{Region "Angulo de rotação das válvulas"}
	//Linha 1
	CA1_L1_V1_POSIC AT %I*	:DUT_PosicValvula;
	CA1_L1_V2_POSIC AT %I*	:DUT_PosicValvula;
	CA1_L1_V3_POSIC AT %I*	:DUT_PosicValvula;
	CA1_L1_V4_POSIC AT %I*	:DUT_PosicValvula;
	//Linha 2
	CA1_L2_V1_POSIC AT %I*	:DUT_PosicValvula;
	CA1_L2_V2_POSIC AT %I*	:DUT_PosicValvula;
	CA1_L2_V3_POSIC AT %I*	:DUT_PosicValvula;
	CA1_L2_V4_POSIC AT %I*	:DUT_PosicValvula;
	//Linha 3
	CA1_L3_V1_POSIC AT %I*	:DUT_PosicValvula;
	CA1_L3_V2_POSIC AT %I*	:DUT_PosicValvula;
	CA1_L3_V3_POSIC AT %I*	:DUT_PosicValvula;
	CA1_L3_V4_POSIC AT %I*	:DUT_PosicValvula;
	//Linha 4
	CA1_L4_V1_POSIC AT %I*	:DUT_PosicValvula;
	CA1_L4_V2_POSIC AT %I*	:DUT_PosicValvula;
	CA1_L4_V3_POSIC AT %I*	:DUT_PosicValvula;
	CA1_L4_V4_POSIC AT %I*	:DUT_PosicValvula;
	
	//Linha 5
	CA2_L5_V1_POSIC AT %I*	:DUT_PosicValvula;
	CA2_L5_V2_POSIC AT %I*	:DUT_PosicValvula;
	CA2_L5_V3_POSIC AT %I*	:DUT_PosicValvula;
	CA2_L5_V4_POSIC AT %I*	:DUT_PosicValvula;
	//Linha 6
	CA2_L6_V1_POSIC AT %I*	:DUT_PosicValvula;
	CA2_L6_V2_POSIC AT %I*	:DUT_PosicValvula;
	CA2_L6_V3_POSIC AT %I*	:DUT_PosicValvula;
	CA2_L6_V4_POSIC AT %I*	:DUT_PosicValvula;
	//Linha 7
	CA2_L7_V1_POSIC AT %I*	:DUT_PosicValvula;
	CA2_L7_V2_POSIC AT %I*	:DUT_PosicValvula;
	CA2_L7_V3_POSIC AT %I*	:DUT_PosicValvula;
	CA2_L7_V4_POSIC AT %I*	:DUT_PosicValvula;
	//Linha 8
	CA2_L8_V1_POSIC AT %I*	:DUT_PosicValvula;
	CA2_L8_V2_POSIC AT %I*	:DUT_PosicValvula;
	CA2_L8_V3_POSIC AT %I*	:DUT_PosicValvula;
	CA2_L8_V4_POSIC AT %I*	:DUT_PosicValvula;
	
	//Linha 9
	CA3_L9_V1_POSIC AT %I*	:DUT_PosicValvula;
	CA3_L9_V2_POSIC AT %I*	:DUT_PosicValvula;
	CA3_L9_V3_POSIC AT %I*	:DUT_PosicValvula;
	CA3_L9_V4_POSIC AT %I*	:DUT_PosicValvula;
	//Linha 10
	CA3_L10_V1_POSIC AT %I*	:DUT_PosicValvula;
	CA3_L10_V2_POSIC AT %I*	:DUT_PosicValvula;
	CA3_L10_V3_POSIC AT %I*	:DUT_PosicValvula;
	CA3_L10_V4_POSIC AT %I*	:DUT_PosicValvula;
	//Linha 11
	CA3_L11_V1_POSIC AT %I*	:DUT_PosicValvula;
	CA3_L11_V2_POSIC AT %I*	:DUT_PosicValvula;
	CA3_L11_V3_POSIC AT %I*	:DUT_PosicValvula;
	CA3_L11_V4_POSIC AT %I*	:DUT_PosicValvula;
	//Linha 12
	CA3_L12_V1_POSIC AT %I*	:DUT_PosicValvula;
	CA3_L12_V2_POSIC AT %I*	:DUT_PosicValvula;
	CA3_L12_V3_POSIC AT %I*	:DUT_PosicValvula;
	CA3_L12_V4_POSIC AT %I*	:DUT_PosicValvula;
{endregion}
	
	
	
	
END_VAR

// ---- GVLs/HMI.TcGVL
{attribute 'qualified_only'}
VAR_GLOBAL
	//Hora de ajuste
	HoraParaAjuste:DT;
	
	//Lavagem das linhas
	IniciaLavagem :BOOL;	//Inicia lavagem na linha selecionada
	PararLavagem:BOOL;		//Interrompe a lavagem
	AbreValvResid:BOOL;		//Abre a válvula de água resisdual
	AbreValvLimpa:BOOL;		//Abre a válvula de água limpa
	
	// General
	bModo_Auto:BOOL;
	bModo_Ciclico:BOOL;
	bModo_UnCiclo:BOOL;
	bMarcha		:BOOL;
	bParada		:BOOL;
	bReset_Alarma:BOOL;
	bPB_vaciarTolva:BOOL;
	bRun			:BOOL;
	bPesoFueraTolerancia :BOOL;
	bDemoraCargaBalanza	:BOOL;
	bDescargarBalanza	:BOOL;
	iCircuito_a_calibrar:INT;
	bPararTolvaSupVacia:BOOL;
	tTiempoBatch:DINT;

	//Agitadores
	PP1_L1_AG_Cmd_Man:BOOL;
	PP1_L1_AG_Alr:BOOL;
	PP1_L1_AG_Alr_discr:BOOL;
	PP1_L1_AG_Estado:INT;
	bPP1_L1_AG_HsParc:DINT;
	bPP1_L1_AG_HsTot:DINT;	
	bPP1_L1_AG_RstHs:BOOL;
	bPP1_L1_AG_RstALr:BOOL;
	//
	PP1_L2_AG_Cmd_Man:BOOL;
	PP1_L2_AG_Alr:BOOL;
	PP1_L2_AG_Alr_discr:BOOL;
	PP1_L2_AG_Estado:INT;
	bPP1_L2_AG_HsParc:DINT;
	bPP1_L2_AG_HsTot:DINT;	
	bPP1_L2_AG_RstHs:BOOL;
	bPP1_L2_AG_RstALr:BOOL;
	//
	PP1_L3_AG_Cmd_Man:BOOL;
	PP1_L3_AG_Alr:BOOL;
	PP1_L3_AG_Alr_discr:BOOL;
	PP1_L3_AG_Estado:INT;
	bPP1_L3_AG_HsParc:DINT;
	bPP1_L3_AG_HsTot:DINT;	
	bPP1_L3_AG_RstHs:BOOL;
	bPP1_L3_AG_RstALr:BOOL;
	//
	PP1_L4_AG_Cmd_Man:BOOL;
	PP1_L4_AG_Alr:BOOL;
	PP1_L4_AG_Alr_discr:BOOL;
	PP1_L4_AG_Estado:INT;
	bPP1_L4_AG_HsParc:DINT;
	bPP1_L4_AG_HsTot:DINT;	
	bPP1_L4_AG_RstHs:BOOL;
	bPP1_L4_AG_RstALr:BOOL;
	
	PP2_L5_AG_Cmd_Man:BOOL;
	PP2_L5_AG_Alr:BOOL;
	PP2_L5_AG_Alr_discr:BOOL;
	PP2_L5_AG_Estado:INT;
	bPP2_L5_AG_HsParc:DINT;
	bPP2_L5_AG_HsTot:DINT;	
	bPP2_L5_AG_RstHs:BOOL;
	bPP2_L5_AG_RstALr:BOOL;
	//
	PP2_L6_AG_Cmd_Man:BOOL;
	PP2_L6_AG_Alr:BOOL;
	PP2_L6_AG_Alr_discr:BOOL;
	PP2_L6_AG_Estado:INT;
	bPP2_L6_AG_HsParc:DINT;
	bPP2_L6_AG_HsTot:DINT;	
	bPP2_L6_AG_RstHs:BOOL;
	bPP2_L6_AG_RstALr:BOOL;
	//
	PP2_L7_AG_Cmd_Man:BOOL;
	PP2_L7_AG_Alr:BOOL;
	PP2_L7_AG_Alr_discr:BOOL;
	PP2_L7_AG_Estado:INT;
	bPP2_L7_AG_HsParc:DINT;
	bPP2_L7_AG_HsTot:DINT;	
	bPP2_L7_AG_RstHs:BOOL;
	bPP2_L7_AG_RstALr:BOOL;
		//
	PP2_L8_AG_Cmd_Man:BOOL;
	PP2_L8_AG_Alr:BOOL;
	PP2_L8_AG_Alr_discr:BOOL;
	PP2_L8_AG_Estado:INT;
	bPP2_L8_AG_HsParc:DINT;
	bPP2_L8_AG_HsTot:DINT;	
	bPP2_L8_AG_RstHs:BOOL;
	bPP2_L8_AG_RstALr:BOOL;
	//
	PP3_L9_AG_Cmd_Man:BOOL;
	PP3_L9_AG_Alr:BOOL;
	PP3_L9_AG_Alr_discr:BOOL;
	PP3_L9_AG_Estado:INT;
	bPP3_L9_AG_HsParc:DINT;
	bPP3_L9_AG_HsTot:DINT;	
	bPP3_L9_AG_RstHs:BOOL;
	bPP3_L9_AG_RstALr:BOOL;
	//
	PP3_L10_AG_Cmd_Man:BOOL;
	PP3_L10_AG_Alr:BOOL;
	PP3_L10_AG_Alr_discr:BOOL;
	PP3_L10_AG_Estado:INT;
	bPP3_L10_AG_HsParc:DINT;
	bPP3_L10_AG_HsTot:DINT;	
	bPP3_L10_AG_RstHs:BOOL;
	bPP3_L10_AG_RstALr:BOOL;
	//
	PP3_L11_AG_Cmd_Man:BOOL;
	PP3_L11_AG_Alr:BOOL;
	PP3_L11_AG_Alr_discr:BOOL;
	PP3_L11_AG_Estado:INT;
	bPP3_L11_AG_HsParc:DINT;
	bPP3_L11_AG_HsTot:DINT;	
	bPP3_L11_AG_RstHs:BOOL;
	bPP3_L11_AG_RstALr:BOOL;
	//
	PP3_L12_AG_Cmd_Man:BOOL;
	PP3_L12_AG_Alr:BOOL;
	PP3_L12_AG_Alr_discr:BOOL;
	PP3_L12_AG_Estado:INT;
	bPP3_L12_AG_HsParc:DINT;
	bPP3_L12_AG_HsTot:DINT;	
	bPP3_L12_AG_RstHs:BOOL;
	bPP3_L12_AG_RstALr:BOOL;
	
	
	//Soplador tratadora
	TR_S_VE1_Cmd_Man:BOOL;
	TR_S_VE1_Alr:BOOL;
	TR_S_VE1_Alr_discr:BOOL;
	TR_S_VE1_Estado:INT;
	TR_S_VE1_HsParc:DINT;
	TR_S_VE1_HsTot:DINT;	
	TR_S_VE1_RstHs:BOOL;
	TR_S_VE1_RstAlr:BOOL;
	
	//Lavado Gral
	bBypassNivelAguaResidual:BOOL;
	
	//Lavado Circuito 1
	bInicioLavado_Cir1:BOOL;//Inicio de Lavado
	bModoECO_Cir1:BOOL;//Seleccion modo ECO
	bCancelarLavado_Cir1:BOOL;//Cancelacion de lavado (finaliza con circuito vacio)
	wEstadoLavado_Cir1:WORD; //1=vaciado 2=prelavado 3=lavado
	iCantCiclosLavado_Cir1:INT;//Cantidad de ciclos a realizar de Lavado
	iCantCiclosECO_Cir1:INT;//Cantidad de ciclos a realizar de Eco
	rPorcECO_Cir1:REAL;//Porcentaje de ciclos ECO en relacion al total pedido (ECO+Lavado)
	rPorcLavado_Cir1:REAL;//Porcentaje de ciclos Lavado en relacion al total pedido (ECO+Lavado)
	rPorcAvance_Cir1:REAL;//Porcentaje de avance en relacion al total pedido (ECO+Lavado)
	tSetTmrVaciado_Cir1:TIME;//Tiempo luego de detectar caudalimetro inferior en cero
	tSetTmrLlenado_Cir1:TIME;//Tiempo luego de detectar caudalimetro superior mayor a cero
	rVelBbaVaciado_Cir1:REAL;//Velocidad de bomba durante vaciado (unidad?)
	rVelBbaLlenado_Cir1:REAL;//Velocidad de bomba durante llenado (unidad?)
	
	//valvula descarga semilla de tambor
	TR_S_V1_Cmd_Man		:BOOL;
	TR_S_V1_Alr			:BOOL;
	TR_S_V1_Alr_discr	:BOOL;
	TR_S_V1_Estado		:INT;  // 1= cerrado 2=abierto 3=alarma 4=emergencia
	TR_S_V1_EventoParc	:DINT;//cant de actuaciones parciales
	TR_S_V1_EventoTot	:DINT;//cant de actuaciones totales
	
	//valvula carga grueso semilla a balanza
	TR_S_V2_Cmd_Man		:BOOL;
	TR_S_V2_Alr			:BOOL;
	TR_S_V2_Alr_discr	:BOOL;
	TR_S_V2_Estado		:INT;
	
	//valvula carga fino semilla a balanza
	TR_S_V3_Cmd_Man		:BOOL;
	TR_S_V3_Alr			:BOOL;
	TR_S_V3_Alr_discr	:BOOL;
	TR_S_V3_Estado		:INT;
	
	//valvula descarga semilla de balanza
	TR_S_V4_Cmd_Man		:BOOL;
	TR_S_V4_Alr			:BOOL;
	TR_S_V4_Alr_discr	:BOOL;
	TR_S_V4_Estado		:INT;
	
	
	//Homogenizador
	CmdM_TR_S_VF1		:BOOL; //marcha en manual
	CmdR_TR_S_VF1		:BOOL; //seleccion reversa en manual
	StMarcha_TR_S_VF1	:BOOL; //confirmacion en marcha
	StAlarma_TR_S_VF1	:BOOL;
	StVeloc_TR_S_VF1	:INT;	
	
	//Aspersor
	CmdM_TR_S_VF2		:BOOL; //marcha en manual
	CmdR_TR_S_VF2		:BOOL; //seleccion reversa en manual
	StMarcha_TR_S_VF2	:BOOL; //confirmacion en marcha
	StAlarma_TR_S_VF2	:BOOL;
	StVeloc_TR_S_VF2	:INT;	
	
	//Valv Calibracion L1
	CA1_L1_V1_estado	:INT;
	CA1_L1_V1_Cmd_Man	:BOOL;
	CA1_L1_V1_RsAlr		:BOOL;
	//Valv Calibracion L2
	CA1_L2_V1_estado	:INT;
	CA1_L2_V1_Cmd_Man	:BOOL;
	CA1_L2_V1_RsAlr		:BOOL;	
	//Valv Calibracion L3
	CA1_L3_V1_estado	:INT;
	CA1_L3_V1_Cmd_Man	:BOOL;
	CA1_L3_V1_RsAlr		:BOOL;
	//Valv Calibracion L4
	CA1_L4_V1_estado	:INT;
	CA1_L4_V1_Cmd_Man	:BOOL;
	CA1_L4_V1_RsAlr		:BOOL;
	//Valv Calibracion L5
	CA2_L5_V1_estado	:INT;
	CA2_L5_V1_Cmd_Man	:BOOL;
	CA2_L5_V1_RsAlr		:BOOL;
	//Valv Calibracion L6
	CA2_L6_V1_estado	:INT;
	CA2_L6_V1_Cmd_Man	:BOOL;
	CA2_L6_V1_RsAlr		:BOOL;
	//Valv Calibracion L7
	CA2_L7_V1_estado	:INT;
	CA2_L7_V1_Cmd_Man	:BOOL;
	CA2_L7_V1_RsAlr		:BOOL;
	//Valv Calibracion L8
	CA2_L8_V1_estado	:INT;
	CA2_L8_V1_Cmd_Man	:BOOL;
	CA2_L8_V1_RsAlr		:BOOL;				
	//Valv Calibracion L9
	CA3_L9_V1_estado	:INT;
	CA3_L9_V1_Cmd_Man	:BOOL;	
	CA3_L9_V1_RsAlr		:BOOL;
	//Valv Calibracion L10
	CA3_L10_V1_estado	:INT;
	CA3_L10_V1_Cmd_Man	:BOOL;
	CA3_L10_V1_RsAlr		:BOOL;
	//Valv Calibracion L11
	CA3_L11_V1_estado	:INT;
	CA3_L11_V1_Cmd_Man	:BOOL;
	CA3_L11_V1_RsAlr		:BOOL;	
	//Valv Calibracion L12
	CA3_L12_V1_estado	:INT;
	CA3_L12_V1_Cmd_Man	:BOOL;
	CA3_L12_V1_RsAlr		:BOOL;		
	
	//Valv Calibracion L1
	CA1_L1_V2_estado	:INT;
	CA1_L1_V2_Cmd_Man	:BOOL;
	CA1_L1_V2_RsAlr		:BOOL;
	//Valv Lavado L1
	CA1_L1_V3_estado	:INT;
	CA1_L1_V3_Cmd_Man	:BOOL;
	CA1_L1_V3_RsAlr		:BOOL;
	//Valv IBC L1
	CA1_L1_V4_estado	:INT;
	CA1_L1_V4_Cmd_Man	:BOOL;
	CA1_L1_V4_RsAlr		:BOOL;
	//Valv Calibracion L2
	CA1_L2_V2_estado	:INT;
	CA1_L2_V2_Cmd_Man	:BOOL;
	CA1_L2_V2_RsAlr		:BOOL;
	//Valv Lavado L2
	CA1_L2_V3_estado	:INT;
	CA1_L2_V3_Cmd_Man	:BOOL;
	CA1_L2_V3_RsAlr		:BOOL;
	//Valv IBC L2
	CA1_L2_V4_estado	:INT;
	CA1_L2_V4_Cmd_Man	:BOOL;
	CA1_L2_V4_RsAlr		:BOOL;
	//Valv Calibracion L3
	CA1_L3_V2_estado	:INT;
	CA1_L3_V2_Cmd_Man	:BOOL;
	CA1_L3_V2_RsAlr		:BOOL;
	//Valv Lavado L3
	CA1_L3_V3_estado	:INT;
	CA1_L3_V3_Cmd_Man	:BOOL;
	CA1_L3_V3_RsAlr		:BOOL;
	//Valv IBC L3
	CA1_L3_V4_estado	:INT;
	CA1_L3_V4_Cmd_Man	:BOOL;
	CA1_L3_V4_RsAlr		:BOOL;
	//Valv Calibracion L4
	CA1_L4_V2_estado	:INT;
	CA1_L4_V2_Cmd_Man	:BOOL;
	CA1_L4_V2_RsAlr		:BOOL;
	//Valv Lavado L4
	CA1_L4_V3_estado	:INT;
	CA1_L4_V3_Cmd_Man	:BOOL;
	CA1_L4_V3_RsAlr		:BOOL;
	//Valv IBC L4
	CA1_L4_V4_estado	:INT;
	CA1_L4_V4_Cmd_Man	:BOOL;
	CA1_L4_V4_RsAlr		:BOOL;
	//Valv Calibracion L5
	CA2_L5_V2_estado	:INT;
	CA2_L5_V2_Cmd_Man	:BOOL;
	CA2_L5_V2_RsAlr		:BOOL;
	//Valv Lavado L5
	CA2_L5_V3_estado	:INT;
	CA2_L5_V3_Cmd_Man	:BOOL;
	CA2_L5_V3_RsAlr		:BOOL;
	//Valv IBC L5
	CA2_L5_V4_estado	:INT;
	CA2_L5_V4_Cmd_Man	:BOOL;
	CA2_L5_V4_RsAlr		:BOOL;
	//Valv Calibracion L6
	CA2_L6_V2_estado	:INT;
	CA2_L6_V2_Cmd_Man	:BOOL;
	CA2_L6_V2_RsAlr		:BOOL;
	//Valv Lavado L6
	CA2_L6_V3_estado	:INT;
	CA2_L6_V3_Cmd_Man	:BOOL;
	CA2_L6_V3_RsAlr		:BOOL;
	//Valv IBC L6
	CA2_L6_V4_estado	:INT;
	CA2_L6_V4_Cmd_Man	:BOOL;
	CA2_L6_V4_RsAlr		:BOOL;
	//Valv Calibracion L7
	CA2_L7_V2_estado	:INT;
	CA2_L7_V2_Cmd_Man	:BOOL;
	CA2_L7_V2_RsAlr		:BOOL;
	//Valv Lavado L7
	CA2_L7_V3_estado	:INT;
	CA2_L7_V3_Cmd_Man	:BOOL;
	CA2_L7_V3_RsAlr		:BOOL;
	//Valv IBC L7
	CA2_L7_V4_estado	:INT;
	CA2_L7_V4_Cmd_Man	:BOOL;
	CA2_L7_V4_RsAlr		:BOOL;
	//Valv Calibracion L8
	CA2_L8_V2_estado	:INT;
	CA2_L8_V2_Cmd_Man	:BOOL;
	CA2_L8_V2_RsAlr		:BOOL;
	//Valv Lavado L8
	CA2_L8_V3_estado	:INT;
	CA2_L8_V3_Cmd_Man	:BOOL;
	CA2_L8_V3_RsAlr		:BOOL;
	//Valv IBC L8
	CA2_L8_V4_estado	:INT;
	CA2_L8_V4_Cmd_Man	:BOOL;
	CA2_L8_V4_RsAlr		:BOOL;
	//Valv Calibracion L9
	CA3_L9_V2_estado	:INT;
	CA3_L9_V2_Cmd_Man	:BOOL;
	CA3_L9_V2_RsAlr		:BOOL;
	//Valv Lavado L9
	CA3_L9_V3_estado	:INT;
	CA3_L9_V3_Cmd_Man	:BOOL;
	CA3_L9_V3_RsAlr		:BOOL;
	//Valv IBC L9
	CA3_L9_V4_estado	:INT;
	CA3_L9_V4_Cmd_Man	:BOOL;
	CA3_L9_V4_RsAlr		:BOOL;
	//Valv Calibracion L10
	CA3_L10_V2_estado	:INT;
	CA3_L10_V2_Cmd_Man	:BOOL;
	CA3_L10_V2_RsAlr	:BOOL;
	//Valv Lavado L10
	CA3_L10_V3_estado	:INT;
	CA3_L10_V3_Cmd_Man	:BOOL;
	CA3_L10_V3_RsAlr	:BOOL;
	//Valv IBC L10
	CA3_L10_V4_estado	:INT;
	CA3_L10_V4_Cmd_Man	:BOOL;
	CA3_L10_V4_RsAlr	:BOOL;
	//Valv Calibracion L11
	CA3_L11_V2_estado	:INT;
	CA3_L11_V2_Cmd_Man	:BOOL;
	CA3_L11_V2_RsAlr	:BOOL;
	//Valv Lavado L11
	CA3_L11_V3_estado	:INT;
	CA3_L11_V3_Cmd_Man	:BOOL;
	CA3_L11_V3_RsAlr	:BOOL;
	//Valv IBC L11
	CA3_L11_V4_estado	:INT;
	CA3_L11_V4_Cmd_Man	:BOOL;
	CA3_L11_V4_RsAlr	:BOOL;
	//Valv Calibracion L12
	CA3_L12_V2_estado	:INT;
	CA3_L12_V2_Cmd_Man	:BOOL;
	CA3_L12_V2_RsAlr	:BOOL;
	//Valv Lavado L12
	CA3_L12_V3_estado	:INT;
	CA3_L12_V3_Cmd_Man	:BOOL;
	CA3_L12_V3_RsAlr	:BOOL;
	//Valv IBC L12
	CA3_L12_V4_estado	:INT;
	CA3_L12_V4_Cmd_Man	:BOOL;
	CA3_L12_V4_RsAlr	:BOOL;
	//Valv Agua limpia
	PU_Lav_V5_estado	:INT;
	PU_Lav_V5_Cmd_Man	:BOOL;
	PU_Lav_V5_RsAlr		:BOOL;
	//Valv Agua residual
	PU_Lav_V6_estado	:INT;
	PU_Lav_V6_Cmd_Man	:BOOL;
	PU_Lav_V6_RsAlr		:BOOL;	
	
	//Bomba circuito L1
	CmdM_PC1_L1_BD	:BOOL; //marcha en manual
	CmdR_PC1_L1_BD	:BOOL; //seleccion reversa en manual
	StMarcha_PC1_L1_BD :BOOL; //confirmacion bomba en marcha
	StAlarma_PC1_L1_BD :BOOL;
	StVeloc_PC1_L1_BD :INT;
	//Bomba circuito L2
	CmdM_PC1_L2_BD	:BOOL; //marcha en manual
	CmdR_PC1_L2_BD	:BOOL; //seleccion reversa en manual
	StMarcha_PC1_L2_BD :BOOL; //confirmacion bomba en marcha
	StAlarma_PC1_L2_BD :BOOL;
	StVeloc_PC1_L2_BD :INT;	
	//Bomba circuito L3
	CmdM_PC1_L3_BD	:BOOL; //marcha en manual
	CmdR_PC1_L3_BD	:BOOL; //seleccion reversa en manual
	StMarcha_PC1_L3_BD :BOOL; //confirmacion bomba en marcha
	StAlarma_PC1_L3_BD :BOOL;
	StVeloc_PC1_L3_BD :INT;	
	//Bomba circuito L4
	CmdM_PC1_L4_BD	:BOOL; //marcha en manual
	CmdR_PC1_L4_BD	:BOOL; //seleccion reversa en manual
	StMarcha_PC1_L4_BD :BOOL; //confirmacion bomba en marcha
	StAlarma_PC1_L4_BD :BOOL;
	StVeloc_PC1_L4_BD :INT;		
	//Bomba circuito L5
	CmdM_PC2_L5_BD	:BOOL; //marcha en manual
	CmdR_PC2_L5_BD	:BOOL; //seleccion reversa en manual
	StMarcha_PC2_L5_BD :BOOL; //confirmacion bomba en marcha
	StAlarma_PC2_L5_BD :BOOL;
	StVeloc_PC2_L5_BD :INT;	
	//Bomba circuito L6
	CmdM_PC2_L6_BD	:BOOL; //marcha en manual
	CmdR_PC2_L6_BD	:BOOL; //seleccion reversa en manual
	StMarcha_PC2_L6_BD :BOOL; //confirmacion bomba en marcha
	StAlarma_PC2_L6_BD :BOOL;
	StVeloc_PC2_L6_BD :INT;	
	//Bomba circuito L7
	CmdM_PC2_L7_BD	:BOOL; //marcha en manual
	CmdR_PC2_L7_BD	:BOOL; //seleccion reversa en manual
	StMarcha_PC2_L7_BD :BOOL; //confirmacion bomba en marcha
	StAlarma_PC2_L7_BD :BOOL;
	StVeloc_PC2_L7_BD :INT;	
	//Bomba circuito L8
	CmdM_PC2_L8_BD	:BOOL; //marcha en manual
	CmdR_PC2_L8_BD	:BOOL; //seleccion reversa en manual
	StMarcha_PC2_L8_BD :BOOL; //confirmacion bomba en marcha
	StAlarma_PC2_L8_BD :BOOL;
	StVeloc_PC2_L8_BD :INT;					
	//Bomba circuito L9
	CmdM_PC3_L9_BD	:BOOL; //marcha en manual
	CmdR_PC3_L9_BD	:BOOL; //seleccion reversa en manual
	StMarcha_PC3_L9_BD :BOOL; //confirmacion bomba en marcha
	StAlarma_PC3_L9_BD :BOOL;
	StVeloc_PC3_L9_BD :INT;	
	//Bomba circuito L10
	CmdM_PC3_L10_BD	:BOOL; //marcha en manual
	CmdR_PC3_L10_BD	:BOOL; //seleccion reversa en manual
	StMarcha_PC3_L10_BD :BOOL; //confirmacion bomba en marcha
	StAlarma_PC3_L10_BD :BOOL;
	StVeloc_PC3_L10_BD :INT;
	//Bomba circuito L11
	CmdM_PC3_L11_BD	:BOOL; //marcha en manual
	CmdR_PC3_L11_BD	:BOOL; //seleccion reversa en manual
	StMarcha_PC3_L11_BD :BOOL; //confirmacion bomba en marcha
	StAlarma_PC3_L11_BD :BOOL;
	StVeloc_PC3_L11_BD :INT;
	//Bomba circuito L12
	CmdM_PC3_L12_BD	:BOOL; //marcha en manual
	CmdR_PC3_L12_BD	:BOOL; //seleccion reversa en manual
	StMarcha_PC3_L12_BD :BOOL; //confirmacion bomba en marcha
	StAlarma_PC3_L12_BD :BOOL;
	StVeloc_PC3_L12_BD :INT;		
	
	//Caudalimetros Calibracion
	CA1_L1_FT1_caudal :REAL;
	CA1_L1_FT1_temp :REAL;
	CA1_L2_FT1_caudal :REAL;
	CA1_L2_FT1_temp :REAL;	
	CA1_L3_FT1_caudal :REAL;
	CA1_L3_FT1_tot	:REAL;
	CA1_L3_FT1_temp :REAL;
	CA1_L4_FT1_caudal :REAL;
	CA1_L4_FT1_temp :REAL;
	CA2_L5_FT1_caudal :REAL;
	CA2_L5_FT1_temp :REAL;
	CA2_L6_FT1_caudal :REAL;
	CA2_L6_FT1_temp :REAL;	
	CA2_L7_FT1_caudal :REAL;
	CA2_L7_FT1_temp :REAL;
	CA2_L8_FT1_caudal :REAL;
	CA2_L8_FT1_temp :REAL;
	CA3_L9_FT1_caudal :REAL;
	CA3_L9_FT1_temp :REAL;
	CA3_L10_FT1_caudal :REAL;
	CA3_L10_FT1_temp :REAL;
	CA3_L11_FT1_caudal :REAL;
	CA3_L11_FT1_temp :REAL;
	CA3_L12_FT1_caudal :REAL;
	CA3_L12_FT1_temp :REAL;
	//Caudalimetros Tratadora
	TR_L1_FT2_caudal :REAL;
	TR_L1_FT2_temp :REAL;
	TR_L2_FT2_caudal :REAL;
	TR_L2_FT2_temp :REAL;	
	TR_L3_FT2_caudal :REAL;
	TR_L3_FT2_temp :REAL;
	TR_L4_FT2_caudal :REAL;
	TR_L4_FT2_temp :REAL;
	TR_L5_FT2_caudal :REAL;
	TR_L5_FT2_temp :REAL;
	TR_L6_FT2_caudal :REAL;
	TR_L6_FT2_temp :REAL;	
	TR_L7_FT2_caudal :REAL;
	TR_L7_FT2_temp :REAL;
	TR_L8_FT2_caudal :REAL;
	TR_L8_FT2_temp :REAL;
	TR_L9_FT2_caudal :REAL;
	TR_L9_FT2_temp :REAL;
	TR_L10_FT2_caudal :REAL;
	TR_L10_FT2_temp :REAL;
	TR_L11_FT2_caudal :REAL;
	TR_L11_FT2_temp :REAL;
	TR_L12_FT2_caudal :REAL;
	TR_L12_FT2_temp :REAL;
	//Balanza probeta CA1
	bCmd_Zero_WT_CA1 :BOOL;
	bCmd_Full_WT_CA1 :BOOL;
	bCmd_LoadReference_WT_CA1:BOOL;
	rPesoPatron_WT_CA1 :REAL;
	bCalibrado_WT_CA1:BOOL;
	//Balanza probeta CA2
	bCmd_Zero_WT_CA2 :BOOL;
	bCmd_Full_WT_CA2 :BOOL;
	bCmd_LoadReference_WT_CA2:BOOL;
	rPesoPatron_WT_CA2 :REAL;
	bCalibrado_WT_CA2:BOOL;	
	//Balanza probeta CA3
	bCmd_Zero_WT_CA3 :BOOL;
	bCmd_Full_WT_CA3 :BOOL;
	bCmd_LoadReference_WT_CA3:BOOL;
	rPesoPatron_WT_CA3 :REAL;
	bCalibrado_WT_CA3:BOOL;
	//Balanza IBC L1
	bCmd_Zero_WT1_PU1 :BOOL;
	bCmd_Full_WT1_PU1 :BOOL;
	bCmd_LoadReference_WT1_PU1:BOOL;
	rPesoPatron_WT1_PU1 :REAL;
	bCalibrado_WT1_PU1:BOOL;
	//Balanza IBC L2
	bCmd_Zero_WT2_PU1 :BOOL;
	bCmd_Full_WT2_PU1 :BOOL;
	bCmd_LoadReference_WT2_PU1:BOOL;
	rPesoPatron_WT2_PU1 :REAL;
	bCalibrado_WT2_PU1:BOOL;
	//Balanza IBC L3
	bCmd_Zero_WT3_PU1 :BOOL;
	bCmd_Full_WT3_PU1 :BOOL;
	bCmd_LoadReference_WT3_PU1:BOOL;
	rPesoPatron_WT3_PU1 :REAL;
	bCalibrado_WT3_PU1:BOOL;
	//Balanza IBC L4
	bCmd_Zero_WT4_PU1 :BOOL;
	bCmd_Full_WT4_PU1 :BOOL;
	bCmd_LoadReference_WT4_PU1:BOOL;
	rPesoPatron_WT4_PU1 :REAL;
	bCalibrado_WT4_PU1:BOOL;
	//Balanza IBC L5
	bCmd_Zero_WT5_PU2 :BOOL;
	bCmd_Full_WT5_PU2 :BOOL;
	bCmd_LoadReference_WT5_PU2:BOOL;
	rPesoPatron_WT5_PU2 :REAL;
	bCalibrado_WT5_PU2:BOOL;
	//Balanza IBC L6
	bCmd_Zero_WT6_PU2 :BOOL;
	bCmd_Full_WT6_PU2 :BOOL;
	bCmd_LoadReference_WT6_PU2:BOOL;
	rPesoPatron_WT6_PU2 :REAL;
	bCalibrado_WT6_PU2:BOOL;
	//Balanza IBC L7
	bCmd_Zero_WT7_PU2 :BOOL;
	bCmd_Full_WT7_PU2 :BOOL;
	bCmd_LoadReference_WT7_PU2:BOOL;
	rPesoPatron_WT7_PU2 :REAL;
	bCalibrado_WT7_PU2:BOOL;
	//Balanza IBC L8
	bCmd_Zero_WT8_PU2 :BOOL;
	bCmd_Full_WT8_PU2 :BOOL;
	bCmd_LoadReference_WT8_PU2:BOOL;
	rPesoPatron_WT8_PU2 :REAL;
	bCalibrado_WT8_PU2:BOOL;
	//Balanza IBC L9
	bCmd_Zero_WT9_PU3 :BOOL;
	bCmd_Full_WT9_PU3 :BOOL;
	bCmd_LoadReference_WT9_PU3:BOOL;
	rPesoPatron_WT9_PU3 :REAL;
	bCalibrado_WT9_PU3:BOOL;
	//Balanza IBC L10
	bCmd_Zero_WT10_PU3 :BOOL;
	bCmd_Full_WT10_PU3 :BOOL;
	bCmd_LoadReference_WT10_PU3:BOOL;
	rPesoPatron_WT10_PU3 :REAL;
	bCalibrado_WT10_PU3:BOOL;
	//Balanza IBC L11
	bCmd_Zero_WT11_PU3 :BOOL;
	bCmd_Full_WT11_PU3 :BOOL;
	bCmd_LoadReference_WT11_PU3:BOOL;
	rPesoPatron_WT11_PU3 :REAL;
	bCalibrado_WT11_PU3:BOOL;
	//Balanza IBC L12
	bCmd_Zero_WT12_PU3 :BOOL;
	bCmd_Full_WT12_PU3 :BOOL;
	bCmd_LoadReference_WT12_PU3:BOOL;
	rPesoPatron_WT12_PU3 :REAL;
	bCalibrado_WT12_PU3:BOOL;	
	//Balanza Semilla
	bCmd_Zero_TR_S_WT1 :BOOL;
	bCmd_Full_TR_S_WT1 :BOOL;
	bCmd_LoadReference_TR_S_WT1:BOOL;
	bInicio_Cal_TR_S_WT1 :BOOL;
	bCalibrando:BOOL;
	bCalibrado:BOOL;
	
	//Dosificador Polvo 1
	CmdM_TR_P1_VF	:BOOL; //marcha en manual
	CmdR_TR_P1_VF	:BOOL; //seleccion reversa en manual
	StMarcha_TR_P1_VF :BOOL; //confirmacion motor en marcha
	StAlarma_TR_P1_VF :BOOL;
	StVeloc_TR_P1_VF :INT;
	//Dosificador Polvo 2
	CmdM_TR_P2_VF	:BOOL; //marcha en manual
	CmdR_TR_P2_VF	:BOOL; //seleccion reversa en manual
	StMarcha_TR_P2_VF :BOOL; //confirmacion motor en marcha
	StAlarma_TR_P2_VF :BOOL;
	StVeloc_TR_P2_VF :INT;
	//Balanza Polvo 1
	bCmd_Zero_TR_P1_WT1 :BOOL;
	bCmd_Full_TR_P1_WT1 :BOOL;
	bCmd_LoadReference_TR_P1_WT1:BOOL;
	rPesoPatron_TR_P1_WT1 :REAL;
	bCalibrado_TR_P1_WT1:BOOL;	
	//Balanza Polvo 2
	bCmd_Zero_TR_P2_WT1 :BOOL;
	bCmd_Full_TR_P2_WT1 :BOOL;
	bCmd_LoadReference_TR_P2_WT1:BOOL;
	rPesoPatron_TR_P2_WT1 :REAL;
	bCalibrado_TR_P2_WT1:BOOL;	
	//Vibrador Polvo 1
	CmdM_TR_P1_VI	:BOOL; //marcha en manual
	CmdR_TR_P1_VI	:BOOL; //seleccion reversa en manual
	CmdV_TR_P1_VI	:REAL; // velocidad manual en % 
	StMarcha_TR_P1_VI :BOOL; //confirmacion motor en marcha
	StAlarma_TR_P1_VI :BOOL;
	StVeloc_TR_P1_VI :INT;
	//Vibrador Polvo 2
	CmdM_TR_P2_VI	:BOOL; //marcha en manual
	CmdR_TR_P2_VI	:BOOL; //seleccion reversa en manual
	CmdV_TR_P2_VI	:REAL; // velocidad manual en % 
	StMarcha_TR_P2_VI :BOOL; //confirmacion motor en marcha
	StAlarma_TR_P2_VI :BOOL;
	StVeloc_TR_P2_VI :INT;
	
	TR_P1_Alr_ZS :BOOL;//alarma zero speed dosificador Polvo 1
	TR_P1_Alr_ZS_RstAlr :BOOL;
	TR_P2_Alr_ZS :BOOL;//alarma zero speed dosificador Polvo 2
	TR_P2_Alr_ZS_RstAlr :BOOL;	
	
	//Perifericos Elevador 1
	CmdM_PE_B_VF1	:BOOL; //marcha en manual
	CmdR_PE_B_VF1	:BOOL; //seleccion reversa en manual
	StMarcha_PE_B_VF1 :BOOL; //confirmacion motor en marcha
	StAlarma_PE_B_VF1 :BOOL;
	StVeloc_PE_B_VF1 :INT;
	//Perifericos Elevador 2
	CmdM_PE_H_VF1	:BOOL; //marcha en manual
	CmdR_PE_H_VF1	:BOOL; //seleccion reversa en manual
	StMarcha_PE_H_VF1 :BOOL; //confirmacion motor en marcha
	StAlarma_PE_H_VF1 :BOOL;
	StVeloc_PE_H_VF1 :INT;	
	//Perifericos Elevador 3
	CmdM_PE_H_VF2	:BOOL; //marcha en manual
	CmdR_PE_H_VF2	:BOOL; //seleccion reversa en manual
	StMarcha_PE_H_VF2 :BOOL; //confirmacion motor en marcha
	StAlarma_PE_H_VF2 :BOOL;
	StVeloc_PE_H_VF2 :INT;	
	
	//valvula intermedia 1 embolse
	PE_B1_V1_Cmd_Man_Pos1:BOOL;// descargando
	PE_B1_V1_Cmd_Man_Pos2:BOOL;// no descarga
	PE_B1_V1_Alr:BOOL;
	PE_B1_V1_Alr_discr:BOOL;
	PE_B1_V1_Estado:INT;
	PE_B1_V1_RsAlr:BOOL;
	//valvula intermedia 12 embolse
	PE_B2_V1_Cmd_Man_Pos1:BOOL;// descargando
	PE_B2_V1_Cmd_Man_Pos2:BOOL;// no descarga
	PE_B2_V1_Alr:BOOL;
	PE_B2_V1_Alr_discr:BOOL;
	PE_B2_V1_Estado:INT;
	PE_B2_V1_RsAlr:BOOL;
	//valvula intermedia 3 embolse
	PE_B3_V1_Cmd_Man_Pos1:BOOL;// descargando
	PE_B3_V1_Cmd_Man_Pos2:BOOL;// no descarga
	PE_B3_V1_Alr:BOOL;
	PE_B3_V1_Alr_discr:BOOL;
	PE_B3_V1_Estado:INT;
	PE_B3_V1_RsAlr:BOOL;
	
	PE_B1_V2_Cmd_Man:BOOL;//valvula descarga tolva embolse CE1
	PE_B2_V2_Cmd_Man:BOOL;//valvula descarga tolva embolse CE2
	PE_B3_V2_Cmd_Man:BOOL;//valvula descarga tolva embolse CE3
	PE_B3_V3_Cmd_Man:BOOL;//valvula tolva CE3b	
	TR_S_V6_Cmd_Man	:BOOL;//registro CP 1,8t
	TR_S_V7_Cmd_Man	:BOOL;//registro CP 30t
	TR_S_V8_Cmd_Man	:BOOL;//registro tolva recepción
	
	
	StMarcha_PC1_L5_BD: BOOL;
	Restart: BOOL;
END_VAR
VAR_GLOBAL PERSISTENT
	
	UltimasCalibracoes	:ARRAY[0..12] OF UDINT;	//Array com as ultima calibrações das linhas
	UltimoAlrCalibr		:ARRAY[0..12] OF LINT;	//Esse array é usado para subir o alarme na tela
	//
	SetTmr_Alr_Mot:TIME;
	SetTmr_Alr_Valv:TIME:=T#5S;
	rPesoPatron_TR_S_WT1 :REAL := 198.2;
	bModo_Pausa:BOOL;
	PE_B_SelectorBigBag	:BOOL;
	PE_B_SelectorBolsas	:BOOL;
	bDeshabilitaRecepcion:BOOL;
	bDeshabilita30t		:BOOL;	
	
	SelecionaBigBag1:BOOL;	//Permite descarga no bigbag1
	SelecionaBigBag2:BOOL;	//DESCARGA NO BIGBAG2
	
	CmdV_TR_S_VF1	:REAL; // Homogenizador velocidad manual en % 
	CmdV_TR_S_VF2	:REAL; // Aspersor velocidad manual en % 
	CmdV_PC1_L1_BD	:REAL; //Bomba circuito L1 velocidad manual en % 
	CmdV_PC1_L2_BD	:REAL; // Bomba circuito L2 velocidad manual en % 
	CmdV_PC1_L3_BD	:REAL; //Bomba circuito L3 velocidad manual en % 
	CmdV_PC1_L4_BD	:REAL; //Bomba circuito L4 velocidad manual en % 
	CmdV_PC2_L5_BD	:REAL; //Bomba circuito L5 velocidad manual en % 
	CmdV_PC2_L6_BD	:REAL; //Bomba circuito L6 velocidad manual en % 
	CmdV_PC2_L7_BD	:REAL; //Bomba circuito L7 velocidad manual en % 
	CmdV_PC2_L8_BD	:REAL; //Bomba circuito L8 velocidad manual en % 
	CmdV_PC3_L9_BD	:REAL; //Bomba circuito L9 velocidad manual en % 	
	CmdV_PC3_L10_BD	:REAL; //Bomba circuito L10 velocidad manual en % 
	CmdV_PC3_L11_BD	:REAL; //Bomba circuito L11 velocidad manual en % 
	CmdV_PC3_L12_BD	:REAL; //Bomba circuito L12 velocidad manual en % 
	CmdV_PE_B_VF1	:REAL; //Perifericos Elevador 1 velocidad manual en % 
	CmdV_PE_H_VF1	:REAL; //Perifericos Elevador 2 velocidad manual en % 
	CmdV_PE_H_VF2	:REAL; //Perifericos velocidad manual en % 
	CmdV_TR_P1_VF	:REAL; //Dosificador Polvo 1 velocidad manual en % 
	CmdV_TR_P2_VF	:REAL; //Dosificador Polvo 2 velocidad manual en % 	
	
	CaudalNom_PC1_L1_BD :REAL := 347.22; //Caudal nominal Bomba circuito L1 en ml/s
	CaudalNom_PC1_L2_BD :REAL := 142.28; //Caudal nominal Bomba circuito L2 en ml/s	
	CaudalNom_PC1_L3_BD :REAL := 142.28; //Caudal nominal Bomba circuito L3 en ml/s
	CaudalNom_PC1_L4_BD :REAL := 142.28; //Caudal nominal Bomba circuito L4 en ml/s
	CaudalNom_PC2_L5_BD :REAL := 142.28; //Caudal nominal Bomba circuito L5 en ml/s
	CaudalNom_PC2_L6_BD :REAL := 142.28; //Caudal nominal Bomba circuito L6 en ml/s
	CaudalNom_PC2_L7_BD :REAL := 142.28; //Caudal nominal Bomba circuito L7 en ml/s
	CaudalNom_PC2_L8_BD :REAL := 80.6; //Caudal nominal Bomba circuito L8 en ml/s
	CaudalNom_PC3_L9_BD :REAL := 80.6; //Caudal nominal Bomba circuito L9 en ml/s
	CaudalNom_PC3_L10_BD :REAL := 80.6; //Caudal nominal Bomba circuito L10 en ml/s
	CaudalNom_PC3_L11_BD :REAL := 36.7; //Caudal nominal Bomba circuito L11 en ml/s
	CaudalNom_PC3_L12_BD :REAL := 36.7; //Caudal nominal Bomba circuito L12 en ml/s
	
	//variables carga semilla
	bSet_pesoSemilla:REAL;
	rSet_corteGrueso_semilla:REAL;
	rSet_corteFino_semilla:REAL;
	rTolerancia_pesoSemilla:REAL;
	rBalanzaVacia_TR_S_WT1:REAL;
	tSetTmrMax_carga_TR_S_WT1:TIME;
	tSetTmrMax_descarga_TR_S_WT1:TIME;
	Pesadas :ARRAY [1..10]  OF REAL;
	
	//Demoras parada elevadores
	tDemoraParadaPE_H_VF1 :DINT;
	tDemoraParadaPE_H_VF2 :DINT;	
	tDemoraParadaPE_B_VF1 :DINT;

	PID_L1_Kp:REAL;
	PID_L2_Kp:REAL;
	PID_L3_Kp:REAL;
	PID_L4_Kp:REAL;	
	PID_L5_Kp:REAL;
	PID_L6_Kp:REAL;
	PID_L7_Kp:REAL;
	PID_L8_Kp:REAL;	
	PID_L9_Kp:REAL;
	PID_L10_Kp:REAL;
	PID_L11_Kp:REAL;
	PID_L12_Kp:REAL;	
	PID_L1_Ti:REAL;
	PID_L2_Ti:REAL;	
	PID_L3_Ti:REAL;
	PID_L4_Ti:REAL;
	PID_L5_Ti:REAL;
	PID_L6_Ti:REAL;	
	PID_L7_Ti:REAL;
	PID_L8_Ti:REAL;
	PID_L9_Ti:REAL;
	PID_L10_Ti:REAL;	
	PID_L11_Ti:REAL;
	PID_L12_Ti:REAL;	
	PID_L1_bMuerta:REAL;
	PID_L2_bMuerta:REAL;	
	PID_L3_bMuerta:REAL;
	PID_L4_bMuerta:REAL;	
	PID_L5_bMuerta:REAL;
	PID_L6_bMuerta:REAL;	
	PID_L7_bMuerta:REAL;
	PID_L8_bMuerta:REAL;	
	PID_L9_bMuerta:REAL;
	PID_L10_bMuerta:REAL;	
	PID_L11_bMuerta:REAL;
	PID_L12_bMuerta:REAL;
END_VAR

// ---- GVLs/HMICA1.TcGVL
{attribute 'qualified_only'}
VAR_GLOBAL
	Inicio_calibracion			:BOOL;
	Pausa_calibracion			:BOOL;
	VaciarProbeta_calibracion	:BOOL;//probeta llena	
	Fin_calibracion				:BOOL;
	Error_promedio				:REAL;
	Continuar_calibracion		:BOOL;
	Volumen_calibracion			:ARRAY[1..3]OF REAL;
	Tiempo_calibracion			:ARRAY[1..3]OF DINT;
	Peso_calibracion			:REAL;
	Dosis_calibracion			:REAL;
	VolumenPedido_calibracion	:REAL;
	Tolerancia_calibracion		:REAL;
	TInyeccion_calibracion		:DINT;
	VolMaxProbeta_calibracion	:REAL;
	Vol_enProbeta				:REAL;
	TiempoInyectado				:DINT;
END_VAR

// ---- GVLs/HMICA2.TcGVL
{attribute 'qualified_only'}
VAR_GLOBAL	
	Inicio_calibracion			:BOOL;
	Pausa_calibracion			:BOOL;
	VaciarProbeta_calibracion	:BOOL;//probeta llena	
	Fin_calibracion				:BOOL;
	Error_promedio				:REAL;
	Continuar_calibracion		:BOOL;
	Volumen_calibracion			:ARRAY[1..3]OF REAL;
	Tiempo_calibracion			:ARRAY[1..3]OF DINT;
	Peso_calibracion			:REAL;
	Dosis_calibracion			:REAL;
	VolumenPedido_calibracion	:REAL;
	Tolerancia_calibracion		:REAL;
	TInyeccion_calibracion		:DINT;
	VolMaxProbeta_calibracion	:REAL;
	Vol_enProbeta				:REAL;
	TiempoInyectado				:DINT;
END_VAR

// ---- GVLs/HMICA3.TcGVL
{attribute 'qualified_only'}
VAR_GLOBAL
	Inicio_calibracion			:BOOL;
	Pausa_calibracion			:BOOL;
	VaciarProbeta_calibracion	:BOOL;//probeta llena	
	Fin_calibracion				:BOOL;
	Error_promedio				:REAL;
	Continuar_calibracion		:BOOL;
	Volumen_calibracion			:ARRAY[1..3]OF REAL;
	Tiempo_calibracion			:ARRAY[1..3]OF DINT;
	Peso_calibracion			:REAL;
	Dosis_calibracion			:REAL;
	VolumenPedido_calibracion	:REAL;
	Tolerancia_calibracion		:REAL;
	TInyeccion_calibracion		:DINT;
	VolMaxProbeta_calibracion	:REAL;
	Vol_enProbeta				:REAL;
	TiempoInyectado				:DINT;
END_VAR

// ---- GVLs/HMIcalP1.TcGVL
{attribute 'qualified_only'}
VAR_GLOBAL
	Inicio:BOOL;
	PesoMaxConte:REAL;
	Dosis:REAL;
	Tinyeccion:DINT;
	PesoBatch:REAL;
	Tolerancia:REAL;
	Pausa:BOOL;		
	Error:REAL;
	ContLleno:BOOL;	
	CantPesadas:INT;
	PesoCalibracion:REAL;
	Muestra1_Ok:BOOL;
	Finalizado:BOOL;
	PesoPromedio6:REAL;
	
END_VAR

// ---- GVLs/HMIcalP2.TcGVL
{attribute 'qualified_only'}
VAR_GLOBAL
	Inicio:BOOL;
	PesoMaxConte:REAL;
	Dosis:REAL;
	Tinyeccion:DINT;
	PesoBatch:REAL;
	Tolerancia:REAL;
	Pausa:BOOL;		
	Error:REAL;
	ContLleno:BOOL;	
	CantPesadas:INT;
	PesoCalibracion:REAL;
	Muestra1_Ok:BOOL;
	Finalizado:BOOL;
	PesoPromedio6:REAL;
	
END_VAR

// ---- GVLs/ioLink.TcGVL
{attribute 'qualified_only'}
VAR_GLOBAL
		
	//Valvulas ioLink PC1
	//St1  	posicion angular (-1800 To 1799) * 0.1 grados
	//St2	bit0=open..bit1=close..bit2=seat..bit3=n/a..bit4..7(Byte)= 0=Ok 1=Mant  2=fuera especificacion  3=funcion chequeo  4=falla
	b0St1_CA1_L1_V1 AT%I*	:BYTE;			//
	b1St1_CA1_L1_V1 AT%I*	:BYTE;			//
	b2St1_CA1_L1_V1 AT%I*	:BYTE;			//
	b3St1_CA1_L1_V1 AT%I*	:BYTE;			//
	b0Cmd_CA1_L1_V1 AT%Q*	:BYTE;
	b0St1_CA1_L2_V1 AT%I*	:BYTE;			//
	b1St1_CA1_L2_V1 AT%I*	:BYTE;			//
	b2St1_CA1_L2_V1 AT%I*	:BYTE;			//
	b3St1_CA1_L2_V1 AT%I*	:BYTE;			//
	b0Cmd_CA1_L2_V1 AT%Q*	:BYTE;
	b0St1_CA1_L3_V1 AT%I*	:BYTE;			//
	b1St1_CA1_L3_V1 AT%I*	:BYTE;			//
	b2St1_CA1_L3_V1 AT%I*	:BYTE;			//
	b3St1_CA1_L3_V1 AT%I*	:BYTE;			//
	b0Cmd_CA1_L3_V1 AT%Q*	:BYTE;
	b0St1_CA1_L4_V1 AT%I*	:BYTE;			//
	b1St1_CA1_L4_V1 AT%I*	:BYTE;			//
	b2St1_CA1_L4_V1 AT%I*	:BYTE;			//
	b3St1_CA1_L4_V1 AT%I*	:BYTE;			//
	b0Cmd_CA1_L4_V1 AT%Q*	:BYTE;
	b0St1_CA2_L5_V1 AT%I*	:BYTE;			//
	b1St1_CA2_L5_V1 AT%I*	:BYTE;			//
	b2St1_CA2_L5_V1 AT%I*	:BYTE;			//
	b3St1_CA2_L5_V1 AT%I*	:BYTE;			//
	b0Cmd_CA2_L5_V1 AT%Q*	:BYTE;
	b0St1_CA2_L6_V1 AT%I*	:BYTE;			//
	b1St1_CA2_L6_V1 AT%I*	:BYTE;			//
	b2St1_CA2_L6_V1 AT%I*	:BYTE;			//
	b3St1_CA2_L6_V1 AT%I*	:BYTE;			//
	b0Cmd_CA2_L6_V1 AT%Q*	:BYTE;
	b0St1_CA2_L7_V1 AT%I*	:BYTE;			//
	b1St1_CA2_L7_V1 AT%I*	:BYTE;			//
	b2St1_CA2_L7_V1 AT%I*	:BYTE;			//
	b3St1_CA2_L7_V1 AT%I*	:BYTE;			//
	b0Cmd_CA2_L7_V1 AT%Q*	:BYTE;
	b0St1_CA2_L8_V1 AT%I*	:BYTE;			//
	b1St1_CA2_L8_V1 AT%I*	:BYTE;			//
	b2St1_CA2_L8_V1 AT%I*	:BYTE;			//
	b3St1_CA2_L8_V1 AT%I*	:BYTE;			//
	b0Cmd_CA2_L8_V1 AT%Q*	:BYTE;
	b0St1_CA3_L9_V1 AT%I*	:BYTE;			//
	b1St1_CA3_L9_V1 AT%I*	:BYTE;			//
	b2St1_CA3_L9_V1 AT%I*	:BYTE;			//
	b3St1_CA3_L9_V1 AT%I*	:BYTE;			//
	b0Cmd_CA3_L9_V1 AT%Q*	:BYTE;
	b0St1_CA3_L10_V1 AT%I*	:BYTE;			//
	b1St1_CA3_L10_V1 AT%I*	:BYTE;			//
	b2St1_CA3_L10_V1 AT%I*	:BYTE;			//
	b3St1_CA3_L10_V1 AT%I*	:BYTE;			//
	b0Cmd_CA3_L10_V1 AT%Q*	:BYTE;
	b0St1_CA3_L11_V1 AT%I*	:BYTE;			//
	b1St1_CA3_L11_V1 AT%I*	:BYTE;			//
	b2St1_CA3_L11_V1 AT%I*	:BYTE;			//
	b3St1_CA3_L11_V1 AT%I*	:BYTE;			//
	b0Cmd_CA3_L11_V1 AT%Q*	:BYTE;
	b0St1_CA3_L12_V1 AT%I*	:BYTE;			//
	b1St1_CA3_L12_V1 AT%I*	:BYTE;			//
	b2St1_CA3_L12_V1 AT%I*	:BYTE;			//
	b3St1_CA3_L12_V1 AT%I*	:BYTE;			//
	b0Cmd_CA3_L12_V1 AT%Q*	:BYTE;		
	
	b0St1_CA1_L1_V2 AT%I*	:BYTE;			//
	b1St1_CA1_L1_V2 AT%I*	:BYTE;			//
	b2St1_CA1_L1_V2 AT%I*	:BYTE;			//
	b3St1_CA1_L1_V2 AT%I*	:BYTE;			//
	b0Cmd_CA1_L1_V2 AT%Q*	:BYTE;
	b0St1_CA1_L1_V3 AT%I*	:BYTE;			//
	b1St1_CA1_L1_V3 AT%I*	:BYTE;			//
	b2St1_CA1_L1_V3 AT%I*	:BYTE;			//
	b3St1_CA1_L1_V3 AT%I*	:BYTE;			//
	b0Cmd_CA1_L1_V3 AT%Q*	:BYTE;
	b0St1_CA1_L1_V4 AT%I*	:BYTE;			//
	b1St1_CA1_L1_V4 AT%I*	:BYTE;			//
	b2St1_CA1_L1_V4 AT%I*	:BYTE;			//
	b3St1_CA1_L1_V4 AT%I*	:BYTE;			//
	b0Cmd_CA1_L1_V4 AT%Q*	:BYTE;
	b0St1_CA1_L2_V2 AT%I*	:BYTE;			//
	b1St1_CA1_L2_V2 AT%I*	:BYTE;			//
	b2St1_CA1_L2_V2 AT%I*	:BYTE;			//
	b3St1_CA1_L2_V2 AT%I*	:BYTE;			//
	b0Cmd_CA1_L2_V2 AT%Q*	:BYTE;
	b0St1_CA1_L2_V3 AT%I*	:BYTE;			//
	b1St1_CA1_L2_V3 AT%I*	:BYTE;			//
	b2St1_CA1_L2_V3 AT%I*	:BYTE;			//
	b3St1_CA1_L2_V3 AT%I*	:BYTE;			//
	b0Cmd_CA1_L2_V3 AT%Q*	:BYTE;
	b0St1_CA1_L2_V4 AT%I*	:BYTE;			//
	b1St1_CA1_L2_V4 AT%I*	:BYTE;			//
	b2St1_CA1_L2_V4 AT%I*	:BYTE;			//
	b3St1_CA1_L2_V4 AT%I*	:BYTE;			//
	b0Cmd_CA1_L2_V4 AT%Q*	:BYTE;
	b0St1_CA1_L3_V2 AT%I*	:BYTE;			//
	b1St1_CA1_L3_V2 AT%I*	:BYTE;			//
	b2St1_CA1_L3_V2 AT%I*	:BYTE;			//
	b3St1_CA1_L3_V2 AT%I*	:BYTE;			//
	b0Cmd_CA1_L3_V2 AT%Q*	:BYTE;
	b0St1_CA1_L3_V3 AT%I*	:BYTE;			//
	b1St1_CA1_L3_V3 AT%I*	:BYTE;			//
	b2St1_CA1_L3_V3 AT%I*	:BYTE;			//
	b3St1_CA1_L3_V3 AT%I*	:BYTE;			//
	b0Cmd_CA1_L3_V3 AT%Q*	:BYTE;
	b0St1_CA1_L3_V4 AT%I*	:BYTE;			//
	b1St1_CA1_L3_V4 AT%I*	:BYTE;			//
	b2St1_CA1_L3_V4 AT%I*	:BYTE;			//
	b3St1_CA1_L3_V4 AT%I*	:BYTE;			//
	b0Cmd_CA1_L3_V4 AT%Q*	:BYTE;
	b0St1_CA1_L4_V2 AT%I*	:BYTE;			//
	b1St1_CA1_L4_V2 AT%I*	:BYTE;			//
	b2St1_CA1_L4_V2 AT%I*	:BYTE;			//
	b3St1_CA1_L4_V2 AT%I*	:BYTE;			//
	b0Cmd_CA1_L4_V2 AT%Q*	:BYTE;
	b0St1_CA1_L4_V3 AT%I*	:BYTE;			//
	b1St1_CA1_L4_V3 AT%I*	:BYTE;			//
	b2St1_CA1_L4_V3 AT%I*	:BYTE;			//
	b3St1_CA1_L4_V3 AT%I*	:BYTE;			//
	b0Cmd_CA1_L4_V3 AT%Q*	:BYTE;
	b0St1_CA1_L4_V4 AT%I*	:BYTE;			//
	b1St1_CA1_L4_V4 AT%I*	:BYTE;			//
	b2St1_CA1_L4_V4 AT%I*	:BYTE;			//
	b3St1_CA1_L4_V4 AT%I*	:BYTE;			//
	b0Cmd_CA1_L4_V4 AT%Q*	:BYTE;
	b1St1_CA2_L5_V2 AT%I*	:BYTE;			//
	b2St1_CA2_L5_V2 AT%I*	:BYTE;			//
	b3St1_CA2_L5_V2 AT%I*	:BYTE;			//
	b0Cmd_CA2_L5_V2 AT%Q*	:BYTE;
	b0St1_CA2_L5_V3 AT%I*	:BYTE;			//
	b1St1_CA2_L5_V3 AT%I*	:BYTE;			//
	b2St1_CA2_L5_V3 AT%I*	:BYTE;			//
	b3St1_CA2_L5_V3 AT%I*	:BYTE;			//
	b0Cmd_CA2_L5_V3 AT%Q*	:BYTE;
	b0St1_CA2_L5_V4 AT%I*	:BYTE;			//
	b1St1_CA2_L5_V4 AT%I*	:BYTE;			//
	b2St1_CA2_L5_V4 AT%I*	:BYTE;			//
	b3St1_CA2_L5_V4 AT%I*	:BYTE;			//
	b0Cmd_CA2_L5_V4 AT%Q*	:BYTE;
	b1St1_CA2_L6_V2 AT%I*	:BYTE;			//
	b2St1_CA2_L6_V2 AT%I*	:BYTE;			//
	b3St1_CA2_L6_V2 AT%I*	:BYTE;			//
	b0Cmd_CA2_L6_V2 AT%Q*	:BYTE;
	b0St1_CA2_L6_V3 AT%I*	:BYTE;			//
	b1St1_CA2_L6_V3 AT%I*	:BYTE;			//
	b2St1_CA2_L6_V3 AT%I*	:BYTE;			//
	b3St1_CA2_L6_V3 AT%I*	:BYTE;			//
	b0Cmd_CA2_L6_V3 AT%Q*	:BYTE;
	b0St1_CA2_L6_V4 AT%I*	:BYTE;			//
	b1St1_CA2_L6_V4 AT%I*	:BYTE;			//
	b2St1_CA2_L6_V4 AT%I*	:BYTE;			//
	b3St1_CA2_L6_V4 AT%I*	:BYTE;			//
	b0Cmd_CA2_L6_V4 AT%Q*	:BYTE;
	b1St1_CA2_L7_V2 AT%I*	:BYTE;			//
	b2St1_CA2_L7_V2 AT%I*	:BYTE;			//
	b3St1_CA2_L7_V2 AT%I*	:BYTE;			//
	b0Cmd_CA2_L7_V2 AT%Q*	:BYTE;
	b0St1_CA2_L7_V3 AT%I*	:BYTE;			//
	b1St1_CA2_L7_V3 AT%I*	:BYTE;			//
	b2St1_CA2_L7_V3 AT%I*	:BYTE;			//
	b3St1_CA2_L7_V3 AT%I*	:BYTE;			//
	b0Cmd_CA2_L7_V3 AT%Q*	:BYTE;
	b0St1_CA2_L7_V4 AT%I*	:BYTE;			//
	b1St1_CA2_L7_V4 AT%I*	:BYTE;			//
	b2St1_CA2_L7_V4 AT%I*	:BYTE;			//
	b3St1_CA2_L7_V4 AT%I*	:BYTE;			//
	b0Cmd_CA2_L7_V4 AT%Q*	:BYTE;
	b1St1_CA2_L8_V2 AT%I*	:BYTE;			//
	b2St1_CA2_L8_V2 AT%I*	:BYTE;			//
	b3St1_CA2_L8_V2 AT%I*	:BYTE;			//
	b0Cmd_CA2_L8_V2 AT%Q*	:BYTE;
	b0St1_CA2_L8_V3 AT%I*	:BYTE;			//
	b1St1_CA2_L8_V3 AT%I*	:BYTE;			//
	b2St1_CA2_L8_V3 AT%I*	:BYTE;			//
	b3St1_CA2_L8_V3 AT%I*	:BYTE;			//
	b0Cmd_CA2_L8_V3 AT%Q*	:BYTE;
	b0St1_CA2_L8_V4 AT%I*	:BYTE;			//
	b1St1_CA2_L8_V4 AT%I*	:BYTE;			//
	b2St1_CA2_L8_V4 AT%I*	:BYTE;			//
	b3St1_CA2_L8_V4 AT%I*	:BYTE;			//
	b0Cmd_CA2_L8_V4 AT%Q*	:BYTE;
	b1St1_CA3_L9_V2 AT%I*	:BYTE;			//
	b2St1_CA3_L9_V2 AT%I*	:BYTE;			//
	b3St1_CA3_L9_V2 AT%I*	:BYTE;			//
	b0Cmd_CA3_L9_V2 AT%Q*	:BYTE;
	b0St1_CA3_L9_V3 AT%I*	:BYTE;			//
	b1St1_CA3_L9_V3 AT%I*	:BYTE;			//
	b2St1_CA3_L9_V3 AT%I*	:BYTE;			//
	b3St1_CA3_L9_V3 AT%I*	:BYTE;			//
	b0Cmd_CA3_L9_V3 AT%Q*	:BYTE;
	b0St1_CA3_L9_V4 AT%I*	:BYTE;			//
	b1St1_CA3_L9_V4 AT%I*	:BYTE;			//
	b2St1_CA3_L9_V4 AT%I*	:BYTE;			//
	b3St1_CA3_L9_V4 AT%I*	:BYTE;			//
	b0Cmd_CA3_L9_V4 AT%Q*	:BYTE;
	b1St1_CA3_L10_V2 AT%I*	:BYTE;			//
	b2St1_CA3_L10_V2 AT%I*	:BYTE;			//
	b3St1_CA3_L10_V2 AT%I*	:BYTE;			//
	b0Cmd_CA3_L10_V2 AT%Q*	:BYTE;
	b0St1_CA3_L10_V3 AT%I*	:BYTE;			//
	b1St1_CA3_L10_V3 AT%I*	:BYTE;			//
	b2St1_CA3_L10_V3 AT%I*	:BYTE;			//
	b3St1_CA3_L10_V3 AT%I*	:BYTE;			//
	b0Cmd_CA3_L10_V3 AT%Q*	:BYTE;
	b0St1_CA3_L10_V4 AT%I*	:BYTE;			//
	b1St1_CA3_L10_V4 AT%I*	:BYTE;			//
	b2St1_CA3_L10_V4 AT%I*	:BYTE;			//
	b3St1_CA3_L10_V4 AT%I*	:BYTE;			//
	b0Cmd_CA3_L10_V4 AT%Q*	:BYTE;
	b1St1_CA3_L11_V2 AT%I*	:BYTE;			//
	b2St1_CA3_L11_V2 AT%I*	:BYTE;			//
	b3St1_CA3_L11_V2 AT%I*	:BYTE;			//
	b0Cmd_CA3_L11_V2 AT%Q*	:BYTE;
	b0St1_CA3_L11_V3 AT%I*	:BYTE;			//
	b1St1_CA3_L11_V3 AT%I*	:BYTE;			//
	b2St1_CA3_L11_V3 AT%I*	:BYTE;			//
	b3St1_CA3_L11_V3 AT%I*	:BYTE;			//
	b0Cmd_CA3_L11_V3 AT%Q*	:BYTE;
	b0St1_CA3_L11_V4 AT%I*	:BYTE;			//
	b1St1_CA3_L11_V4 AT%I*	:BYTE;			//
	b2St1_CA3_L11_V4 AT%I*	:BYTE;			//
	b3St1_CA3_L11_V4 AT%I*	:BYTE;			//
	b0Cmd_CA3_L11_V4 AT%Q*	:BYTE;
	b1St1_CA3_L12_V2 AT%I*	:BYTE;			//
	b2St1_CA3_L12_V2 AT%I*	:BYTE;			//
	b3St1_CA3_L12_V2 AT%I*	:BYTE;			//
	b0Cmd_CA3_L12_V2 AT%Q*	:BYTE;
	b0St1_CA3_L12_V3 AT%I*	:BYTE;			//
	b1St1_CA3_L12_V3 AT%I*	:BYTE;			//
	b2St1_CA3_L12_V3 AT%I*	:BYTE;			//
	b3St1_CA3_L12_V3 AT%I*	:BYTE;			//
	b0Cmd_CA3_L12_V3 AT%Q*	:BYTE;
	b0St1_CA3_L12_V4 AT%I*	:BYTE;			//
	b1St1_CA3_L12_V4 AT%I*	:BYTE;			//
	b2St1_CA3_L12_V4 AT%I*	:BYTE;			//
	b3St1_CA3_L12_V4 AT%I*	:BYTE;			//
	b0Cmd_CA3_L12_V4 AT%Q*	:BYTE;		
	//Valvula agua limpia
	b0St1_PU_Lav_V6  AT%I*	:BYTE;
	b1St1_PU_Lav_V6  AT%I*	:BYTE;	
	b2St1_PU_Lav_V6  AT%I*	:BYTE;
	b3St1_PU_Lav_V6  AT%I*	:BYTE;
	b0Cmd_PU_Lav_V6  AT%Q*	:BYTE;
	//Valvula agua residual
	b0St1_PU_Lav_V5  AT%I*	:BYTE;
	b1St1_PU_Lav_V5  AT%I*	:BYTE;	
	b2St1_PU_Lav_V5  AT%I*	:BYTE;
	b3St1_PU_Lav_V5  AT%I*	:BYTE;
	b0Cmd_PU_Lav_V5  AT%Q*	:BYTE;	
	
	
	wSt1_PC1_V10:WORD;			//
	wSt2_PC1_V10:WORD;			
	wSt1_PC1_V20:WORD;			//
	wSt2_PC1_V20:WORD;	


		
END_VAR

// ---- GVLs/Liquidos.TcGVL
{attribute 'qualified_only'}
VAR_GLOBAL
END_VAR

VAR_GLOBAL PERSISTENT
	TablaLiquidos				:ARRAY[1..64]OF stListado_Liquidos;
	Circuito_Liquido			:ARRAY[1..12]OF INT;	//Array que salva o indice do produto que está associado ao liquido
	Circuito_Offset				:ARRAY[1..12]OF REAL;
	InyectarLiq					:ARRAY[1..12]OF BOOL;
	LiqNaReceita				:ARRAY[1..12]OF BOOL; 	//Liquidos que estão sendo usados na receita
	UltimoAlrLavagem			:ARRAY[1..12] OF LINT;	//Hora do ultimo alarme por falta de lavagem
	
END_VAR

// ---- GVLs/Polvos.TcGVL
{attribute 'qualified_only'}
VAR_GLOBAL PERSISTENT
	ProdutoAsociado			:ARRAY[1..4] OF INT;
	TablaPolvos				:ARRAY[1..10]OF stListado_Polvos;
	InyectarPolvo			:ARRAY[1..4]OF BOOL;
END_VAR

// ---- GVLs/RecetasGestion.TcGVL
{attribute 'qualified_only'}
VAR_GLOBAL PERSISTENT
	aComboboxRecipes : ARRAY [1..100] OF stComboBoxRecipes;
	RecetaEditar:RecetaEdicion;
	EdicionRecetaNro:INT;
	GrabarRecetaEdicion:BOOL;
	LeerRecetaEditar:BOOL;
	BibliotecaRecetas:ARRAY [1..100] OF RecetaEdicion;
END_VAR

// ---- GVLs/Receta_Activa.TcGVL
{attribute 'qualified_only'}
VAR_GLOBAL
END_VAR
VAR_GLOBAL PERSISTENT
	//Receita enviada para a máquina
	SetNombreRecetaActiva	:STRING;
	SetTmrHomogenizado		:DINT;
	SetTmrDescarga			:DINT;
	SetVelocHomogenizado	:REAL;// %
	SetVelocDescarga		:REAL;// %
	SetCircuitosLiq			:ARRAY [1..12] OF stReceta_Circuito;
	SetCircuitosPo			:ARRAY [1..4] OF stReceta_Polvo;
	SetTiempoTotal			:REAL;
	SetAspiracao			:BOOL;

	//Interface da receita. Esses variáveis são interligadas com a tela de edição
	//Quando o operador aperta para carregar a receita, as variáveis de interface
	//são enviadas para a máquina
	interfaceSetNombreRecetaActiva	:STRING;	//Nome da receita na interface
	interfaceSetTmrHomogenizado		:DINT;
	interfaceSetTmrDescarga			:DINT;
	interfaceSetVelocHomogenizado	:REAL;// %
	interfaceSetVelocDescarga		:REAL;// %
	interfaceSetCircuitosLiq		:ARRAY [1..12] OF stReceta_Circuito;
	interfaceSetCircuitosPo			:ARRAY [1..4] OF stReceta_Polvo;
	interfaceSetTiempoTotal			:REAL;
	interfaceSetAspiracao			:BOOL;
END_VAR

// ---- GVLs/SafetyInputs.TcGVL
{attribute 'qualified_only'}
VAR_GLOBAL
	//Essa GVL é para os sensores de porta da tratadora
	
	//Entradas da régua TR_2
	TR2_E1_CH01 AT %I*	:BOOL;	//Tampa esquerda da balança
	TR2_E1_CH02 AT %I*	:BOOL;
	TR2_E2_CH01 AT %I*	:BOOL;	//Tampa traseira inferior da balança
	TR2_E2_CH02 AT %I*	:BOOL;
	TR2_E3_CH01 AT %I*	:BOOL;	//Tampa frontal da balança
	TR2_E3_CH02 AT %I*	:BOOL;
	TR2_E4_CH01 AT %I*	:BOOL;	//Tampa frontal inferior da balança
	TR2_E4_CH02 AT %I*	:BOOL;
	
		//Entradas da régua TR_2
	TR3_E1_CH01 AT %I*	:BOOL;	//Tampa direita da balança
	TR3_E1_CH02 AT %I*	:BOOL;
	TR3_E2_CH01 AT %I*	:BOOL;	//Tampa traseira da balança
	TR3_E2_CH02 AT %I*	:BOOL;
	TR3_E3_CH01 AT %I*	:BOOL;	//Tampas do homogeneizador
	TR3_E3_CH02 AT %I*	:BOOL;
	TR3_E4_CH01 AT %I*	:BOOL;	//Tampa da porta de inspeção da descarga
	TR3_E4_CH02 AT %I*	:BOOL;
END_VAR

// ---- GVLs/Salidas.TcGVL
{attribute 'qualified_only'}
VAR_GLOBAL
	
	//Alarmas
	TR_AL1_L AT %Q*:BYTE;
	TR_AL2_L AT %Q*:BYTE;
	TR_AL2_Ac AT %Q*:BYTE;//acustica
	
	//Agitadores
	bPP1_L1_AG_M   AT %Q* :BOOL;
	bPP1_L2_AG_M   AT %Q* :BOOL;
	bPP1_L3_AG_M   AT %Q* :BOOL;
	bPP1_L4_AG_M   AT %Q* :BOOL;
	bPP2_L5_AG_M   AT %Q* :BOOL;
	bPP2_L6_AG_M   AT %Q* :BOOL;
	bPP2_L7_AG_M   AT %Q* :BOOL;
	bPP2_L8_AG_M   AT %Q* :BOOL;	
	bPP3_L9_AG_M   AT %Q* :BOOL;
	bPP3_L10_AG_M   AT %Q* :BOOL;
	bPP3_L11_AG_M   AT %Q* :BOOL;
	bPP3_L12_AG_M   AT %Q* :BOOL;
	
	//Soplador 
	bTR_S_VE1 AT %Q*	:BOOL;
	
	//valvulas tratadora
	TR_S_V1 AT %Q* :BOOL;
	TR_S_V2 AT %Q*:BOOL;
	TR_S_V3 AT %Q*:BOOL;
	TR_S_V4 AT %Q*:BOOL;
	TR_S_V5 AT %Q*:BOOL;	//Pesos de calibração da balança
	
	//TR_S_WT1 semilla
	TR_S_WT1_wControl AT %Q*:WORD;
	
	//Balanza probeta CA1
	CA1_WT1_wControl AT%Q* :WORD;
	//Balanza probeta CA2
	CA2_WT1_wControl AT%Q* :WORD;
	//Balanza probeta CA3
	CA3_WT1_wControl AT%Q* :WORD;
	
	//Balanza IBC L1
	PU1_WT1_wControl AT%Q* :WORD;
	//Balanza IBC L2
	PU1_WT2_wControl AT%Q* :WORD;
	//Balanza IBC L31
	PU1_WT3_wControl AT%Q* :WORD;
	//Balanza IBC L4
	PU1_WT4_wControl AT%Q* :WORD;
	//Balanza IBC L5
	PU2_WT5_wControl AT%Q* :WORD;
	//Balanza IBC L6
	PU2_WT6_wControl AT%Q* :WORD;
	//Balanza IBC L7
	PU2_WT7_wControl AT%Q* :WORD;
	//Balanza IBC L8
	PU2_WT8_wControl AT%Q* :WORD;
	//Balanza IBC L9
	PU3_WT9_wControl AT%Q* :WORD;
	//Balanza IBC L10
	PU3_WT10_wControl AT%Q* :WORD;	
	//Balanza IBC L11
	PU3_WT11_wControl AT%Q* :WORD;
	//Balanza IBC L12
	PU3_WT12_wControl AT%Q* :WORD;
	
	//Bomba Circuito 1
	wPP1_L1_BD_Cmd AT%Q* :WORD;
	wPP1_L1_BD_Set AT%Q* :WORD;
	//Bomba Circuito 2
	wPP1_L2_BD_Cmd AT%Q* :WORD;
	wPP1_L2_BD_Set AT%Q* :WORD;
	//Bomba Circuito 3
	wPP1_L3_BD_Cmd AT%Q* :WORD;
	wPP1_L3_BD_Set AT%Q* :WORD;
	//Bomba Circuito 4
	wPP1_L4_BD_Cmd AT%Q* :WORD;
	wPP1_L4_BD_Set AT%Q* :WORD;
	//Bomba Circuito 5
	wPP2_L5_BD_Cmd AT%Q* :WORD;
	wPP2_L5_BD_Set AT%Q* :WORD;
	//Bomba Circuito 6
	wPP2_L6_BD_Cmd AT%Q* :WORD;
	wPP2_L6_BD_Set AT%Q* :WORD;
	//Bomba Circuito 7
	wPP2_L7_BD_Cmd AT%Q* :WORD;
	wPP2_L7_BD_Set AT%Q* :WORD;
	//Bomba Circuito 8
	wPP2_L8_BD_Cmd AT%Q* :WORD;
	wPP2_L8_BD_Set AT%Q* :WORD;
	//Bomba Circuito 9
	wPP3_L9_BD_Cmd AT%Q* :WORD;
	wPP3_L9_BD_Set AT%Q* :WORD;
	//Bomba Circuito 10
	wPP3_L10_BD_Cmd AT%Q* :WORD;
	wPP3_L10_BD_Set AT%Q* :WORD;
	//Bomba Circuito 11
	wPP3_L11_BD_Cmd AT%Q* :WORD;
	wPP3_L11_BD_Set AT%Q* :WORD;
	//Bomba Circuito 12
	wPP3_L12_BD_Cmd AT%Q* :WORD;
	wPP3_L12_BD_Set AT%Q* :WORD;

	//Balanza Polvo P1
	TR_P1_WT1_wControl AT%Q* :WORD;	
	//Balanza Polvo P2
	TR_P2_WT1_wControl AT%Q* :WORD;		
	//Dosificador Polvo 1
	TR_P1_VF_Cmd AT%Q* :WORD;
	TR_P1_VF_Set AT%Q* :WORD;
	// habilita carga de polvo 1
	PE_P1_HC AT %Q* :BOOL;
	//Dosificador Polvo 2
	TR_P2_VF_Cmd AT%Q* :WORD;
	TR_P2_VF_Set AT%Q* :WORD;
	// habilita carga de polvo 2
	PE_P2_HC AT %Q* :BOOL;	
	//Vibrador Polvo 1 
	TR_P1_VI_Cmd AT%Q* :WORD;
	TR_P1_VI_Set AT%Q* :WORD;	
	//Vibrador Polvo 2 
	TR_P2_VI_Cmd AT%Q* :WORD;
	TR_P2_VI_Set AT%Q* :WORD;	
	
	wTR_S_VF1_Cmd AT%Q* :WORD;//homogenizador
	wTR_S_VF1_Set AT%Q* :WORD;//homogenizador

	wTR_S_VF2_Cmd AT%Q* :WORD;//aspersor
	wTR_S_VF2_Set AT%Q* :WORD;//aspersor
	
	//Perifericos Elevador 1
	wPE_B_VF1_Cmd AT%Q* :WORD;	
	wPE_B_VF1_Set AT%Q* :WORD;
	//Perifericos Elevador 2
	wPE_H_VF1_Cmd AT%Q* :WORD;	
	wPE_H_VF1_Set AT%Q* :WORD;
	//Perifericos Elevador 3
	wPE_H_VF2_Cmd AT%Q* :WORD;	
	wPE_H_VF2_Set AT%Q* :WORD;

	PE_B1_V1_Pos1	AT%Q* 	:BOOL;//descargando intermedia 1
	PE_B1_V1_Pos2	AT%Q*	:BOOL;//no descarga intermedia 1
	PE_B2_V1_Pos1	AT%Q* 	:BOOL;//descargando intermedia 2
	PE_B2_V1_Pos2	AT%Q* 	:BOOL;//no descarga intermedia 2
	PE_B3_V1_Pos1	AT%Q*	:BOOL;//descargando intermedia 3
	PE_B3_V1_Pos2	AT%Q*	:BOOL;//no descarga intermedia 3
	PE_B1_V2		AT%Q*	:BOOL;//descarga tolva CE1
	PE_B2_V2		AT%Q* 	:BOOL;//descarga tolva CE2
	PE_B3_V2		AT%Q* 	:BOOL;//descarga tolva CE3a
	PE_B3_V3		AT%Q* 	:BOOL;//descarga tolva CE3b
	
	TR_S_V6			AT%Q* 	:BOOL;//registro CP 1,8t
	TR_S_V7			AT%Q*	:BOOL;//registro CP 30t
	TR_S_V8			AT%Q*	:BOOL;//registro tolva recepción	
	
	TravaHomog		AT%Q*	:BOOL;	//Trava magnética da tampa do homogeneizador
		
END_VAR

// ---- GVLs/Seguridad.TcGVL
{attribute 'qualified_only'}
VAR_GLOBAL
	Run				AT%Q* :BOOL;
	ErrorAck		AT%Q* :BOOL;
	Restart			AT%Q* :BOOL;
	ResetPorta		AT%Q* :BOOL;
	PB_Emergencia	AT%I* :BOOL;	//Fica em TRUE quando a emergência está ok
	ParadaDePorta	AT%I* :BOOL;	//Fica em TRUE quando as portas estão fechadas e foi feito o reset
END_VAR

// ---- POUs/Testes Thiago/Testes.TcGVL
{attribute 'qualified_only'}
VAR_GLOBAL
	EmTeste:BOOL;
	LinhaSelecionada:INT;
	TesteHora:DATE;
	Teste2:DT;
END_VAR

// ---- POUs/MAIN.TcPOU
PROGRAM MAIN
VAR
	HS AT %I*:BOOL;
	DataHoraIHM:DATE_AND_TIME;
	testeString:STRING;
	NomeUsuario:STRING;		//Nome do usuário vindo da IHM
	SerialDaMaquina:STRING;		//Serial da máquina com 16 digitos
	
	//Reloj
	fbTime: FB_LocalSystemTime;
	DataHora	:STRING;
	wHora		:INT;
	wMin		: INT;
	wSec		: INT;


	indice: INT;
	SetLocalTime: NT_SetLocalTime;	//Instância para ajustar a hora
	
	Teste:UDINT;
	Teste2:time;
	Teste3:DT;
	fbSystemTime : GETSYSTEMTIME;
    timeAsFileTime : T_FILETIME;
	
	
	HoraAtual	:DT;	//Hora atual
	udHoraAtual	:UDINT;	//Hora atual em UDINT
	// variavel para testes
	i: INT;
END_VAR

//Serial da máquina
SerialDaMaquina := '9BLSB3002RPR0004';



//Ajusta a data e hora do CLP pela IHM
SetLocalTime(
	NETID:= '127.0.0.1.1.1', 
	TIMESTR:= , 
	START:= , 
	TMOUT:= , 
	BUSY=> , 
	ERR=> , 
	ERRID=> );
IF SetLocalTime.START THEN
	SetLocalTime.START := FALSE;
END_IF

//Essa parte do código é utilizada para auxiliar na verificação da útima vez da calibração/lavagem 
fbSystemTime(
    timeLoDW=>timeAsFileTime.dwLowDateTime,
    timeHiDW=>timeAsFileTime.dwHighDateTime 
);

HoraAtual 	:= FILETIME_TO_DT(timeAsFileTime); 
udHoraAtual	:= DT_TO_UDINT(HoraAtual);

Teste := TIME_TO_UDINT(t#1D);



//'DT#1970-01-01-00:00:00'
SetLocalTime.TIMESTR.wDay		:= STRING_TO_WORD(MID(DT_TO_STRING(DataHoraIHM), 2, 12));
SetLocalTime.TIMESTR.wMonth		:= STRING_TO_WORD(MID(DT_TO_STRING(DataHoraIHM), 2, 9));
SetLocalTime.TIMESTR.wYear		:= STRING_TO_WORD(MID(DT_TO_STRING(DataHoraIHM), 4, 4));
SetLocalTime.TIMESTR.wHour		:= STRING_TO_WORD(MID(DT_TO_STRING(DataHoraIHM - T#3H), 2, 15));
SetLocalTime.TIMESTR.wMinute	:= STRING_TO_WORD(MID(DT_TO_STRING(DataHoraIHM), 2, 18));
SetLocalTime.TIMESTR.wSecond	:= STRING_TO_WORD(MID(DT_TO_STRING(DataHoraIHM), 2, 21));

//Faz a leitura da data e hora
fbTime(
	sNetID:= '' , 
	bEnable:= TRUE, 
	dwCycle:=1 , 
	dwOpt:= , 
	tTimeout:= , 
	bValid=> , 
	systemTime=> , 
	tzID=> );
wHora:=WORD_TO_INT(fbTime.systemTime.wHour);
wMin:=WORD_TO_INT(fbTime.systemTime.wMinute);
wSec:=WORD_TO_INT(fbTime.systemTime.wSecond);


//Data e hora formatada para a IHM
//dd/MM/AAAA, HH:mm
DataHora := CONCAT(
    CONCAT(
        CONCAT(
            CONCAT(
                CONCAT(
                    WORD_TO_STRING(fbTime.systemTime.wDay), '/'
                ),
                WORD_TO_STRING(fbTime.systemTime.wMonth)
            ),
            '/'
        ),
        WORD_TO_STRING(fbTime.systemTime.wYear)
    ),
    CONCAT(
        CONCAT(', ', INT_TO_STRING(wHora)),
        CONCAT(':', INT_TO_STRING(wMin))
    )
);

//Inicializacion de variables
IF HMI.iCircuito_a_calibrar=0 THEN
	HMI.iCircuito_a_calibrar:=1;
END_IF
FOR indice:= 1 TO 12 BY 1 DO
	IF Liquidos.Circuito_Liquido[indice]=0 THEN
		Liquidos.Circuito_Liquido[indice]:=1;
	END_IF
END_FOR

//Verifica se tem alguma linha de pó sem produto definido
FOR indice := 1 TO 4 DO
	IF Polvos.ProdutoAsociado[indice] = 0 THEN
		Polvos.ProdutoAsociado[indice] := 1;
	END_IF
END_FOR


VarPersistentes();
Datos_Variadores();
Datos_Caudalimetros();
Agitadores();
_Seguridad();
Alarmas();
Inicio();
Tratadora();
Balanza_Semilla();
Puesto_CA1();
Circuito_L1();
Circuito_L2();
Circuito_L3();
Circuito_L4();
Puesto_CA2();
Circuito_L5();
Circuito_L6();
Circuito_L7();
Circuito_L8();
Puesto_CA3();
Circuito_L9();
Circuito_L10();
Circuito_L11();
Circuito_L12();
Valvulas_Lavado();
Dosificador_Polvo_1();
Dosificador_Polvo_2();
Carga_Semilla();
Descarga_Semilla();

//Testes
Receitas();
PRG_DE_TESTES();
//BancoDeDados();
AlarmesDaMaquina();
IntervaloLavCalibr();
CalculoConsumo();
ConsumoIBCs();
AquecimentoValvulas();
ConfigBombas();
iPC_Diagnostic();

END_PROGRAM

// ---- POUs/VarPersistentes.TcPOU

 PROGRAM VarPersistentes
VAR
		Datos_persistentes :WritePersistentData;
		StartON:TON;
		IntervalON:TON;
END_VAR
VAR // added by the converter: edge detectors and wires of the graphical bodies
    _rt1 : R_TRIG;
END_VAR

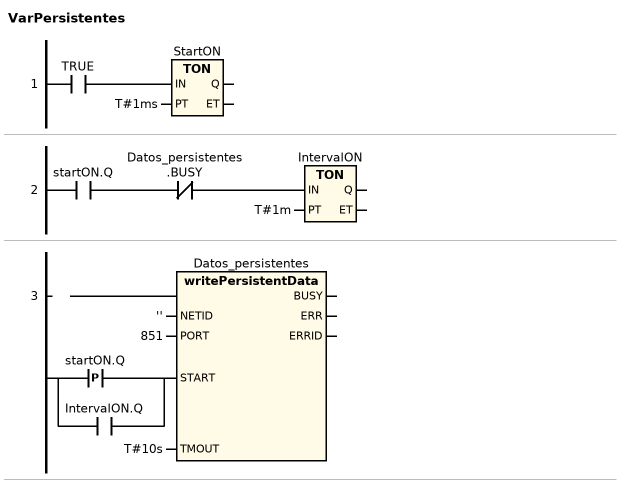
// NETWORK 1
StartON(IN := TRUE, PT := T#1ms); // TON

// NETWORK 2
IntervalON(IN := startON.Q AND NOT Datos_persistentes.BUSY, PT := T#1m); // TON

// NETWORK 3
_rt1(CLK := startON.Q);
Datos_persistentes(NETID := '', PORT := 851, START := _rt1.Q OR IntervalON.Q, TMOUT := T#10s); // writePersistentData

END_PROGRAM

// ---- POUs/Datos_Variadores.TcPOU
PROGRAM Datos_Variadores
VAR
	Variador_6 :SDO_READ;
	ReadStart :BOOL;
	ReadError :DWORD;
	ReadData :ARRAY[0..255] OF BYTE;
	AuxRPM:u_RPM;
	RPM_6 :INT;
END_VAR



Variador_6(

    StartReading := ReadStart,
    CO_Index := 16#2042,
    CO_SubIndex := 16#5,
    DataLength := 2,
    PortNr := 16#1005,
    ADSNetID:='169.254.25.50.3.1'
    );

IF Variador_6.ReadDataAvailable THEN
    ReadStart := FALSE;
    ReadError := Variador_6.Error;
    ReadData := Variador_6.ReadData;
END_IF
AuxRPM.rpm[0]:=ReadData[0];
AuxRPM.rpm[1]:=ReadData[1];
RPM_6 :=AuxRPM.iRpm;

END_PROGRAM

// ---- POUs/CanOpen/SDO_READ.TcPOU
FUNCTION_BLOCK SDO_READ
VAR_INPUT
    ADSNetID:STRING(23); // The AMSNetID addresses the EL6751. Can be empty if only one local single channel card is present

    PortNr:WORD;         //  This Port No. addresses the CANopen Node (see System Manager) 

    CO_Index:DWORD;      //  This is the Index of the CANopen Object Dictionary Entry

    CO_SubIndex:DWORD;   // This is the Sub-Index of the CANopen Object Dictionary Entry

    DataLength:DWORD;    //  This is the Length of the CANopen Object Dictionary Entry

    StartReading:BOOL;   //  only reset to FALSE after ReadDataAvailable=TRUE

END_VAR

VAR_OUTPUT
    ReadData:ARRAY[0..255] OF BYTE;
    ReadDataAvailable:BOOL;
    Error:DWORD;
END_VAR

VAR
    state:BYTE := 0;
    ADSREAD:ADSREAD;
END_VAR

CASE
state OF
    0:
        IF StartReading THEN
           ReadDataAvailable := FALSE;
           Error := 0;
           ADSRead(
               NETID:= ADSNetID,
               PORT:= PortNr,
               IDXGRP:= CO_Index,
               IDXOFFS:= CO_SubIndex,
               LEN:= DataLength,
               DESTADDR:= ADR(ReadData),
               READ:= TRUE,
               TMOUT := T#1s
               );
           IF ADSRead.err THEN
               state := 2;
               ReadDataAvailable := TRUE;
               Error := ADSRead.ErrId;
           ELSE
               state := 1;
           END_IF
        ELSE
           ADSRead(
               NETID:= ADSNetID,
               PORT:= PortNr,
               IDXGRP:= CO_Index,
               IDXOFFS:= CO_SubIndex,
               LEN:= DataLength,
               DESTADDR:= ADR(ReadData),
               READ:= FALSE,
               TMOUT := T#1s
           );
        END_IF
    1:
        ADSRead(READ:= FALSE);
        IF ADSRead.err THEN
           state := 2;
           ReadDataAvailable := TRUE;
           Error := ADSRead.ErrId;
        ELSE
           IF NOT ADSRead.busy THEN
               state := 2;
               ReadDataAvailable := TRUE;
           END_IF
        END_IF
    2:
        ADSRead(READ:= FALSE);
        state := 0;
END_CASE

END_FUNCTION_BLOCK

// ---- POUs/Datos_Caudalimetros.TcPOU
PROGRAM Datos_Caudalimetros
VAR
END_VAR

(*
HMI.CA1_L1_FT1_caudal	:= SEL(TO_REAL(Entradas.CA1_L1_FT1_caudal.icaudal)*16.6667/1000 > 0, 0, TO_REAL(Entradas.CA1_L1_FT1_caudal.icaudal)*16.6667/1000);		// Em L/min 
HMI.CA1_L1_FT1_temp 	:= TO_REAL(Entradas.CA1_L1_FT1_temp.itemp)*0.01; // en grados centigrados
HMI.CA1_L2_FT1_caudal	:= SEL(TO_REAL(Entradas.CA1_L2_FT1_caudal.icaudal)*16.6667/1000 > 0, 0, TO_REAL(Entradas.CA1_L2_FT1_caudal.icaudal)*16.6667/1000);		// Em L/min 
HMI.CA1_L2_FT1_temp		:= TO_REAL(Entradas.CA1_L2_FT1_temp.itemp)*0.01; // en grados centigrados
HMI.CA1_L3_FT1_caudal 	:= SEL(TO_REAL(Entradas.CA1_L3_FT1_caudal.icaudal)*16.6667/1000 > 0, 0, TO_REAL(Entradas.CA1_L3_FT1_caudal.icaudal)*16.6667/1000);		// Em L/min
HMI.CA1_L3_FT1_temp 	:= TO_REAL(Entradas.CA1_L3_FT1_temp.itemp)*0.01; // en grados centigrados
HMI.CA1_L4_FT1_caudal 	:= SEL(TO_REAL(Entradas.CA1_L4_FT1_caudal.icaudal)*16.6667/1000 > 0, 0, TO_REAL(Entradas.CA1_L4_FT1_caudal.icaudal)*16.6667/1000);		// Em L/min
HMI.CA1_L4_FT1_temp 	:= TO_REAL(Entradas.CA1_L4_FT1_temp.itemp)*0.01; // en grados centigrados
HMI.CA2_L5_FT1_caudal 	:= SEL(TO_REAL(Entradas.CA2_L5_FT1_caudal.icaudal)*16.6667/1000 > 0, 0, TO_REAL(Entradas.CA2_L5_FT1_caudal.icaudal)*16.6667/1000);		// Em L/min
HMI.CA2_L5_FT1_temp 	:= TO_REAL(Entradas.CA2_L5_FT1_temp.itemp)*0.01; // en grados centigrados
HMI.CA2_L6_FT1_caudal 	:= SEL(TO_REAL(Entradas.CA2_L6_FT1_caudal.icaudal)*16.6667/1000 > 0, 0, TO_REAL(Entradas.CA2_L6_FT1_caudal.icaudal)*16.6667/1000);		// Em L/min
HMI.CA2_L6_FT1_temp 	:= TO_REAL(Entradas.CA2_L6_FT1_temp.itemp)*0.01; // en grados centigrados
HMI.CA2_L7_FT1_caudal 	:= SEL(TO_REAL(Entradas.CA2_L7_FT1_caudal.icaudal)*16.6667/1000 > 0, 0, TO_REAL(Entradas.CA2_L7_FT1_caudal.icaudal)*16.6667/1000);		// Em L/min
HMI.CA2_L7_FT1_temp 	:= TO_REAL(Entradas.CA2_L7_FT1_temp.itemp)*0.01; // en grados centigrados
HMI.CA2_L8_FT1_caudal 	:= SEL(TO_REAL(Entradas.CA2_L8_FT1_caudal.icaudal)*16.6667/1000 > 0, 0, TO_REAL(Entradas.CA2_L8_FT1_caudal.icaudal)*16.6667/1000);		// Em L/min
HMI.CA2_L8_FT1_temp 	:= TO_REAL(Entradas.CA2_L8_FT1_temp.itemp)*0.01; // en grados centigrados
HMI.CA3_L9_FT1_caudal 	:= SEL(TO_REAL(Entradas.CA3_L9_FT1_caudal.icaudal)*16.6667/1000 > 0, 0, TO_REAL(Entradas.CA3_L9_FT1_caudal.icaudal)*16.6667/1000);		// Em L/min
HMI.CA3_L9_FT1_temp 	:= TO_REAL(Entradas.CA3_L9_FT1_temp.itemp)*0.01; // en grados centigrados
HMI.CA3_L10_FT1_caudal 	:= SEL(TO_REAL(Entradas.CA3_L10_FT1_caudal.icaudal)*16.6667/1000 > 0, 0, TO_REAL(Entradas.CA3_L10_FT1_caudal.icaudal)*16.6667/1000);		// Em L/min
HMI.CA3_L10_FT1_temp 	:= TO_REAL(Entradas.CA3_L10_FT1_temp.itemp)*0.01; // en grados centigrados
HMI.CA3_L11_FT1_caudal 	:= SEL(TO_REAL(Entradas.CA3_L11_FT1_caudal.icaudal)*16.6667/1000 > 0, 0, TO_REAL(Entradas.CA3_L11_FT1_caudal.icaudal)*16.6667/1000);		// Em L/min
HMI.CA3_L11_FT1_temp 	:= TO_REAL(Entradas.CA3_L11_FT1_temp.itemp)*0.01; // en grados centigrados 
HMI.CA3_L12_FT1_caudal 	:= SEL(TO_REAL(Entradas.CA3_L12_FT1_caudal.icaudal)*16.6667/1000 > 0, 0, TO_REAL(Entradas.CA3_L12_FT1_caudal.icaudal)*16.6667/1000);		// Em L/min
HMI.CA3_L12_FT1_temp 	:= TO_REAL(Entradas.CA3_L12_FT1_temp.itemp)*0.01; // en grados centigrados
//
HMI.TR_L1_FT2_caudal	:= SEL(TO_REAL(Entradas.TR_L1_FT2_caudal.icaudal)*16.6667/1000 > 0, 0, TO_REAL(Entradas.TR_L1_FT2_caudal.icaudal)*16.6667/1000); // en ml/s
HMI.TR_L1_FT2_temp 		:= TO_REAL(Entradas.TR_L1_FT2_temp.itemp)*0.01; // en grados centigrados
HMI.TR_L2_FT2_caudal 	:= SEL(TO_REAL(Entradas.TR_L2_FT2_caudal.icaudal)*16.6667/1000 > 0, 0, TO_REAL(Entradas.TR_L2_FT2_caudal.icaudal)*16.6667/1000); // en ml/s
HMI.TR_L2_FT2_temp 		:= TO_REAL(Entradas.TR_L2_FT2_temp.itemp)*0.01; // en grados centigrados
HMI.TR_L3_FT2_caudal 	:= SEL(TO_REAL(Entradas.TR_L3_FT2_caudal.icaudal)*16.6667/1000 > 0, 0, TO_REAL(Entradas.TR_L3_FT2_caudal.icaudal)*16.6667/1000); // en ml/s
HMI.TR_L3_FT2_temp 		:= TO_REAL(Entradas.TR_L3_FT2_temp.itemp)*0.01; // en grados centigrados
HMI.TR_L4_FT2_caudal 	:= SEL(TO_REAL(Entradas.TR_L4_FT2_caudal.icaudal)*16.6667/1000 > 0, 0, TO_REAL(Entradas.TR_L4_FT2_caudal.icaudal)*16.6667/1000); // en ml/s
HMI.TR_L4_FT2_temp 		:= TO_REAL(Entradas.TR_L4_FT2_temp.itemp)*0.01; // en grados centigrados
HMI.TR_L5_FT2_caudal 	:= SEL(TO_REAL(Entradas.TR_L5_FT2_caudal.icaudal)*16.6667/1000 > 0, 0, TO_REAL(Entradas.TR_L5_FT2_caudal.icaudal)*16.6667/1000); // en ml/s
HMI.TR_L5_FT2_temp 		:= TO_REAL(Entradas.TR_L5_FT2_temp.itemp)*0.01; // en grados centigrados
HMI.TR_L6_FT2_caudal 	:= SEL(TO_REAL(Entradas.TR_L6_FT2_caudal.icaudal)*16.6667/1000 > 0, 0, TO_REAL(Entradas.TR_L6_FT2_caudal.icaudal)*16.6667/1000); // en ml/s
HMI.TR_L6_FT2_temp 		:= TO_REAL(Entradas.TR_L6_FT2_temp.itemp)*0.01; // en grados centigrados
HMI.TR_L7_FT2_caudal 	:= SEL(TO_REAL(Entradas.TR_L7_FT2_caudal.icaudal)*16.6667/1000 > 0, 0, TO_REAL(Entradas.TR_L7_FT2_caudal.icaudal)*16.6667/1000); // en ml/s
HMI.TR_L7_FT2_temp 		:= TO_REAL(Entradas.TR_L7_FT2_temp.itemp)*0.01; // en grados centigrados
HMI.TR_L8_FT2_caudal 	:= SEL(TO_REAL(Entradas.TR_L8_FT2_caudal.icaudal)*16.6667/1000 > 0, 0, TO_REAL(Entradas.TR_L8_FT2_caudal.icaudal)*16.6667/1000); // en ml/s
HMI.TR_L8_FT2_temp 		:= TO_REAL(Entradas.TR_L8_FT2_temp.itemp)*0.01; // en grados centigrados
HMI.TR_L9_FT2_caudal 	:= SEL(TO_REAL(Entradas.TR_L9_FT2_caudal.icaudal)*16.6667/1000 > 0, 0, TO_REAL(Entradas.TR_L9_FT2_caudal.icaudal)*16.6667/1000); // en ml/s
HMI.TR_L9_FT2_temp 		:= TO_REAL(Entradas.TR_L9_FT2_temp.itemp)*0.01; // en grados centigrados
HMI.TR_L10_FT2_caudal 	:= SEL(TO_REAL(Entradas.TR_L10_FT2_caudal.icaudal)*16.6667/1000 > 0, 0, TO_REAL(Entradas.TR_L10_FT2_caudal.icaudal)*16.6667/1000); // en ml/s
HMI.TR_L10_FT2_temp 	:= TO_REAL(Entradas.TR_L10_FT2_temp.itemp)*0.01; // en grados centigrados
HMI.TR_L11_FT2_caudal 	:= SEL(TO_REAL(Entradas.TR_L11_FT2_caudal.icaudal)*16.6667/1000 > 0, 0, TO_REAL(Entradas.TR_L11_FT2_caudal.icaudal)*16.6667/1000); // en ml/s
HMI.TR_L11_FT2_temp 	:= TO_REAL(Entradas.TR_L11_FT2_temp.itemp)*0.01; // en grados centigrados
HMI.TR_L12_FT2_caudal 	:= SEL(TO_REAL(Entradas.TR_L12_FT2_caudal.icaudal)*16.6667/1000 > 0, 0, TO_REAL(Entradas.TR_L12_FT2_caudal.icaudal)*16.6667/1000); // en ml/s
HMI.TR_L12_FT2_temp 	:= TO_REAL(Entradas.TR_L12_FT2_temp.itemp)*0.01; // en grados centigrados

*)

{Region "Sensores dos totens"}

//Sensores de vazão doos totens
	HMI.CA1_L1_FT1_caudal	:=TO_REAL(Entradas.CA1_L1_FT1_caudal.icaudal)*0.0166667*16.6667; // en ml/s
	HMI.CA1_L2_FT1_caudal	:=TO_REAL(Entradas.CA1_L2_FT1_caudal.icaudal)*0.0166667*16.6667; // en ml/s
	HMI.CA1_L3_FT1_caudal	:=TO_REAL(Entradas.CA1_L3_FT1_caudal.icaudal)*0.0166667*16.6667; // en ml/s
	HMI.CA1_L4_FT1_caudal 	:=TO_REAL(Entradas.CA1_L4_FT1_caudal.icaudal)*0.0166667*16.6667; // en ml/s
	HMI.CA2_L5_FT1_caudal 	:=TO_REAL(Entradas.CA2_L5_FT1_caudal.icaudal)*0.0166667*16.6667; // en ml/s
	HMI.CA2_L6_FT1_caudal 	:=TO_REAL(Entradas.CA2_L6_FT1_caudal.icaudal)*0.0166667*16.6667; // en ml/s
	HMI.CA2_L7_FT1_caudal 	:=TO_REAL(Entradas.CA2_L7_FT1_caudal.icaudal)*0.0166667*16.6667; // en ml/s
	HMI.CA2_L8_FT1_caudal 	:=TO_REAL(Entradas.CA2_L8_FT1_caudal.icaudal)*0.0166667*16.6667; // en ml/s
	HMI.CA3_L9_FT1_caudal 	:=TO_REAL(Entradas.CA3_L9_FT1_caudal.icaudal)*0.0166667*16.6667; // en ml/s
	HMI.CA3_L10_FT1_caudal 	:=TO_REAL(Entradas.CA3_L10_FT1_caudal.icaudal)*0.0166667*16.6667; // en ml/s
	HMI.CA3_L11_FT1_caudal 	:=TO_REAL(Entradas.CA3_L11_FT1_caudal.icaudal)*0.00166667*16.6667; // en ml/s
	HMI.CA3_L12_FT1_caudal 	:=TO_REAL(Entradas.CA3_L12_FT1_caudal.icaudal)*0.00166667*16.6667; // en ml/s
	
	//Sensores de temperatura dos totens
	HMI.CA1_L1_FT1_temp		:=TO_REAL(Entradas.CA1_L1_FT1_temp.itemp)*0.01; // en grados centigrados
	HMI.CA1_L2_FT1_temp		:=TO_REAL(Entradas.CA1_L2_FT1_temp.itemp)*0.01; // en grados centigrados
	HMI.CA1_L3_FT1_temp 	:=TO_REAL(Entradas.CA1_L3_FT1_temp.itemp)*0.01; // en grados centigrados
	HMI.CA1_L4_FT1_temp 	:=TO_REAL(Entradas.CA1_L4_FT1_temp.itemp)*0.01; // en grados centigrados
	HMI.CA2_L5_FT1_temp 	:=TO_REAL(Entradas.CA2_L5_FT1_temp.itemp)*0.01; // en grados centigrados
	HMI.CA2_L6_FT1_temp 	:=TO_REAL(Entradas.CA2_L6_FT1_temp.itemp)*0.01; // en grados centigrados
	HMI.CA2_L7_FT1_temp 	:=TO_REAL(Entradas.CA2_L7_FT1_temp.itemp)*0.01; // en grados centigrados
	HMI.CA2_L8_FT1_temp 	:=TO_REAL(Entradas.CA2_L8_FT1_temp.itemp)*0.01; // en grados centigrados
	HMI.CA3_L9_FT1_temp 	:=TO_REAL(Entradas.CA3_L9_FT1_temp.itemp)*0.01; // en grados centigrados
	HMI.CA3_L10_FT1_temp 	:=TO_REAL(Entradas.CA3_L10_FT1_temp.itemp)*0.01; // en grados centigrados
	HMI.CA3_L11_FT1_temp 	:=TO_REAL(Entradas.CA3_L11_FT1_temp.itemp)*0.01; // en grados centigrados
	HMI.CA3_L12_FT1_temp 	:=TO_REAL(Entradas.CA3_L12_FT1_temp.itemp)*0.01; // en grados centigrados
{endregion}


{Region "Sensores da tratadora"}

	//Sensores de vazão da tratadora
	HMI.TR_L1_FT2_caudal :=TO_REAL(Entradas.TR_L1_FT2_caudal.icaudal)*0.0166667*16.6667; // en ml/s
	HMI.TR_L2_FT2_caudal :=TO_REAL(Entradas.TR_L2_FT2_caudal.icaudal)*0.0166667*16.6667; // en ml/s
	HMI.TR_L3_FT2_caudal :=TO_REAL(Entradas.TR_L3_FT2_caudal.icaudal)*0.0166667*16.6667; // en ml/s
	HMI.TR_L4_FT2_caudal :=TO_REAL(Entradas.TR_L4_FT2_caudal.icaudal)*0.0166667*16.6667; // en ml/s
	HMI.TR_L5_FT2_caudal :=TO_REAL(Entradas.TR_L5_FT2_caudal.icaudal)*0.0166667*16.6667; // en ml/s
	HMI.TR_L6_FT2_caudal :=TO_REAL(Entradas.TR_L6_FT2_caudal.icaudal)*0.0166667*16.6667; // en ml/s
	HMI.TR_L7_FT2_caudal :=TO_REAL(Entradas.TR_L7_FT2_caudal.icaudal)*0.0166667*16.6667; // en ml/s
	HMI.TR_L8_FT2_caudal :=TO_REAL(Entradas.TR_L8_FT2_caudal.icaudal)*0.0166667*16.6667; // en ml/s
	HMI.TR_L9_FT2_caudal :=TO_REAL(Entradas.TR_L9_FT2_caudal.icaudal)*0.0166667*16.6667; // en ml/s
	HMI.TR_L10_FT2_caudal :=TO_REAL(Entradas.TR_L10_FT2_caudal.icaudal)*0.0166667*16.6667; // en ml/s
	HMI.TR_L11_FT2_caudal :=TO_REAL(Entradas.TR_L11_FT2_caudal.icaudal)*0.00166667*16.6667; // en ml/s
	HMI.TR_L12_FT2_caudal :=TO_REAL(Entradas.TR_L12_FT2_caudal.icaudal)*0.00166667*16.6667; // en ml/s
	
	//Sensores de temperatura da tratadora
	HMI.TR_L1_FT2_temp :=TO_REAL(Entradas.TR_L1_FT2_temp.itemp)*0.01; // en grados centigrados
	HMI.TR_L2_FT2_temp :=TO_REAL(Entradas.TR_L2_FT2_temp.itemp)*0.01; // en grados centigrados
	HMI.TR_L3_FT2_temp :=TO_REAL(Entradas.TR_L3_FT2_temp.itemp)*0.01; // en grados centigrados
	HMI.TR_L4_FT2_temp :=TO_REAL(Entradas.TR_L4_FT2_temp.itemp)*0.01; // en grados centigrados
	HMI.TR_L5_FT2_temp :=TO_REAL(Entradas.TR_L5_FT2_temp.itemp)*0.01; // en grados centigrados
	HMI.TR_L6_FT2_temp :=TO_REAL(Entradas.TR_L6_FT2_temp.itemp)*0.01; // en grados centigrados
	HMI.TR_L7_FT2_temp :=TO_REAL(Entradas.TR_L7_FT2_temp.itemp)*0.01; // en grados centigrados
	HMI.TR_L8_FT2_temp :=TO_REAL(Entradas.TR_L8_FT2_temp.itemp)*0.01; // en grados centigrados
	HMI.TR_L9_FT2_temp :=TO_REAL(Entradas.TR_L9_FT2_temp.itemp)*0.01; // en grados centigrados
	HMI.TR_L10_FT2_temp :=TO_REAL(Entradas.TR_L10_FT2_temp.itemp)*0.01; // en grados centigrados
	HMI.TR_L11_FT2_temp :=TO_REAL(Entradas.TR_L11_FT2_temp.itemp)*0.01; // en grados centigrados
	HMI.TR_L12_FT2_temp :=TO_REAL(Entradas.TR_L12_FT2_temp.itemp)*0.01;  // en grados centigrados

{endregion}

END_PROGRAM

// ---- POUs/Tratadora.TcPOU
PROGRAM Tratadora
VAR
	//Ventilador en tratadora
	TR_S_VE1: Equipo_Motor_No_Rev;
	//
	Eq_TR_sinFalla:BOOL;

	// puerta descarga semilla procesada
	TR_S_V1: Equipo_Valvula_5_2;	//Porta de descarga
	TR_S_V1_CmdAuto:BOOL;	//Comando automático da porta de descarga
	Tmr_PuertaDescarga	:TOF;
	
	fbHomogenizador :Equipo_Motor_ATV320;//Homogenizador
	fbAspersor :Equipo_Motor_ATV320;//Aspersor
	//provisorio
	bHSTR	:BOOL;
	Fin_Dosificado :BOOL;
	
	bHSVE	:BOOL;
	
	Aux_VE:BOOL;
	AbrirDescarga :BOOL;
	
	Tmr_Homogenizado: TON;
	Tiempo_seg_to_TIME_THomog: Tiempo_seg_to_TIME;
	AuxSetTmrPuertaDescarga :TIME;
	AuxSetTmrHomogenizado	:TIME;
	DetenerHomogenizador: BOOL;
	MarchaAutoAspersor: BOOL;
	Dosificar: BOOL;
	PasoDosif: INT;
	VeloAspersorAuto_TR: VeloAspersorAuto;
	TmrDuracionBatch: TON;
	Tiempo_TIME_to_seg_Duracion: Tiempo_TIME_to_seg;
	TBatch:BOOL;
	AuxET_segBatch:DINT;
	CalcPercentual: Percentual;
	TOF_Aspersor: TOF;			//Após a dosagem de produtos, o aspersor fica ligado por 5s 
	TotalizBateladas	:REAL;	//Totalizador dos tempos individuais das bateladas
	TempoBatelada		:REAL; 	//Tempo decorrido da batelada atual
END_VAR
VAR // added by the converter: edge detectors and wires of the graphical bodies
    _w1, _w2, _w3 : BOOL;
    _rt1, _rt2, _rt3 : R_TRIG;
    _ft1 : F_TRIG;
END_VAR

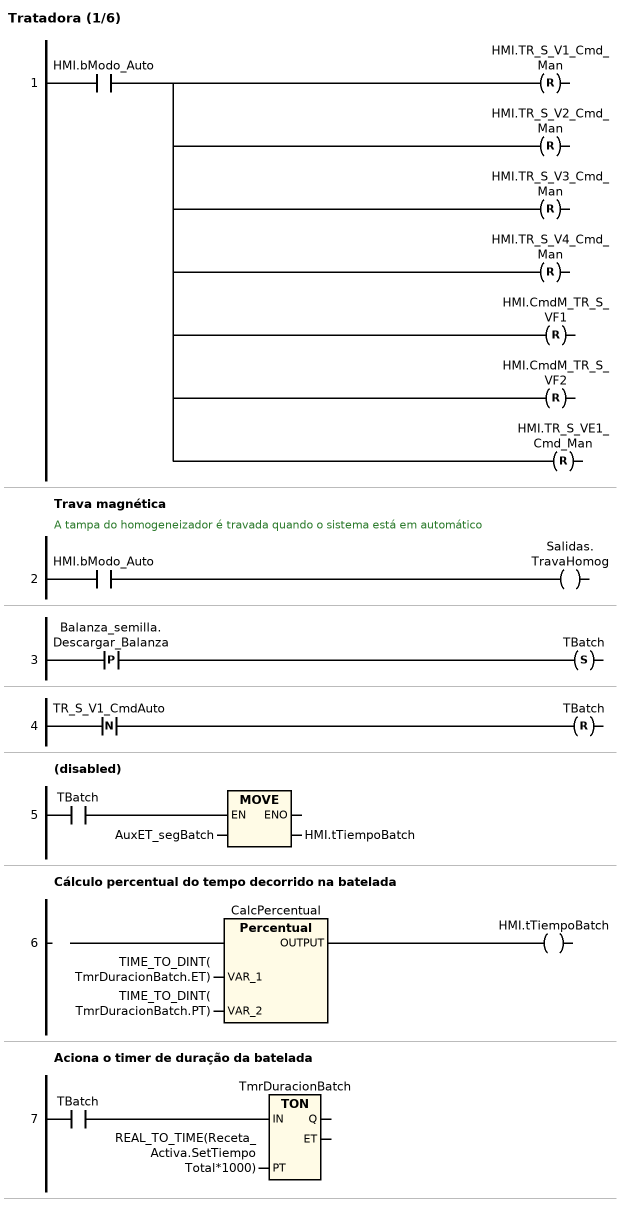
// NETWORK 1
_w1 := HMI.bModo_Auto;
HMI.TR_S_V1_Cmd_Man R= _w1;
HMI.TR_S_V2_Cmd_Man R= _w1;
HMI.TR_S_V3_Cmd_Man R= _w1;
HMI.TR_S_V4_Cmd_Man R= _w1;
HMI.CmdM_TR_S_VF1 R= _w1;
HMI.CmdM_TR_S_VF2 R= _w1;
HMI.TR_S_VE1_Cmd_Man R= _w1;

// NETWORK 2: Trava magnética
// A tampa do homogeneizador é travada quando o sistema está em automático
Salidas.TravaHomog := HMI.bModo_Auto;

// NETWORK 3
_rt1(CLK := Balanza_semilla.Descargar_Balanza);
TBatch S= _rt1.Q;

// NETWORK 4
_ft1(CLK := TR_S_V1_CmdAuto);
TBatch R= _ft1.Q;

// NETWORK 5 (disabled)
// IF TBatch THEN HMI.tTiempoBatch := AuxET_segBatch; END_IF

// NETWORK 6: Cálculo percentual do tempo decorrido na batelada
CalcPercentual(VAR_1 := TIME_TO_DINT(TmrDuracionBatch.ET), VAR_2 := TIME_TO_DINT(TmrDuracionBatch.PT)); // Percentual
HMI.tTiempoBatch := CalcPercentual.OUTPUT;

// NETWORK 7: Aciona o timer de duração da batelada
TmrDuracionBatch(IN := TBatch, PT := REAL_TO_TIME(Receta_Activa.SetTiempoTotal*1000)); // TON

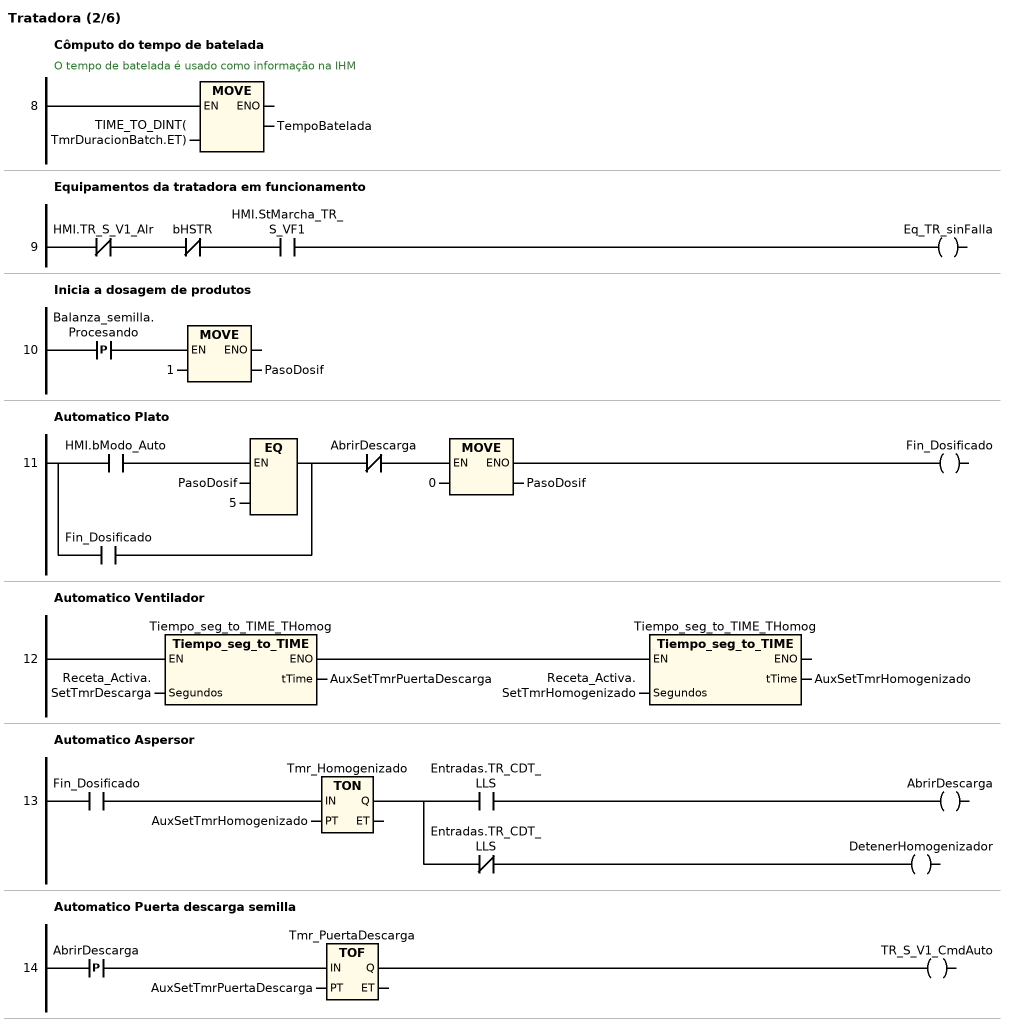
// NETWORK 8: Cômputo do tempo de batelada
// O tempo de batelada é usado como informação na IHM
TempoBatelada := TIME_TO_DINT(TmrDuracionBatch.ET);

// NETWORK 9: Equipamentos da tratadora em funcionamento
Eq_TR_sinFalla := NOT HMI.TR_S_V1_Alr AND NOT bHSTR AND HMI.StMarcha_TR_S_VF1;

// NETWORK 10: Inicia a dosagem de produtos
_rt2(CLK := Balanza_semilla.Procesando);
IF _rt2.Q THEN PasoDosif := 1; END_IF

// NETWORK 11: Automatico Plato
_w2 := (HMI.bModo_Auto AND PasoDosif = 5 OR Fin_Dosificado) AND NOT AbrirDescarga;
IF _w2 THEN PasoDosif := 0; END_IF
Fin_Dosificado := _w2;

// NETWORK 12: Automatico Ventilador
Tiempo_seg_to_TIME_THomog(Segundos := Receta_Activa.SetTmrDescarga, tTime => AuxSetTmrPuertaDescarga); // Tiempo_seg_to_TIME
Tiempo_seg_to_TIME_THomog(Segundos := Receta_Activa.SetTmrHomogenizado, tTime => AuxSetTmrHomogenizado); // Tiempo_seg_to_TIME

// NETWORK 13: Automatico Aspersor
Tmr_Homogenizado(IN := Fin_Dosificado, PT := AuxSetTmrHomogenizado); // TON
AbrirDescarga := Tmr_Homogenizado.Q AND Entradas.TR_CDT_LLS;
DetenerHomogenizador := Tmr_Homogenizado.Q AND NOT Entradas.TR_CDT_LLS;

// NETWORK 14: Automatico Puerta descarga semilla
_rt3(CLK := AbrirDescarga);
Tmr_PuertaDescarga(IN := _rt3.Q, PT := AuxSetTmrPuertaDescarga); // TOF
TR_S_V1_CmdAuto := Tmr_PuertaDescarga.Q;

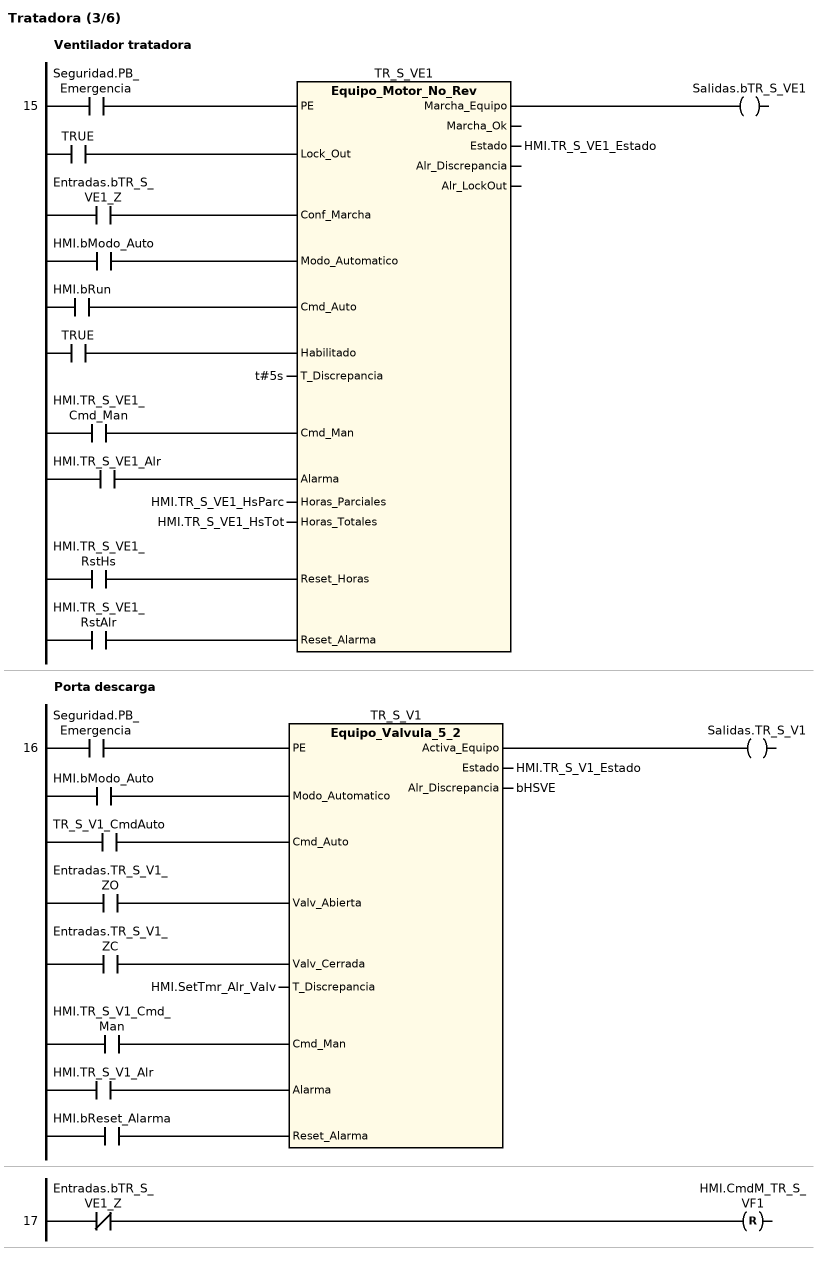
// NETWORK 15: Ventilador tratadora
TR_S_VE1(
    PE := Seguridad.PB_Emergencia,
    Lock_Out := TRUE,
    Conf_Marcha := Entradas.bTR_S_VE1_Z,
    Modo_Automatico := HMI.bModo_Auto,
    Cmd_Auto := HMI.bRun,
    Habilitado := TRUE,
    T_Discrepancia := t#5s,
    Cmd_Man := HMI.TR_S_VE1_Cmd_Man,
    Alarma := HMI.TR_S_VE1_Alr,
    Horas_Parciales := HMI.TR_S_VE1_HsParc,
    Horas_Totales := HMI.TR_S_VE1_HsTot,
    Reset_Horas := HMI.TR_S_VE1_RstHs,
    Reset_Alarma := HMI.TR_S_VE1_RstAlr,
    Estado => HMI.TR_S_VE1_Estado); // Equipo_Motor_No_Rev
Salidas.bTR_S_VE1 := TR_S_VE1.Marcha_Equipo;

// NETWORK 16: Porta descarga
TR_S_V1(
    PE := Seguridad.PB_Emergencia,
    Modo_Automatico := HMI.bModo_Auto,
    Cmd_Auto := TR_S_V1_CmdAuto,
    Valv_Abierta := Entradas.TR_S_V1_ZO,
    Valv_Cerrada := Entradas.TR_S_V1_ZC,
    T_Discrepancia := HMI.SetTmr_Alr_Valv,
    Cmd_Man := HMI.TR_S_V1_Cmd_Man,
    Alarma := HMI.TR_S_V1_Alr,
    Reset_Alarma := HMI.bReset_Alarma,
    Estado => HMI.TR_S_V1_Estado,
    Alr_Discrepancia => bHSVE); // Equipo_Valvula_5_2
Salidas.TR_S_V1 := TR_S_V1.Activa_Equipo;

// NETWORK 17
HMI.CmdM_TR_S_VF1 R= NOT Entradas.bTR_S_VE1_Z;

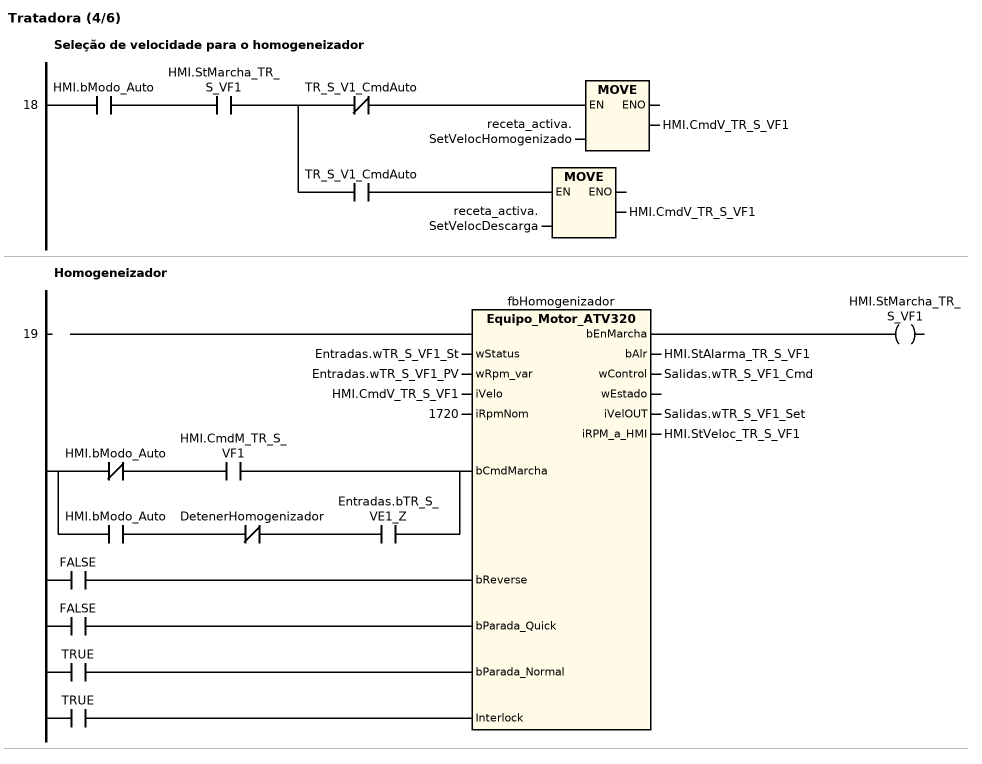
// NETWORK 18: Seleção de velocidade para o homogeneizador
_w3 := HMI.bModo_Auto AND HMI.StMarcha_TR_S_VF1;
IF _w3 AND NOT TR_S_V1_CmdAuto THEN HMI.CmdV_TR_S_VF1 := receta_activa.SetVelocHomogenizado; END_IF
IF _w3 AND TR_S_V1_CmdAuto THEN HMI.CmdV_TR_S_VF1 := receta_activa.SetVelocDescarga; END_IF

// NETWORK 19: Homogeneizador
fbHomogenizador(
    wStatus := Entradas.wTR_S_VF1_St,
    wRpm_var := Entradas.wTR_S_VF1_PV,
    iVelo := HMI.CmdV_TR_S_VF1,
    iRpmNom := 1720,
    bCmdMarcha := NOT HMI.bModo_Auto AND HMI.CmdM_TR_S_VF1 OR HMI.bModo_Auto AND NOT DetenerHomogenizador AND Entradas.bTR_S_VE1_Z,
    bReverse := FALSE,
    bParada_Quick := FALSE,
    bParada_Normal := TRUE,
    Interlock := TRUE,
    bAlr => HMI.StAlarma_TR_S_VF1,
    wControl => Salidas.wTR_S_VF1_Cmd,
    iVelOUT => Salidas.wTR_S_VF1_Set,
    iRPM_a_HMI => HMI.StVeloc_TR_S_VF1); // Equipo_Motor_ATV320
HMI.StMarcha_TR_S_VF1 := fbHomogenizador.bEnMarcha;

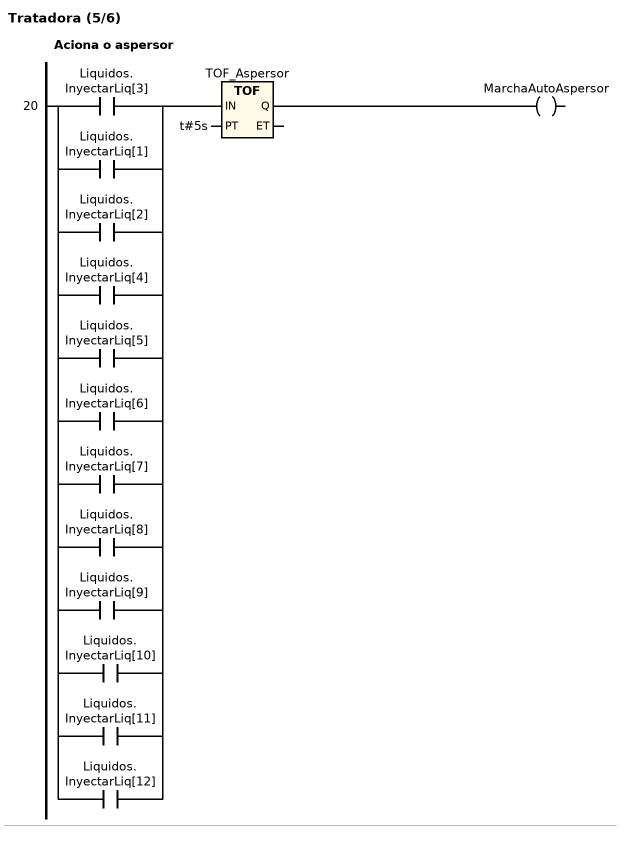
// NETWORK 20: Aciona o aspersor
TOF_Aspersor(IN := Liquidos.InyectarLiq[3] OR Liquidos.InyectarLiq[1] OR Liquidos.InyectarLiq[2] OR Liquidos.InyectarLiq[4] OR Liquidos.InyectarLiq[5] OR Liquidos.InyectarLiq[6] OR Liquidos.InyectarLiq[7] OR Liquidos.InyectarLiq[8] OR Liquidos.InyectarLiq[9] OR Liquidos.InyectarLiq[10] OR Liquidos.InyectarLiq[11] OR Liquidos.InyectarLiq[12], PT := t#5s); // TOF
MarchaAutoAspersor := TOF_Aspersor.Q;

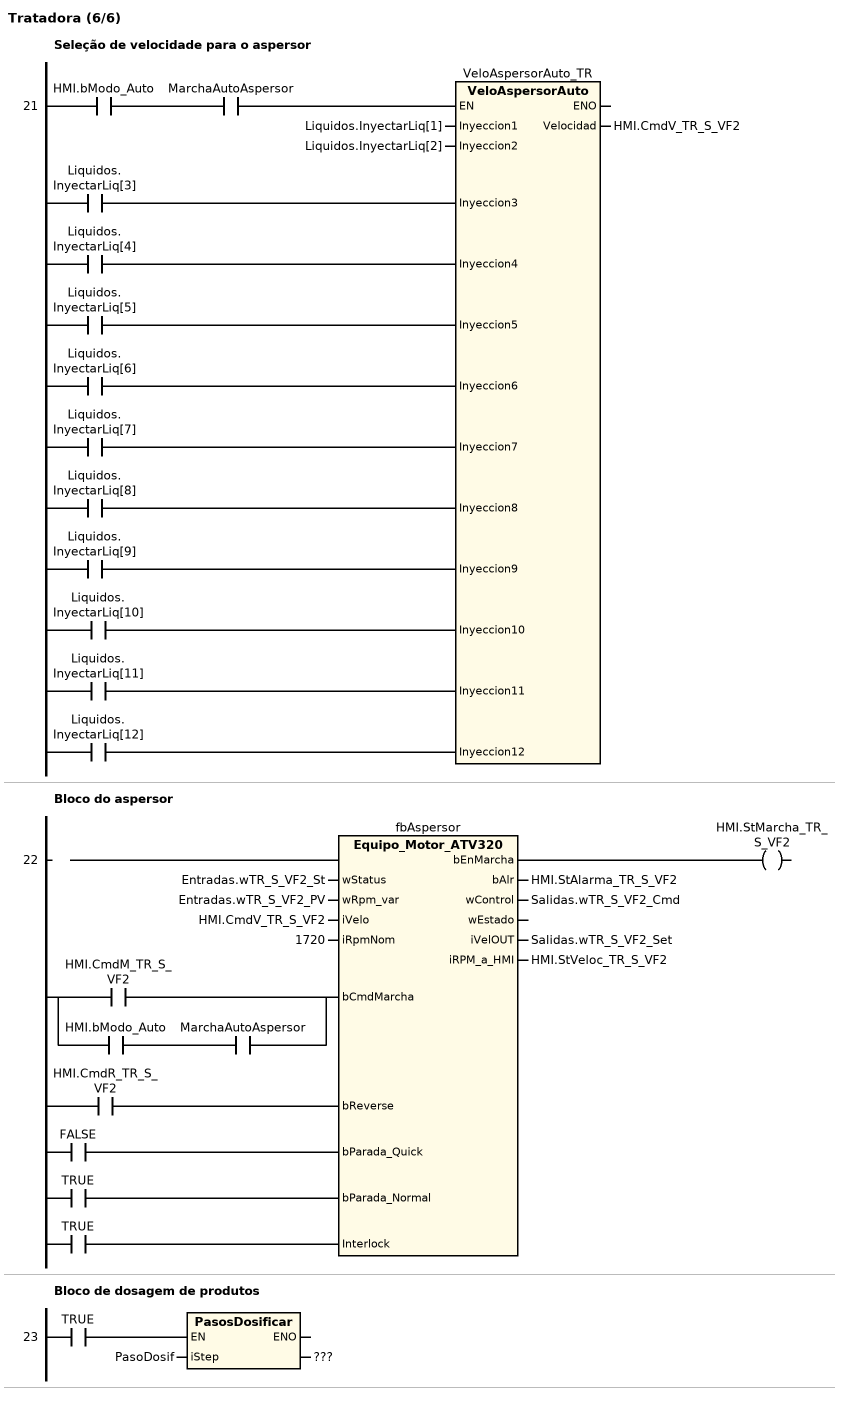
// NETWORK 21: Seleção de velocidade para o aspersor
IF HMI.bModo_Auto AND MarchaAutoAspersor THEN
    VeloAspersorAuto_TR(
        Inyeccion1 := Liquidos.InyectarLiq[1],
        Inyeccion2 := Liquidos.InyectarLiq[2],
        Inyeccion3 := Liquidos.InyectarLiq[3],
        Inyeccion4 := Liquidos.InyectarLiq[4],
        Inyeccion5 := Liquidos.InyectarLiq[5],
        Inyeccion6 := Liquidos.InyectarLiq[6],
        Inyeccion7 := Liquidos.InyectarLiq[7],
        Inyeccion8 := Liquidos.InyectarLiq[8],
        Inyeccion9 := Liquidos.InyectarLiq[9],
        Inyeccion10 := Liquidos.InyectarLiq[10],
        Inyeccion11 := Liquidos.InyectarLiq[11],
        Inyeccion12 := Liquidos.InyectarLiq[12],
        Velocidad => HMI.CmdV_TR_S_VF2); // VeloAspersorAuto
END_IF

// NETWORK 22: Bloco do aspersor
fbAspersor(
    wStatus := Entradas.wTR_S_VF2_St,
    wRpm_var := Entradas.wTR_S_VF2_PV,
    iVelo := HMI.CmdV_TR_S_VF2,
    iRpmNom := 1720,
    bCmdMarcha := HMI.CmdM_TR_S_VF2 OR HMI.bModo_Auto AND MarchaAutoAspersor,
    bReverse := HMI.CmdR_TR_S_VF2,
    bParada_Quick := FALSE,
    bParada_Normal := TRUE,
    Interlock := TRUE,
    bAlr => HMI.StAlarma_TR_S_VF2,
    wControl => Salidas.wTR_S_VF2_Cmd,
    iVelOUT => Salidas.wTR_S_VF2_Set,
    iRPM_a_HMI => HMI.StVeloc_TR_S_VF2); // Equipo_Motor_ATV320
HMI.StMarcha_TR_S_VF2 := fbAspersor.bEnMarcha;

// NETWORK 23: Bloco de dosagem de produtos
PasosDosificar(iStep := PasoDosif);

END_PROGRAM

// ---- POUs/Control Equipos/Equipo_Motor_No_Rev.TcPOU
FUNCTION_BLOCK Equipo_Motor_No_Rev

VAR_INPUT
PE 	  					  : BOOL; (*Parada deemergencia*)
Lock_Out 				  : BOOL;
Conf_Marcha 			  : BOOL; (*Confirmacion de Marcha *)
Modo_Automatico           : BOOL;
Cmd_Auto         		  : BOOL;
Habilitado  			  : BOOL;
T_Discrepancia            : TIME;
END_VAR

VAR_OUTPUT
	Marcha_Equipo	 	  : BOOL;
	Marcha_Ok  				  : BOOL;
	Estado					  : INT;
	Alr_Discrepancia		  : BOOL;	
	Alr_LockOut        		  : BOOL;
END_VAR

VAR_IN_OUT
	Cmd_Man 				  : BOOL;
	Alarma				      : BOOL;
	Horas_Parciales			  : DINT;
	Horas_Totales		 	  : DINT;
	Reset_Horas         	  : BOOL;
	Reset_Alarma		      : BOOL;
END_VAR

VAR_TEMP
	Reset_Cmd_Auto 		      : BOOL;
	Aux_Limpieza		      : TIME;
END_VAR

VAR_STAT
	Cmd_Auto_Directa		  : BOOL;
	FP_Reset				  : R_TRIG;
	FN_Parada_Auto			  : F_TRIG;
	Parcial_Horas			  : INT;
END_VAR

VAR
	Timer_Discrepancia		  : TON;
	Timer_Segundos		      : TON;
END_VAR
VAR PERSISTENT
	Acionamentos	:UDINT;	//Quantidade de vezes que o motor foi acionado
	TempoFuncionando:UDINT;	//Tempo de funcionamento do motor
		
END_VAR
VAR // added by the converter: edge detectors and wires of the graphical bodies
    _w1, _w2, _w3, _w4, _w5, _w6, _w7, _w8, _w9, _w10 : BOOL;
    _rt1 : R_TRIG;
END_VAR

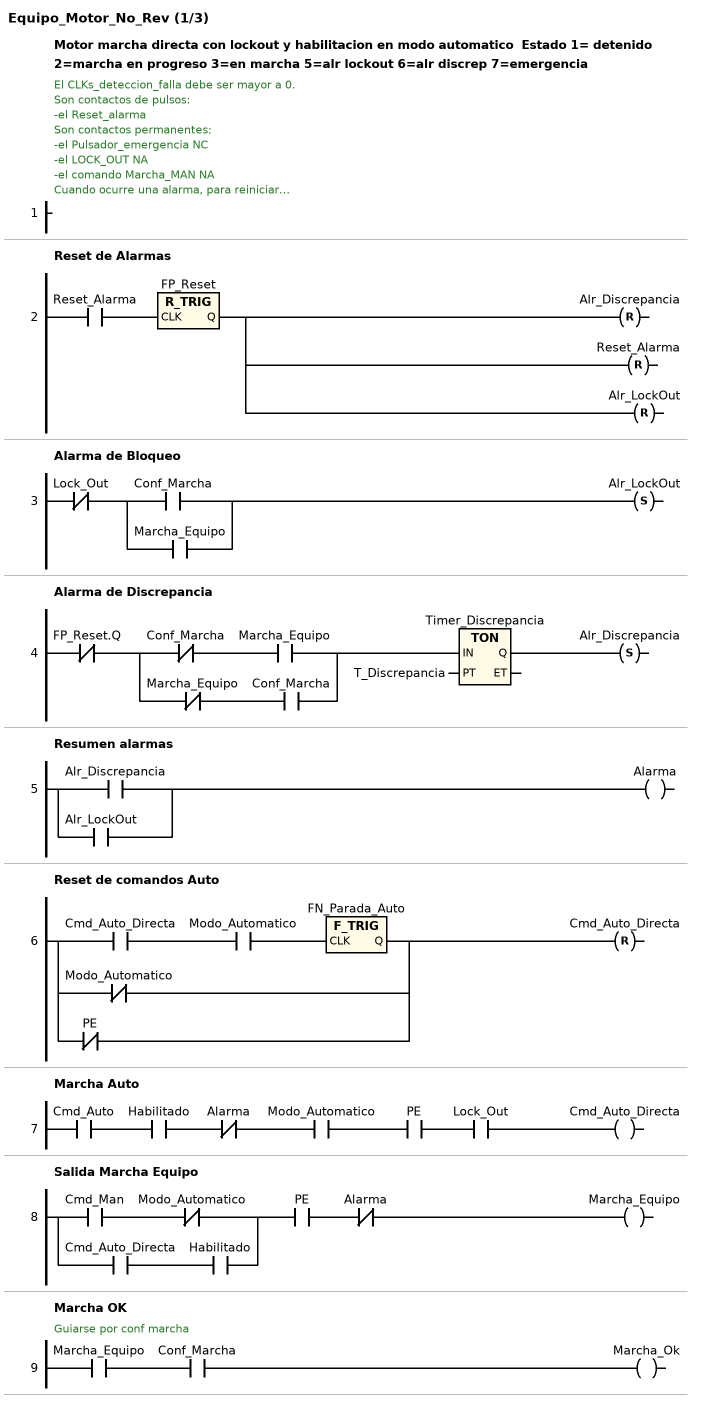
// NETWORK 1: Motor marcha directa con lockout y habilitacion en modo automatico Estado 1= detenido 2=marcha en progreso 3=en marcha 5=alr lockout 6=alr discrep 7=emergencia
// El CLKs_deteccion_falla debe ser mayor a 0.
//
// Son contactos de pulsos:
// -el Reset_alarma
//
// Son contactos permanentes:
// -el Pulsador_emergencia NC
// -el LOCK_OUT NA
// -el comando Marcha_MAN NA
//
// Cuando ocurre una alarma, para reiniciar:
// -en manual reponer la causa de la alarma, pulsar Reset_alarma y pulsar
// Marcha_MAN.
// -en automático reponer la causa de la alarma, pulsar Reset_alarma y si el
// equipo aguas abajo y la Marcha_auto continuan activas, el equipo arrancará.
//
// Siempre que se conmute de automático a manual y viceversa, el equipo se
// detendrá.
//
// Si el equipo es el primero aguas abajo se debe setear siempre en
// 1 Equipos_aguas_abajoOk.
//
// Si el equipo no tiene equipos aguas arribas se debe poner el mismo comando de
// Marcha_MAN en Marcha_aguas_arribaOk

// NETWORK 2: Reset de Alarmas
FP_Reset(CLK := Reset_Alarma); // R_TRIG
Alr_Discrepancia R= FP_Reset.Q;
Reset_Alarma R= FP_Reset.Q;
Alr_LockOut R= FP_Reset.Q;

// NETWORK 3: Alarma de Bloqueo
Alr_LockOut S= NOT Lock_Out AND (Conf_Marcha OR Marcha_Equipo);

// NETWORK 4: Alarma de Discrepancia
Timer_Discrepancia(IN := NOT FP_Reset.Q AND (NOT Conf_Marcha AND Marcha_Equipo OR NOT Marcha_Equipo AND Conf_Marcha), PT := T_Discrepancia); // TON
Alr_Discrepancia S= Timer_Discrepancia.Q;

// NETWORK 5: Resumen alarmas
Alarma := Alr_Discrepancia OR Alr_LockOut;

// NETWORK 6: Reset de comandos Auto
FN_Parada_Auto(CLK := Cmd_Auto_Directa AND Modo_Automatico); // F_TRIG
Cmd_Auto_Directa R= FN_Parada_Auto.Q OR NOT Modo_Automatico OR NOT PE;

// NETWORK 7: Marcha Auto
Cmd_Auto_Directa := Cmd_Auto AND Habilitado AND NOT Alarma AND Modo_Automatico AND PE AND Lock_Out;

// NETWORK 8: Salida Marcha Equipo
Marcha_Equipo := (Cmd_Man AND NOT Modo_Automatico OR Cmd_Auto_Directa AND Habilitado) AND PE AND NOT Alarma;

// NETWORK 9: Marcha OK
// Guiarse por conf marcha
Marcha_Ok := Marcha_Equipo AND Conf_Marcha;

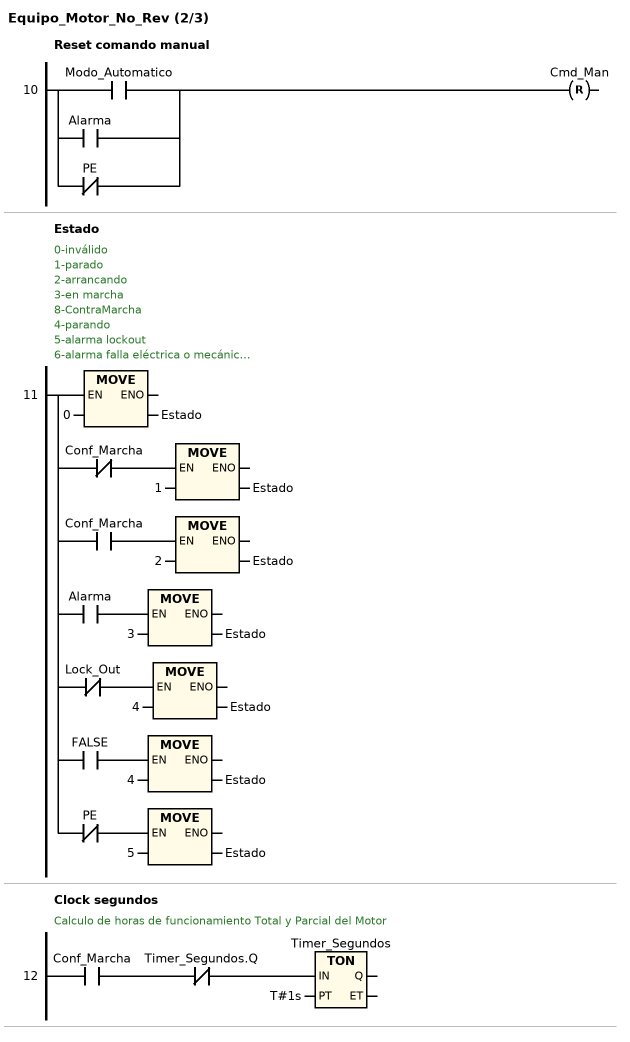
// NETWORK 10: Reset comando manual
Cmd_Man R= Modo_Automatico OR Alarma OR NOT PE;

// NETWORK 11: Estado
// 0-inválido
// 1-parado
// 2-arrancando
// 3-en marcha
// 8-ContraMarcha
// 4-parando
// 5-alarma lockout
// 6-alarma falla eléctrica o mecánica
// 7-alarma pulsador emergencia
Estado := 0;
_w1 := NOT Conf_Marcha;
IF _w1 THEN Estado := 1; END_IF
_w2 := Conf_Marcha;
IF _w2 THEN Estado := 2; END_IF
_w3 := Alarma;
IF _w3 THEN Estado := 3; END_IF
_w4 := NOT Lock_Out;
IF _w4 THEN Estado := 4; END_IF
IF FALSE THEN Estado := 4; END_IF
_w5 := NOT PE;
IF _w5 THEN Estado := 5; END_IF

// NETWORK 12: Clock segundos
// Calculo de horas de funcionamiento Total y Parcial del Motor
Timer_Segundos(IN := Conf_Marcha AND NOT Timer_Segundos.Q, PT := T#1s); // TON

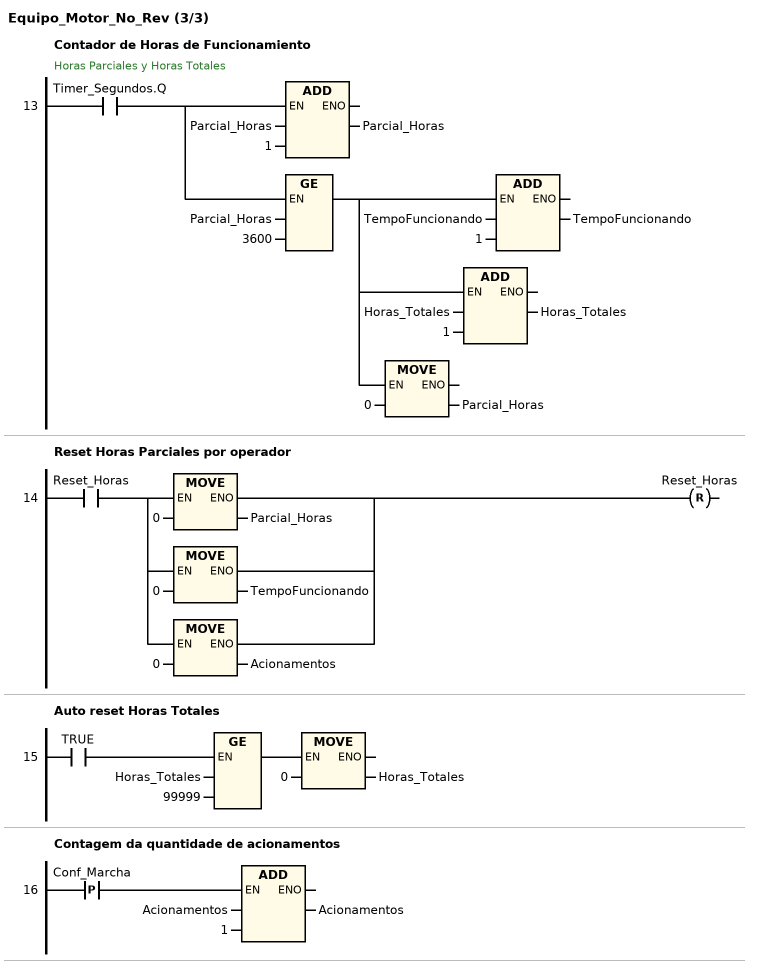
// NETWORK 13: Contador de Horas de Funcionamiento
// Horas Parciales y Horas Totales
_w6 := Timer_Segundos.Q;
IF _w6 THEN Parcial_Horas := Parcial_Horas + 1; END_IF
_w7 := Timer_Segundos.Q AND Parcial_Horas >= 3600;
IF _w7 THEN TempoFuncionando := TempoFuncionando + 1; END_IF
IF _w7 THEN Horas_Totales := Horas_Totales + 1; END_IF
IF _w7 THEN Parcial_Horas := 0; END_IF

// NETWORK 14: Reset Horas Parciales por operador
_w8 := Reset_Horas;
IF _w8 THEN Parcial_Horas := 0; END_IF
_w9 := Reset_Horas;
IF _w9 THEN TempoFuncionando := 0; END_IF
_w10 := Reset_Horas;
IF _w10 THEN Acionamentos := 0; END_IF
Reset_Horas R= _w8 OR (_w9 OR _w10);

// NETWORK 15: Auto reset Horas Totales
IF Horas_Totales >= 99999 THEN Horas_Totales := 0; END_IF

// NETWORK 16: Contagem da quantidade de acionamentos
_rt1(CLK := Conf_Marcha);
IF _rt1.Q THEN Acionamentos := Acionamentos + 1; END_IF

END_FUNCTION_BLOCK

// ---- POUs/Control Equipos/Equipo_Valvula_5_2.TcPOU
FUNCTION_BLOCK Equipo_Valvula_5_2
VAR_INPUT
	PE				: BOOL;	//Parada de emergência
	Modo_Automatico	: BOOL;	//Modo automático
	Cmd_Auto		: BOOL;	//Comando automático
	Valv_Abierta	: BOOL;	//Válvula aberta
	Valv_Cerrada	: BOOL;	//Válvula fechada
	T_Discrepancia	: TIME;	//Tempo para erro de abertura
END_VAR
VAR_OUTPUT
	Activa_Equipo		: BOOL;	//Aciona equipamento
	Estado				: INT;	//Status da válvula
	Alr_Discrepancia	: BOOL;	//Alarme de falha no acionamento
END_VAR
VAR_IN_OUT
	Cmd_Man			: BOOL;	//Comando manual
	Alarma			: BOOL;	//Alarme
	Reset_Alarma	: BOOL;	//Reset alarmes
END_VAR
VAR_STAT
	FP_Reset				  : R_TRIG;
	FN_Parada_Auto			  : F_TRIG;
	FP_Marcha_Auto            : R_TRIG;
	Cmd_Auto_interno		  :BOOL;	
END_VAR

VAR PERSISTENT
	Reset_Eventos         	  : BOOL;
	Timer_Discrepancia		  : TON;
	TON_TempoAbertura: TON;
	R_TRIG_TempoAbertura: R_TRIG;
	TempoAbertura	:DINT;	//Tempo que a válvula demora para abrir
	Eventos_Parciales		  : DINT;
	Eventos_Totales			  : DINT;
END_VAR


VAR
	TON_ResetAlarme: TON;
END_VAR
VAR // added by the converter: edge detectors and wires of the graphical bodies
    _w1, _w2, _w3, _w4, _w5, _w6, _w7 : BOOL;
    _rt1 : R_TRIG;
END_VAR

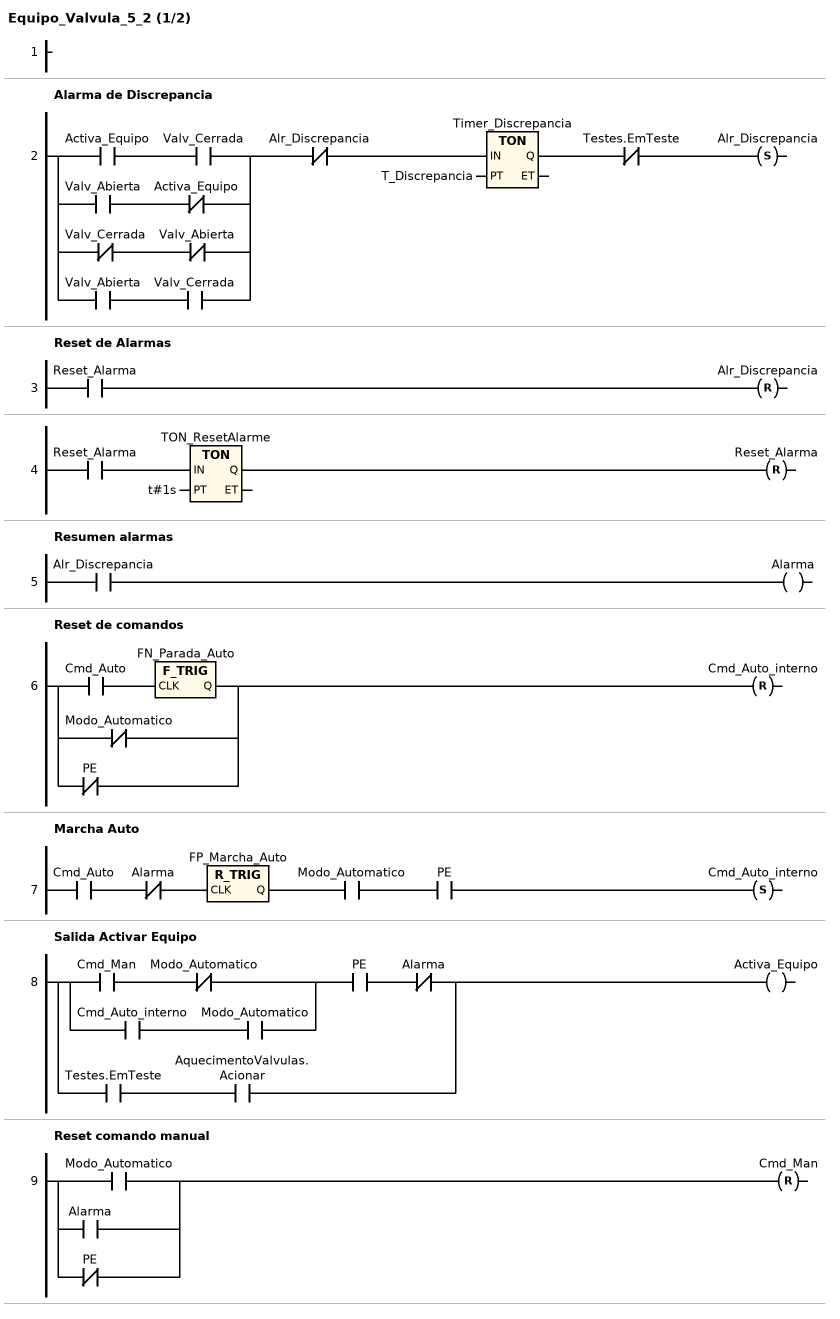
// NETWORK 1

// NETWORK 2: Alarma de Discrepancia
Timer_Discrepancia(IN := (Activa_Equipo AND Valv_Cerrada OR Valv_Abierta AND NOT Activa_Equipo OR NOT Valv_Cerrada AND NOT Valv_Abierta OR Valv_Abierta AND Valv_Cerrada) AND NOT Alr_Discrepancia, PT := T_Discrepancia); // TON
Alr_Discrepancia S= Timer_Discrepancia.Q AND NOT Testes.EmTeste;

// NETWORK 3: Reset de Alarmas
Alr_Discrepancia R= Reset_Alarma;

// NETWORK 4
TON_ResetAlarme(IN := Reset_Alarma, PT := t#1s); // TON
Reset_Alarma R= TON_ResetAlarme.Q;

// NETWORK 5: Resumen alarmas
Alarma := Alr_Discrepancia;

// NETWORK 6: Reset de comandos
FN_Parada_Auto(CLK := Cmd_Auto); // F_TRIG
Cmd_Auto_interno R= FN_Parada_Auto.Q OR NOT Modo_Automatico OR NOT PE;

// NETWORK 7: Marcha Auto
FP_Marcha_Auto(CLK := Cmd_Auto AND NOT Alarma); // R_TRIG
Cmd_Auto_interno S= FP_Marcha_Auto.Q AND Modo_Automatico AND PE;

// NETWORK 8: Salida Activar Equipo
Activa_Equipo := (Cmd_Man AND NOT Modo_Automatico OR Cmd_Auto_interno AND Modo_Automatico) AND PE AND NOT Alarma OR Testes.EmTeste AND AquecimentoValvulas.Acionar;

// NETWORK 9: Reset comando manual
Cmd_Man R= Modo_Automatico OR Alarma OR NOT PE;

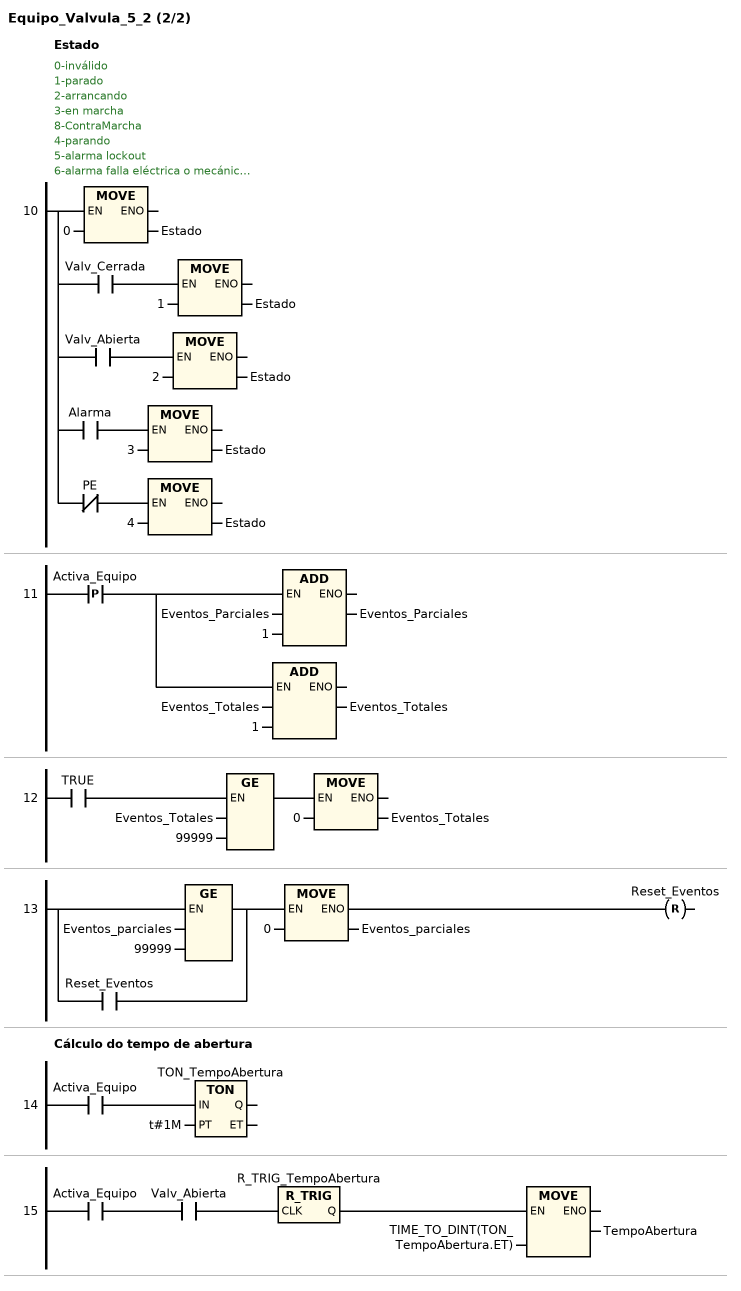
// NETWORK 10: Estado
// 0-inválido
// 1-parado
// 2-arrancando
// 3-en marcha
// 8-ContraMarcha
// 4-parando
// 5-alarma lockout
// 6-alarma falla eléctrica o mecánica
// 7-alarma pulsador emergencia
Estado := 0;
_w1 := Valv_Cerrada;
IF _w1 THEN Estado := 1; END_IF
_w2 := Valv_Abierta;
IF _w2 THEN Estado := 2; END_IF
_w3 := Alarma;
IF _w3 THEN Estado := 3; END_IF
_w4 := NOT PE;
IF _w4 THEN Estado := 4; END_IF

// NETWORK 11
_rt1(CLK := Activa_Equipo);
_w5 := _rt1.Q;
IF _w5 THEN Eventos_Parciales := Eventos_Parciales + 1; END_IF
_w6 := _rt1.Q;
IF _w6 THEN Eventos_Totales := Eventos_Totales + 1; END_IF

// NETWORK 12
IF Eventos_Totales >= 99999 THEN Eventos_Totales := 0; END_IF

// NETWORK 13
_w7 := Reset_Eventos;
IF NOT _w7 THEN
    _w7 := Eventos_parciales >= 99999;
END_IF
IF _w7 THEN Eventos_parciales := 0; END_IF
Reset_Eventos R= _w7;

// NETWORK 14: Cálculo do tempo de abertura
TON_TempoAbertura(IN := Activa_Equipo, PT := t#1M); // TON

// NETWORK 15
R_TRIG_TempoAbertura(CLK := Activa_Equipo AND Valv_Abierta); // R_TRIG
IF R_TRIG_TempoAbertura.Q THEN TempoAbertura := TIME_TO_DINT(TON_TempoAbertura.ET); END_IF

END_FUNCTION_BLOCK

// ---- POUs/Testes Thiago/AquecimentoValvulas.TcPOU
PROGRAM AquecimentoValvulas
VAR
	TON_Acionamento: TON;
	Iniciar	: BOOL;		//Inicia o aquecimento das válvulas
	Tempo	: DINT := 5;		//Tempo em que elas ficarão acionadas (s)
	VarAux: INT;
END_VAR
VAR_OUTPUT
	Acionar	:BOOL;
END_VAR

TON_Acionamento(IN:=Iniciar AND NOT TON_Acionamento.Q AND Testes.EmTeste, PT := DINT_TO_TIME(Tempo * 1000));

//Fica variando a variável auxiliar entre 0 e 1
IF TON_Acionamento.Q THEN
	IF VarAux = 0 THEN
		VarAux := 1;
	ELSE
		VarAux := 0;
	END_IF
END_IF

//Aciona a saída
Acionar := SEL(VarAux = 1, FALSE, TRUE);

END_PROGRAM

// ---- POUs/Control Equipos/Equipo_Motor_ATV320.TcPOU
FUNCTION_BLOCK Equipo_Motor_ATV320
VAR_INPUT
	wStatus			:UINT;
	wRpm_var		:WORD; // rpm actuales leidas del variador
	iVelo			:REAL; // set velocidad en %
	iRpmNom			:INT;// rpm nominales leidas del variador
	bCmdMarcha		:BOOL;
	bReverse		:BOOL;
	bParada_Quick	:BOOL;//parada rapida 16#0002
	bParada_Normal	:BOOL;//parada normal 16#0007
	Interlock	:BOOL;	//Deve estar em TRUE para liberar o funcionamento da bomba
END_VAR
VAR_OUTPUT
	bEnMarcha:BOOL;
	bAlr:BOOL;
	wControl:UINT;
	wEstado:WORD;
	iVelOUT:UINT;
	iRPM_a_HMI:INT; //rpm para el HMI

END_VAR
VAR
	Aux_Status:DINT;
	bMarcha:BOOL;
	TempoFuncionando:UDINT;	//Tempo de funcionamento do motor
	Acionamentos	:UDINT;	//Quantidade de acionamentos do motor
	TON_Horimetro: TON;
	RTRIG_Funcionamento: R_TRIG;
	ResetContadores: BOOL;
	TONR_Horimetro: TONR;
	ResetFalhas		:BOOL;	//Reset das falhas do inversor
END_VAR


(*cuenta horas de marcha parciales*)
(*cuenta horas de marcha totales*)

(***********************************************************************Tratamiento PDO*)
wEstado := wStatus;
iVelOUT:=REAL_TO_UINT(iRpmNom*iVelo/100);// convierte velocidad solicitada en % a rpm
iRPM_a_HMI:=WORD_TO_INT (wRpm_var);

Aux_Status:= DINT_TO_UINT(wStatus) AND 16#007F;


(*Secuencia Marcha*)
IF bCmdMarcha AND Interlock THEN
	IF (Aux_Status=16#0050 OR Aux_Status =16#0060 OR Aux_Status =16#0080) THEN
		wControl:=16#0006;	
	END_IF
	IF Aux_Status=16#0031  THEN
		wControl:=16#0007;	
	END_IF
	IF Aux_Status=16#0033  THEN
		IF bReverse THEN	
			wControl:=16#080F;
		ELSE	
			wControl:=16#000F;
		END_IF
	END_IF	
END_IF

(*Secuencia Parada*)
IF  (NOT bCmdMarcha OR NOT Interlock) AND Aux_Status=16#0037 THEN
	IF bParada_Quick THEN
		wControl:=16#0002;//quick	
		ELSE
		wControl:=16#0007;//normal
	END_IF
END_IF 

(*Deshabilita tension*)
IF  Aux_Status=16#0017 THEN
	wControl:=16#0000;
END_IF 

(*Aviso Falla*)
IF (Aux_Status=16#0008 OR Aux_Status=16#0028 OR Aux_Status=16#000F OR Aux_Status=16#0038 OR Aux_Status=16#002F OR Aux_Status=16#0018 ) THEN
	bAlr:=1;
	ELSE
	bAlr:=0;	
	END_IF
	
(*Reset Falla*)
IF bAlr AND ResetFalhas THEN
	wControl := 128;		//Aciona o bit 7 da palavra de controle
	ResetFalhas := FALSE;
END_IF

(*Estado*)
IF (Aux_Status=16#0037) THEN
	bEnMarcha:=1;
	
ELSE
	bEnMarcha:=0;	
END_IF

//Motor rodando
//Motor rodando

TONR_Horimetro(
	EN:= bEnMarcha, 
	PRE:= T#1M, 
	RES:= TONR_Horimetro.DN, 
	DN=> , 
	ACC=> , 
	TT=> );

IF TONR_Horimetro.DN THEN
	TempoFuncionando := TempoFuncionando + 1;
	TempoFuncionando := TempoFuncionando/2;	//Essa divisão foi necessária pois o TONR não reseta corretamente
END_IF

//Quantidade de acionamentos
RTRIG_Funcionamento(CLK:=bEnMarcha);
IF RTRIG_Funcionamento.Q THEN
	Acionamentos := Acionamentos + 1;
END_IF

//Reset contadores
IF ResetContadores THEN
	Acionamentos		:= 0;
	TempoFuncionando	:= 0;
	ResetContadores		:= FALSE;
END_IF


(***********************************************************************Tratamiento SDO*)

END_FUNCTION_BLOCK

// ---- POUs/Testes Thiago/TONR.TcPOU
FUNCTION_BLOCK TONR
VAR_INPUT
    EN: BOOL; // timer enable
    PRE: TIME; // preset time
    RES: BOOL; // reset signal
END_VAR
VAR_OUTPUT
    DN: BOOL; // timer done
    ACC: TIME; // accumulated time
    TT: BOOL; // timer timing
END_VAR
VAR
    Timer: TON;
    TempAcc: TIME;
END_VAR

ACC := TempAcc + Timer.ET;
DN := (ACC >= PRE);

IF NOT EN OR DN THEN
    TempAcc := TempAcc + Timer.ET;
END_IF

IF RES THEN
    ACC := T#0MS;
    TempAcc := T#0MS;
END_IF

Timer(IN:=EN AND NOT DN AND NOT RES, PT:=T#2147483647MS);

TT := Timer.IN;

END_FUNCTION_BLOCK

// ---- POUs/Elementos/Tiempo_seg_to_TIME.TcPOU
FUNCTION_BLOCK Tiempo_seg_to_TIME
VAR_INPUT
	Segundos:REAL;
END_VAR
VAR_OUTPUT
	tTime:TIME;
END_VAR
VAR
END_VAR

tTIME:=REAL_TO_TIME (Segundos*1000);

END_FUNCTION_BLOCK

// ---- POUs/Secuencias/VeloAspersorAuto.TcPOU
FUNCTION_BLOCK VeloAspersorAuto
VAR_INPUT
	Inyeccion1:BOOL;
	Inyeccion2:BOOL;	
	Inyeccion3:BOOL;
	Inyeccion4:BOOL;
	Inyeccion5:BOOL;
	Inyeccion6:BOOL;	
	Inyeccion7:BOOL;
	Inyeccion8:BOOL;
	Inyeccion9:BOOL;
	Inyeccion10:BOOL;	
	Inyeccion11:BOOL;
	Inyeccion12:BOOL;
		
END_VAR
VAR_OUTPUT
	Velocidad:REAL;
END_VAR
VAR
END_VAR

Velocidad:=0;
IF Inyeccion1 THEN
	IF Liquidos.TablaLiquidos[Liquidos.Circuito_Liquido[1]].iVelAspersor>Velocidad  THEN
		Velocidad:=Liquidos.TablaLiquidos[Liquidos.Circuito_Liquido[1]].iVelAspersor;
	END_IF
END_IF
IF Inyeccion2 THEN
	IF Liquidos.TablaLiquidos[Liquidos.Circuito_Liquido[2]].iVelAspersor>Velocidad  THEN
		Velocidad:=Liquidos.TablaLiquidos[Liquidos.Circuito_Liquido[2]].iVelAspersor; 
	END_IF
END_IF
IF Inyeccion3 THEN
	IF Liquidos.TablaLiquidos[Liquidos.Circuito_Liquido[3]].iVelAspersor>Velocidad  THEN
		Velocidad:=Liquidos.TablaLiquidos[Liquidos.Circuito_Liquido[3]].iVelAspersor;
	END_IF
END_IF

IF Inyeccion4 THEN
	IF Liquidos.TablaLiquidos[Liquidos.Circuito_Liquido[4]].iVelAspersor>Velocidad  THEN
		Velocidad:=Liquidos.TablaLiquidos[Liquidos.Circuito_Liquido[4]].iVelAspersor;
	END_IF
END_IF
IF Inyeccion5 THEN
	IF Liquidos.TablaLiquidos[Liquidos.Circuito_Liquido[5]].iVelAspersor>Velocidad  THEN
		Velocidad:=Liquidos.TablaLiquidos[Liquidos.Circuito_Liquido[5]].iVelAspersor;
	END_IF
END_IF
IF Inyeccion6 THEN
	IF Liquidos.TablaLiquidos[Liquidos.Circuito_Liquido[6]].iVelAspersor>Velocidad  THEN
		Velocidad:=Liquidos.TablaLiquidos[Liquidos.Circuito_Liquido[6]].iVelAspersor;
	END_IF
END_IF
IF Inyeccion7 THEN
	IF Liquidos.TablaLiquidos[Liquidos.Circuito_Liquido[7]].iVelAspersor>Velocidad  THEN
		Velocidad:=Liquidos.TablaLiquidos[Liquidos.Circuito_Liquido[7]].iVelAspersor;
	END_IF
END_IF
IF Inyeccion8 THEN
	IF Liquidos.TablaLiquidos[Liquidos.Circuito_Liquido[8]].iVelAspersor>Velocidad  THEN
		Velocidad:=Liquidos.TablaLiquidos[Liquidos.Circuito_Liquido[8]].iVelAspersor;
	END_IF
END_IF
IF Inyeccion9 THEN
	IF Liquidos.TablaLiquidos[Liquidos.Circuito_Liquido[9]].iVelAspersor>Velocidad  THEN
		Velocidad:=Liquidos.TablaLiquidos[Liquidos.Circuito_Liquido[9]].iVelAspersor;
	END_IF
END_IF
IF Inyeccion10 THEN
	IF Liquidos.TablaLiquidos[Liquidos.Circuito_Liquido[10]].iVelAspersor>Velocidad  THEN
		Velocidad:=Liquidos.TablaLiquidos[Liquidos.Circuito_Liquido[10]].iVelAspersor;
	END_IF
END_IF
IF Inyeccion11 THEN
	IF Liquidos.TablaLiquidos[Liquidos.Circuito_Liquido[11]].iVelAspersor>Velocidad  THEN
		Velocidad:=Liquidos.TablaLiquidos[Liquidos.Circuito_Liquido[11]].iVelAspersor;
	END_IF
END_IF
IF Inyeccion12 THEN
	IF Liquidos.TablaLiquidos[Liquidos.Circuito_Liquido[12]].iVelAspersor>Velocidad  THEN
		Velocidad:=Liquidos.TablaLiquidos[Liquidos.Circuito_Liquido[12]].iVelAspersor;
	END_IF
END_IF
IF NOT Inyeccion1 AND
	NOT Inyeccion2 AND
	NOT Inyeccion3 AND
	NOT Inyeccion4 AND
	NOT Inyeccion5 AND
	NOT Inyeccion6 AND
	NOT Inyeccion7 AND
	NOT Inyeccion8 AND
	NOT Inyeccion9 AND
	NOT Inyeccion10 AND
	NOT Inyeccion11 AND
	NOT Inyeccion12 THEN
	Velocidad := 100;
	END_IF

END_FUNCTION_BLOCK

// ---- POUs/Elementos/Tiempo_TIME_to_seg.TcPOU
FUNCTION_BLOCK Tiempo_TIME_to_seg
VAR_INPUT
	tTime:TIME;
END_VAR
VAR_OUTPUT
	Segundos:DINT;
END_VAR
VAR
END_VAR

Segundos:=TIME_TO_DINT (tTime)/100;

END_FUNCTION_BLOCK

// ---- POUs/Testes Thiago/Percentual.TcPOU
FUNCTION_BLOCK Percentual
VAR_INPUT
	VAR_1:DINT;
	VAR_2:DINT;
END_VAR
VAR_OUTPUT
	OUTPUT:DINT;
END_VAR

//Retorna o valor percentual da variável 1 em relação a variável 2
OUTPUT := SEL(VAR_2 > 0, 0,(VAR_1*100/VAR_2*100)/100);

END_FUNCTION_BLOCK

// ---- POUs/Balanza_Semilla.TcPOU
PROGRAM Balanza_Semilla
VAR
	// grueso carga balanza
	TR_S_V2: Equipo_Valvula_5_2; //Válvula de corte grosso
	// fino carga balanza
	TR_S_V3: Equipo_Valvula_5_2;
	// descarga balanza
	TR_S_V4: Equipo_Valvula_5_2;
	//
	TR_S_V2_CmdAuto:BOOL;	//Válvula de corte grosso
	TR_S_V3_CmdAuto:BOOL;	//Válvula de corte fino
	TR_S_V4_CmdAuto:BOOL;	//Válvula de descarga
	// Balanza de pesaje de semilla
	TR_S_WT1: Balanza;
	//
	Hab_cargarSemilla	:BOOL;
	Cargar_Balanza		:BOOL;
	TolerInf_pesoSemilla:REAL;	//Tolerância inferior da carga da balança
	TolerSup_pesoSemilla:REAL;	//Tolerância superior da balança
	Balanza_cargadaOk	:BOOL;
	Hab_descargarSemilla:BOOL;
	Descargar_Balanza	:BOOL;
	PesoSemilla_paraDosificar:REAL;
	Espera_pesasArriba:TON;
	Espera_Estable:TON;
	Espera_DescAbierta:TON;
	
	// tiempo de carga/descarga de balanza semilla excesivo
	Alr_demoraCarga: TON;
	Alr_demoraDescarga:TON;
	
	TriggerTomarPeso :BOOL;
	
	//provisorios
	bHS :BOOL;
	dintHS	:DINT:=3;
	Hx :BOOL;
	IniCal:BOOL;
	
	iStep :INT;
	Espera_pesas :TON;
	
	AuxHugo :BOOL;
	Procesando: BOOL;
	Tabla_FIFO_Peso: Tabla_FIFO;
	Balanza_vacia: BOOL;
	FinCarga: BOOL;
	TmrGruesoOk: TON;
	TBalanzaVacia: TON;
	PolvosOk: BOOL;
	// Timer para aparecer a popup de peso fora de tolerância
	TON_PesoForaTolerancia: TON;
	TON_DemoraCarga: TON;
	// Se a caixa superior estiver sem nível de sementes, permite que a semente remanescente seja carregada na balança
	EsvaziarCaixa: BOOL;
	qtdBateladas	:UDINT;	//Quantidade de bateladas feitas
END_VAR
VAR // added by the converter: edge detectors and wires of the graphical bodies
    _rt1, _rt2, _rt3, _rt4, _rt5, _rt6 : R_TRIG;
    _w1, _w2, _w3, _w4, _w5, _w6, _w7, _w8, _w9, _w10, _w11, _w12, _w13, _w14, _w15 : BOOL;
    _ft1 : F_TRIG;
END_VAR

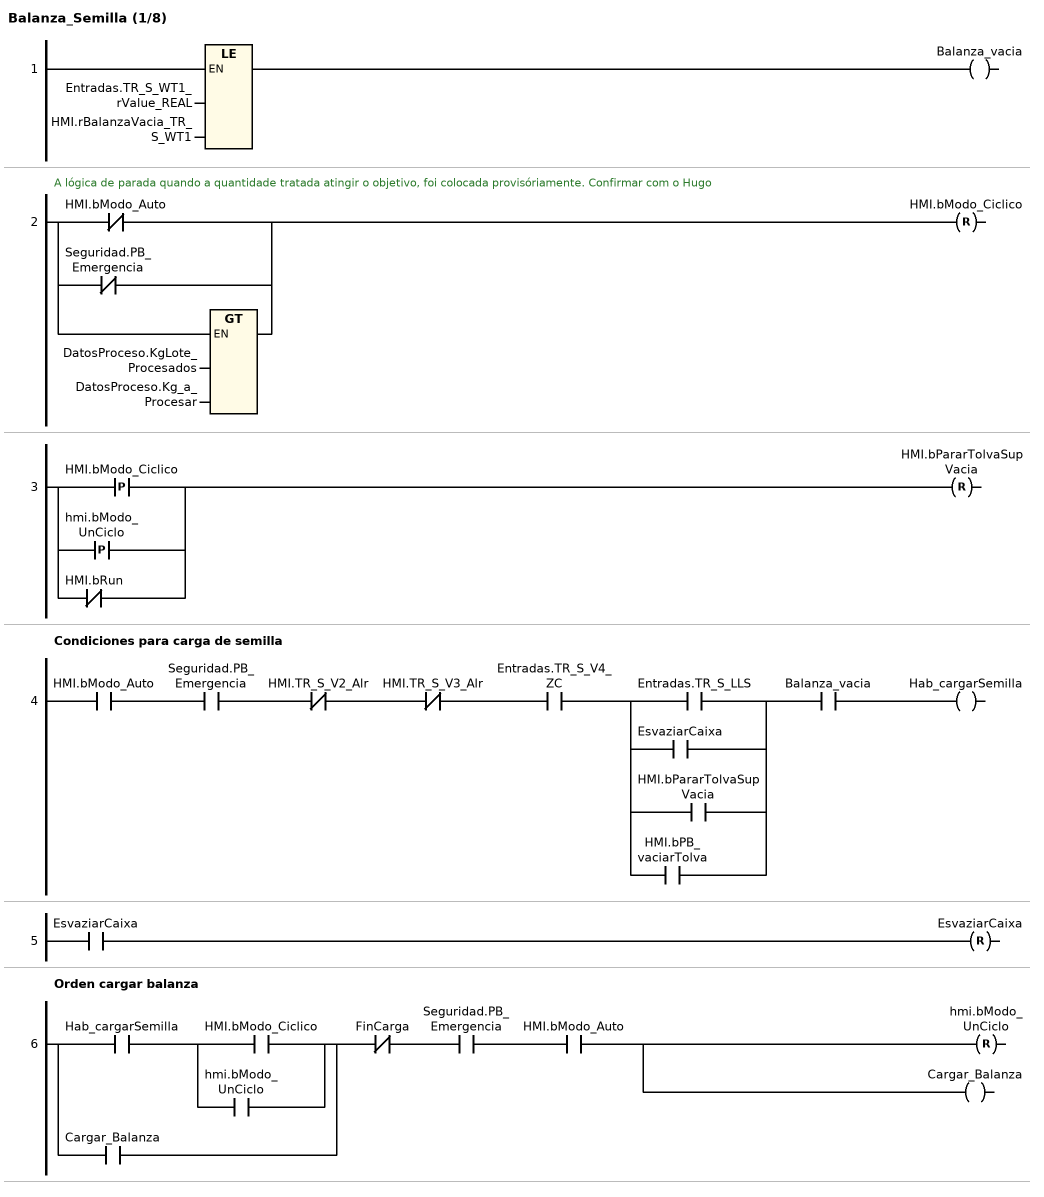
// NETWORK 1
Balanza_vacia := Entradas.TR_S_WT1_rValue_REAL <= HMI.rBalanzaVacia_TR_S_WT1;

// NETWORK 2
// A lógica de parada quando a quantidade tratada atingir o objetivo, foi colocada provisóriamente. Confirmar com o Hugo
HMI.bModo_Ciclico R= NOT HMI.bModo_Auto OR NOT Seguridad.PB_Emergencia OR DatosProceso.KgLote_Procesados > DatosProceso.Kg_a_Procesar;

// NETWORK 3
_rt1(CLK := HMI.bModo_Ciclico);
_rt2(CLK := hmi.bModo_UnCiclo);
HMI.bPararTolvaSupVacia R= _rt1.Q OR _rt2.Q OR NOT HMI.bRun;

// NETWORK 4: Condiciones para carga de semilla
Hab_cargarSemilla := HMI.bModo_Auto AND Seguridad.PB_Emergencia AND NOT HMI.TR_S_V2_Alr AND NOT HMI.TR_S_V3_Alr AND Entradas.TR_S_V4_ZC AND (Entradas.TR_S_LLS OR EsvaziarCaixa OR HMI.bPararTolvaSupVacia OR HMI.bPB_vaciarTolva) AND Balanza_vacia;

// NETWORK 5
EsvaziarCaixa R= EsvaziarCaixa;

// NETWORK 6: Orden cargar balanza
_w1 := (Hab_cargarSemilla AND (HMI.bModo_Ciclico OR hmi.bModo_UnCiclo) OR Cargar_Balanza) AND NOT FinCarga AND Seguridad.PB_Emergencia AND HMI.bModo_Auto;
hmi.bModo_UnCiclo R= _w1;
Cargar_Balanza := _w1;

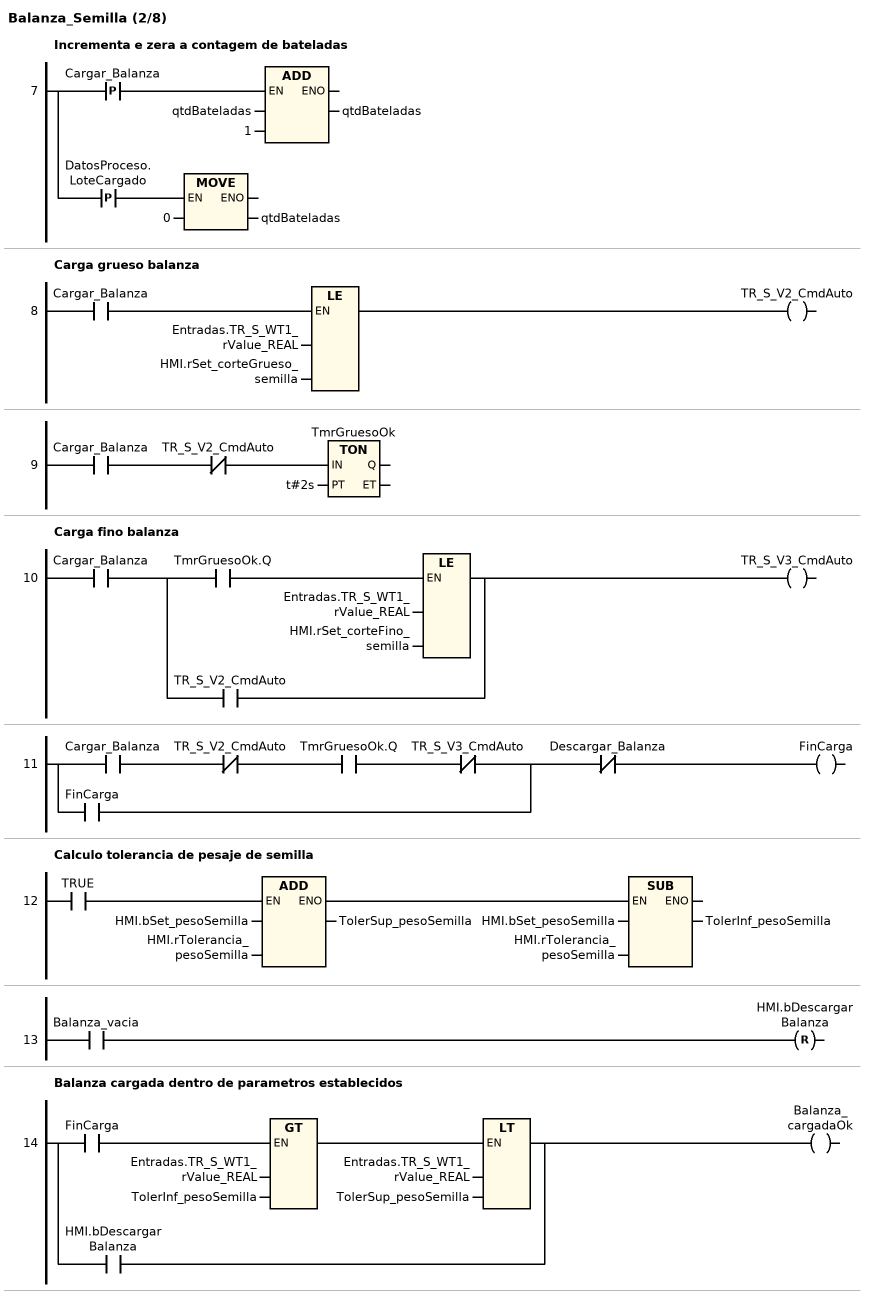
// NETWORK 7: Incrementa e zera a contagem de bateladas
_rt3(CLK := Cargar_Balanza);
_w2 := _rt3.Q;
IF _w2 THEN qtdBateladas := qtdBateladas + 1; END_IF
_rt4(CLK := DatosProceso.LoteCargado);
_w3 := _rt4.Q;
IF _w3 THEN qtdBateladas := 0; END_IF
(* _w2 OR _w3; result not used *)

// NETWORK 8: Carga grueso balanza
TR_S_V2_CmdAuto := Cargar_Balanza AND Entradas.TR_S_WT1_rValue_REAL <= HMI.rSet_corteGrueso_semilla;

// NETWORK 9
TmrGruesoOk(IN := Cargar_Balanza AND NOT TR_S_V2_CmdAuto, PT := t#2s); // TON

// NETWORK 10: Carga fino balanza
_w4 := Cargar_Balanza AND TR_S_V2_CmdAuto;
IF NOT _w4 THEN
    _w4 := Cargar_Balanza AND TmrGruesoOk.Q AND Entradas.TR_S_WT1_rValue_REAL <= HMI.rSet_corteFino_semilla;
END_IF
TR_S_V3_CmdAuto := _w4;

// NETWORK 11
FinCarga := (Cargar_Balanza AND NOT TR_S_V2_CmdAuto AND TmrGruesoOk.Q AND NOT TR_S_V3_CmdAuto OR FinCarga) AND NOT Descargar_Balanza;

// NETWORK 12: Calculo tolerancia de pesaje de semilla
TolerSup_pesoSemilla := HMI.bSet_pesoSemilla + HMI.rTolerancia_pesoSemilla;
TolerInf_pesoSemilla := HMI.bSet_pesoSemilla - HMI.rTolerancia_pesoSemilla;

// NETWORK 13
HMI.bDescargarBalanza R= Balanza_vacia;

// NETWORK 14: Balanza cargada dentro de parametros establecidos
_w5 := HMI.bDescargarBalanza;
IF NOT _w5 THEN
    _w5 := FinCarga AND Entradas.TR_S_WT1_rValue_REAL > TolerInf_pesoSemilla AND Entradas.TR_S_WT1_rValue_REAL < TolerSup_pesoSemilla;
END_IF
Balanza_cargadaOk := _w5;

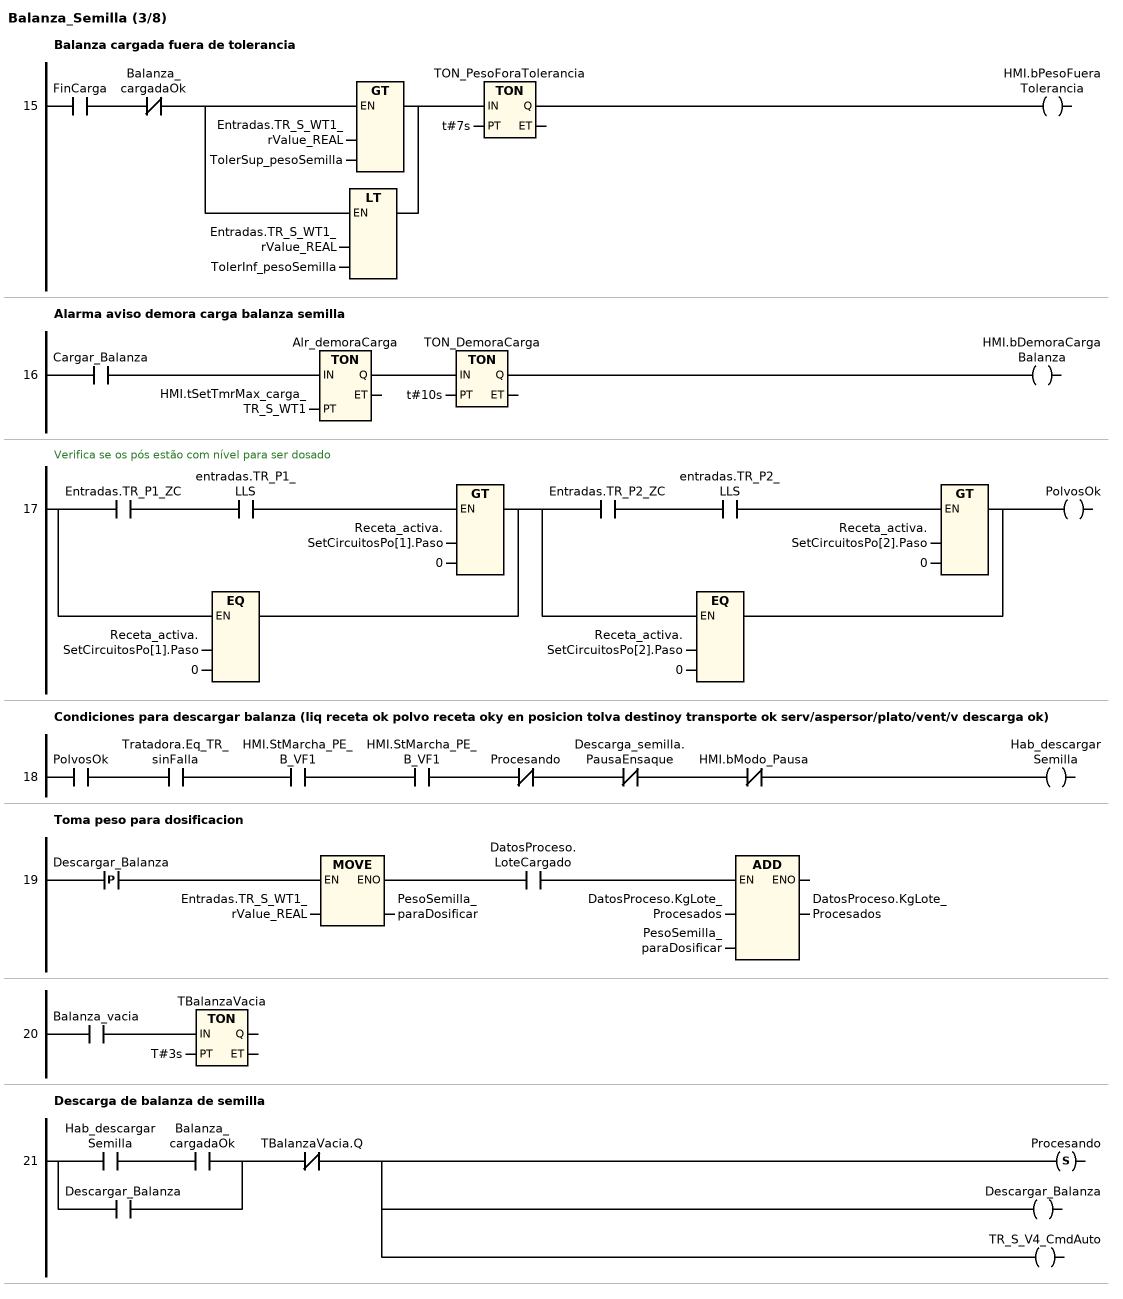
// NETWORK 15: Balanza cargada fuera de tolerancia
_w6 := FinCarga AND NOT Balanza_cargadaOk;
TON_PesoForaTolerancia(IN := _w6 AND Entradas.TR_S_WT1_rValue_REAL > TolerSup_pesoSemilla OR _w6 AND Entradas.TR_S_WT1_rValue_REAL < TolerInf_pesoSemilla, PT := t#7s); // TON
HMI.bPesoFueraTolerancia := TON_PesoForaTolerancia.Q;

// NETWORK 16: Alarma aviso demora carga balanza semilla
Alr_demoraCarga(IN := Cargar_Balanza, PT := HMI.tSetTmrMax_carga_TR_S_WT1); // TON
TON_DemoraCarga(IN := Alr_demoraCarga.Q, PT := t#10s); // TON
HMI.bDemoraCargaBalanza := TON_DemoraCarga.Q;

// NETWORK 17
// Verifica se os pós estão com nível para ser dosado
_w7 := Entradas.TR_P1_ZC AND entradas.TR_P1_LLS AND Receta_activa.SetCircuitosPo[1].Paso > 0 OR Receta_activa.SetCircuitosPo[1].Paso = 0;
PolvosOk := (_w7 AND Entradas.TR_P2_ZC) AND entradas.TR_P2_LLS AND Receta_activa.SetCircuitosPo[2].Paso > 0 OR _w7 AND Receta_activa.SetCircuitosPo[2].Paso = 0;

// NETWORK 18: Condiciones para descargar balanza (liq receta ok polvo receta oky en posicion tolva destinoy transporte ok serv/aspersor/plato/vent/v descarga ok)
Hab_descargarSemilla := PolvosOk AND Tratadora.Eq_TR_sinFalla AND HMI.StMarcha_PE_B_VF1 AND HMI.StMarcha_PE_B_VF1 AND NOT Procesando AND NOT Descarga_semilla.PausaEnsaque AND NOT HMI.bModo_Pausa;

// NETWORK 19: Toma peso para dosificacion
_rt5(CLK := Descargar_Balanza);
_w8 := _rt5.Q;
IF _w8 THEN PesoSemilla_paraDosificar := Entradas.TR_S_WT1_rValue_REAL; END_IF
IF _w8 AND DatosProceso.LoteCargado THEN
    DatosProceso.KgLote_Procesados := DatosProceso.KgLote_Procesados + PesoSemilla_paraDosificar;
END_IF

// NETWORK 20
TBalanzaVacia(IN := Balanza_vacia, PT := T#3s); // TON

// NETWORK 21: Descarga de balanza de semilla
_w9 := (Hab_descargarSemilla AND Balanza_cargadaOk OR Descargar_Balanza) AND NOT TBalanzaVacia.Q;
Procesando S= _w9;
Descargar_Balanza := _w9;
TR_S_V4_CmdAuto := _w9;

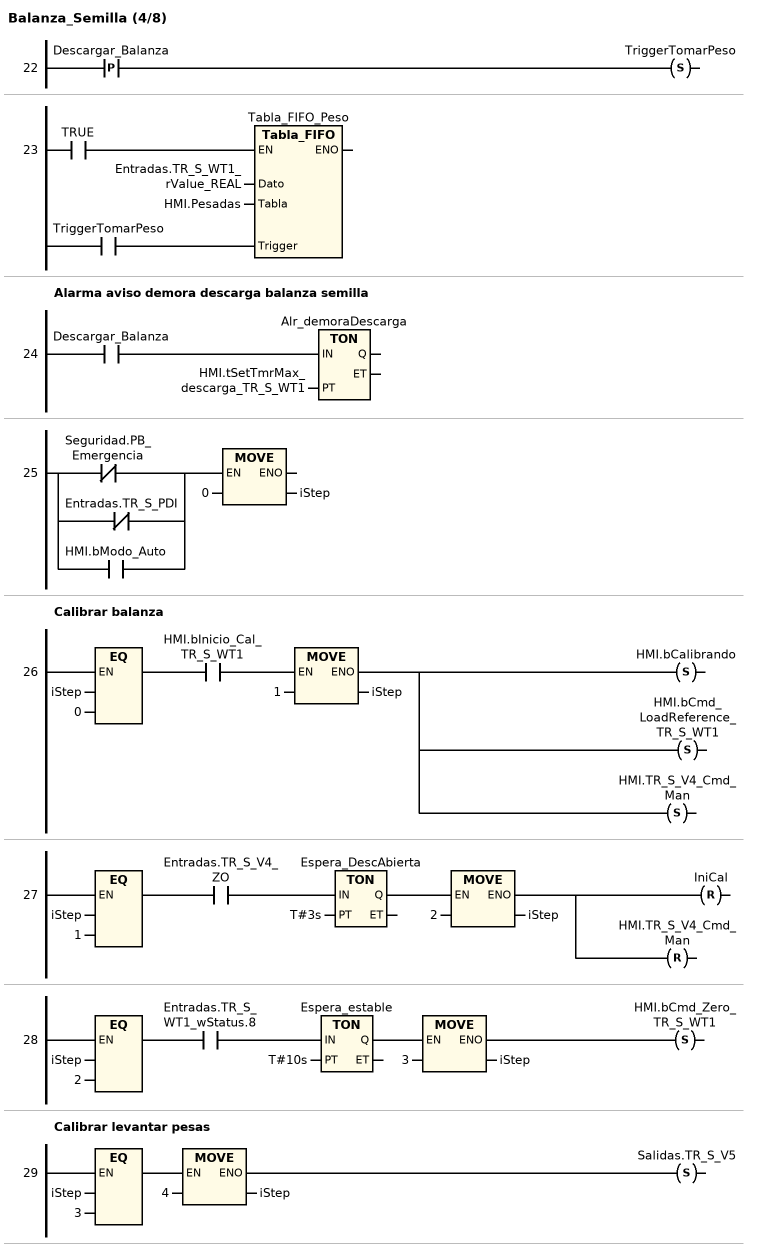
// NETWORK 22
_rt6(CLK := Descargar_Balanza);
TriggerTomarPeso S= _rt6.Q;

// NETWORK 23
Tabla_FIFO_Peso(Dato := Entradas.TR_S_WT1_rValue_REAL, Tabla := HMI.Pesadas, Trigger := TriggerTomarPeso); // Tabla_FIFO

// NETWORK 24: Alarma aviso demora descarga balanza semilla
Alr_demoraDescarga(IN := Descargar_Balanza, PT := HMI.tSetTmrMax_descarga_TR_S_WT1); // TON

// NETWORK 25
IF NOT Seguridad.PB_Emergencia OR NOT Entradas.TR_S_PDI OR HMI.bModo_Auto THEN iStep := 0; END_IF

// NETWORK 26: Calibrar balanza
_w10 := iStep = 0 AND HMI.bInicio_Cal_TR_S_WT1;
IF _w10 THEN iStep := 1; END_IF
HMI.bCalibrando S= _w10;
HMI.bCmd_LoadReference_TR_S_WT1 S= _w10;
HMI.TR_S_V4_Cmd_Man S= _w10;

// NETWORK 27
Espera_DescAbierta(IN := iStep = 1 AND Entradas.TR_S_V4_ZO, PT := T#3s); // TON
_w11 := Espera_DescAbierta.Q;
IF _w11 THEN iStep := 2; END_IF
IniCal R= _w11;
HMI.TR_S_V4_Cmd_Man R= _w11;

// NETWORK 28
Espera_estable(IN := iStep = 2 AND Entradas.TR_S_WT1_wStatus.8, PT := T#10s); // TON
_w12 := Espera_estable.Q;
IF _w12 THEN iStep := 3; END_IF
HMI.bCmd_Zero_TR_S_WT1 S= _w12;

// NETWORK 29: Calibrar levantar pesas
_w13 := iStep = 3;
IF _w13 THEN iStep := 4; END_IF
Salidas.TR_S_V5 S= _w13;

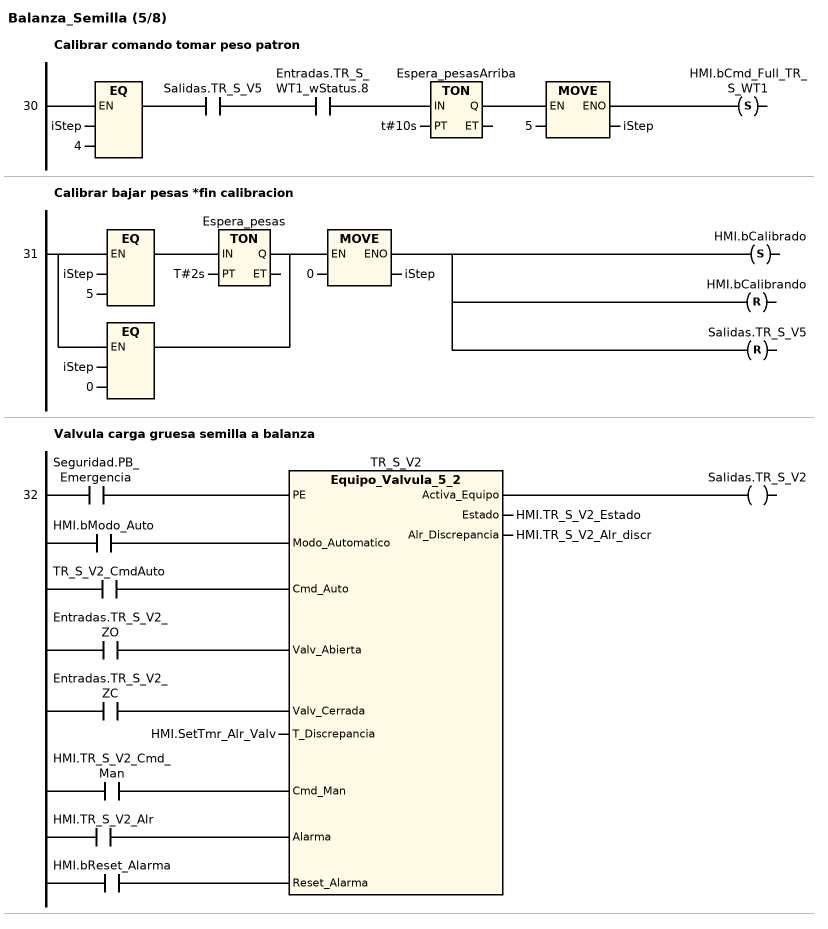
// NETWORK 30: Calibrar comando tomar peso patron
Espera_pesasArriba(IN := iStep = 4 AND Salidas.TR_S_V5 AND Entradas.TR_S_WT1_wStatus.8, PT := t#10s); // TON
_w14 := Espera_pesasArriba.Q;
IF _w14 THEN iStep := 5; END_IF
HMI.bCmd_Full_TR_S_WT1 S= _w14;

// NETWORK 31: Calibrar bajar pesas *fin calibracion
Espera_pesas(IN := iStep = 5, PT := T#2s); // TON
_w15 := Espera_pesas.Q OR iStep = 0;
IF _w15 THEN iStep := 0; END_IF
HMI.bCalibrado S= _w15;
HMI.bCalibrando R= _w15;
Salidas.TR_S_V5 R= _w15;

// NETWORK 32: Valvula carga gruesa semilla a balanza
TR_S_V2(
    PE := Seguridad.PB_Emergencia,
    Modo_Automatico := HMI.bModo_Auto,
    Cmd_Auto := TR_S_V2_CmdAuto,
    Valv_Abierta := Entradas.TR_S_V2_ZO,
    Valv_Cerrada := Entradas.TR_S_V2_ZC,
    T_Discrepancia := HMI.SetTmr_Alr_Valv,
    Cmd_Man := HMI.TR_S_V2_Cmd_Man,
    Alarma := HMI.TR_S_V2_Alr,
    Reset_Alarma := HMI.bReset_Alarma,
    Estado => HMI.TR_S_V2_Estado,
    Alr_Discrepancia => HMI.TR_S_V2_Alr_discr); // Equipo_Valvula_5_2
Salidas.TR_S_V2 := TR_S_V2.Activa_Equipo;

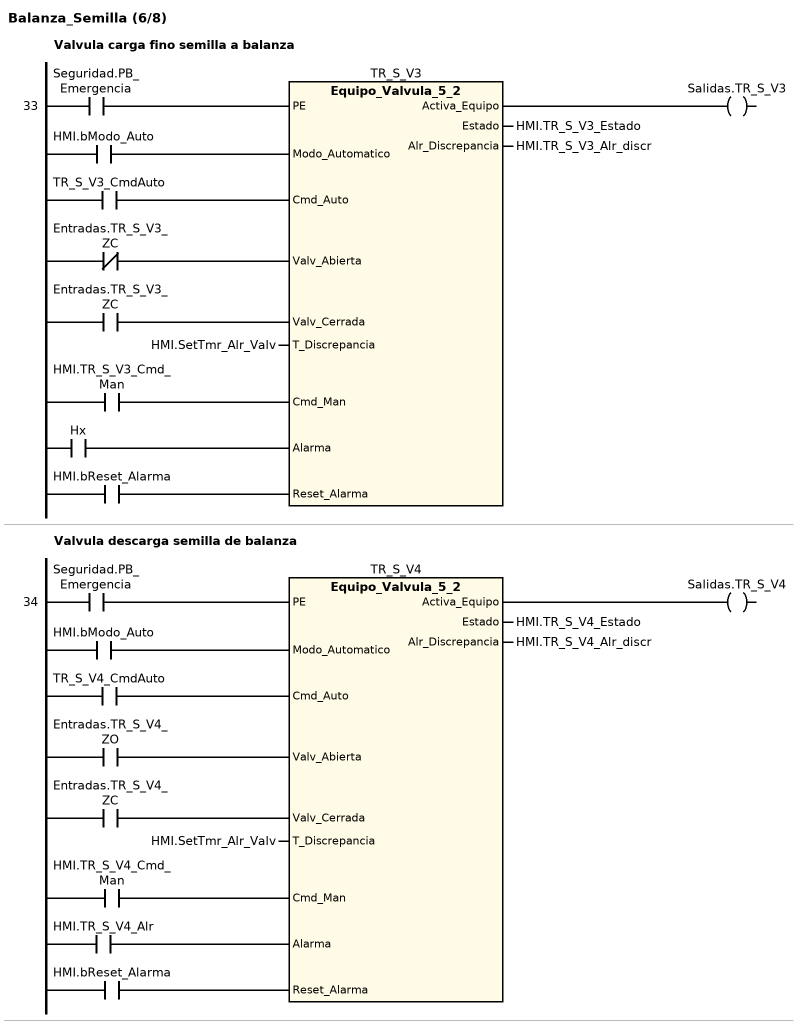
// NETWORK 33: Valvula carga fino semilla a balanza
TR_S_V3(
    PE := Seguridad.PB_Emergencia,
    Modo_Automatico := HMI.bModo_Auto,
    Cmd_Auto := TR_S_V3_CmdAuto,
    Valv_Abierta := NOT Entradas.TR_S_V3_ZC,
    Valv_Cerrada := Entradas.TR_S_V3_ZC,
    T_Discrepancia := HMI.SetTmr_Alr_Valv,
    Cmd_Man := HMI.TR_S_V3_Cmd_Man,
    Alarma := Hx,
    Reset_Alarma := HMI.bReset_Alarma,
    Estado => HMI.TR_S_V3_Estado,
    Alr_Discrepancia => HMI.TR_S_V3_Alr_discr); // Equipo_Valvula_5_2
Salidas.TR_S_V3 := TR_S_V3.Activa_Equipo;

// NETWORK 34: Valvula descarga semilla de balanza
TR_S_V4(
    PE := Seguridad.PB_Emergencia,
    Modo_Automatico := HMI.bModo_Auto,
    Cmd_Auto := TR_S_V4_CmdAuto,
    Valv_Abierta := Entradas.TR_S_V4_ZO,
    Valv_Cerrada := Entradas.TR_S_V4_ZC,
    T_Discrepancia := HMI.SetTmr_Alr_Valv,
    Cmd_Man := HMI.TR_S_V4_Cmd_Man,
    Alarma := HMI.TR_S_V4_Alr,
    Reset_Alarma := HMI.bReset_Alarma,
    Estado => HMI.TR_S_V4_Estado,
    Alr_Discrepancia => HMI.TR_S_V4_Alr_discr); // Equipo_Valvula_5_2
Salidas.TR_S_V4 := TR_S_V4.Activa_Equipo;

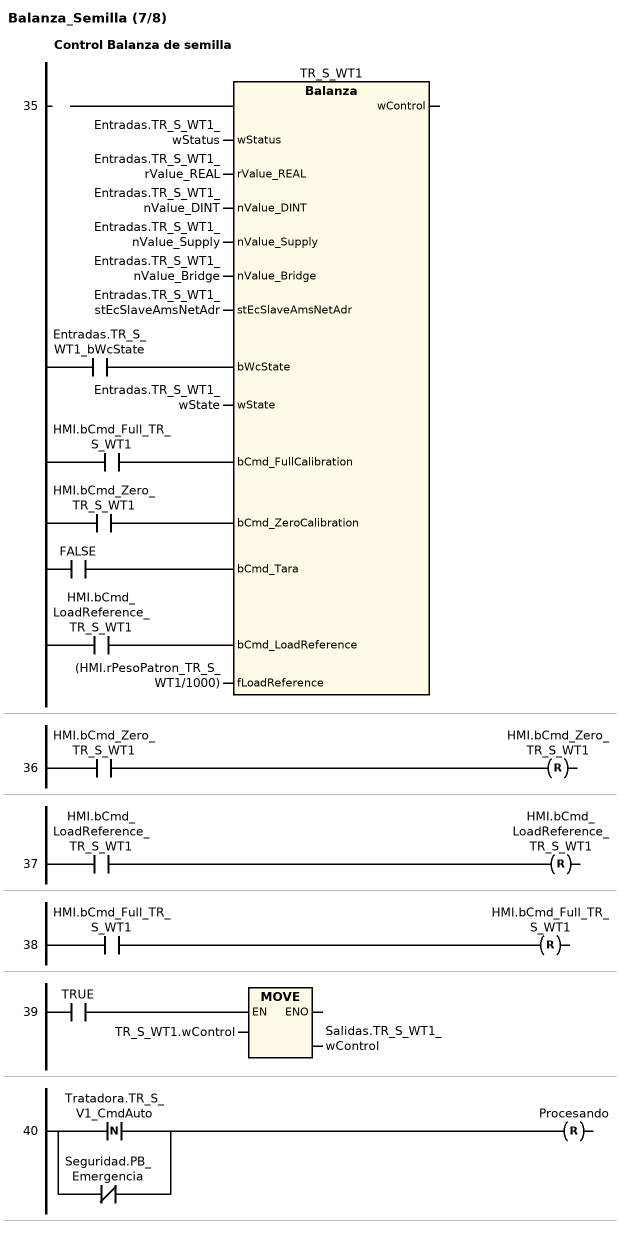
// NETWORK 35: Control Balanza de semilla
TR_S_WT1(
    wStatus := Entradas.TR_S_WT1_wStatus,
    rValue_REAL := Entradas.TR_S_WT1_rValue_REAL,
    nValue_DINT := Entradas.TR_S_WT1_nValue_DINT,
    nValue_Supply := Entradas.TR_S_WT1_nValue_Supply,
    nValue_Bridge := Entradas.TR_S_WT1_nValue_Bridge,
    stEcSlaveAmsNetAdr := Entradas.TR_S_WT1_stEcSlaveAmsNetAdr,
    bWcState := Entradas.TR_S_WT1_bWcState,
    wState := Entradas.TR_S_WT1_wState,
    bCmd_FullCalibration := HMI.bCmd_Full_TR_S_WT1,
    bCmd_ZeroCalibration := HMI.bCmd_Zero_TR_S_WT1,
    bCmd_Tara := FALSE,
    bCmd_LoadReference := HMI.bCmd_LoadReference_TR_S_WT1,
    fLoadReference := (HMI.rPesoPatron_TR_S_WT1/1000)); // Balanza

// NETWORK 36
HMI.bCmd_Zero_TR_S_WT1 R= HMI.bCmd_Zero_TR_S_WT1;

// NETWORK 37
HMI.bCmd_LoadReference_TR_S_WT1 R= HMI.bCmd_LoadReference_TR_S_WT1;

// NETWORK 38
HMI.bCmd_Full_TR_S_WT1 R= HMI.bCmd_Full_TR_S_WT1;

// NETWORK 39
Salidas.TR_S_WT1_wControl := TR_S_WT1.wControl;

// NETWORK 40
_ft1(CLK := Tratadora.TR_S_V1_CmdAuto);
Procesando R= _ft1.Q OR NOT Seguridad.PB_Emergencia;

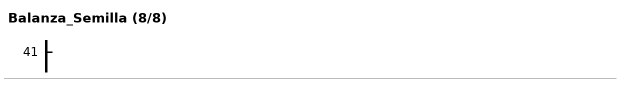
// NETWORK 41

END_PROGRAM

// ---- POUs/Pesajes/Balanza.TcPOU
FUNCTION_BLOCK Balanza
VAR_INPUT
				(* process data IN*)
	wStatus :WORD;
	rValue_REAL  :REAL;
	nValue_DINT  :DINT;
	nValue_Supply :DINT;		(*only for voltage measurement, change PDO settings"*)
	nValue_Bridge:DINT;		(*only for voltage measurement, change PDO settings"*)
	stEcSlaveAmsNetAdr :ST_AmsAddr;
	bWcState:BOOL;
	wState:WORD;
	bCmd_FullCalibration:BOOL;
	bCmd_ZeroCalibration:BOOL;
	bCmd_Tara:BOOL;
	bCmd_LoadReference:BOOL;
	fLoadReference	:REAL;

END_VAR
VAR_OUTPUT
				(* process data OUT*)
	wControl :WORD;
END_VAR

VAR

	(* commands *)
	bStartManualCalib:BOOL;
	bDisableCalibration:BOOL:=TRUE;
	bInputFreeze:BOOL;
	bSampleMode:BOOL;
	bTara:BOOL;

	bCmd_TaraEEProm:BOOL;

